REGION Network 40: ERROR - Descarga por S1
   RUNG wire#powerrail
      Contact( #EstadoZona.Rearme_CBx )
      S_RS(operand := #EstadoVI.Err_FTF_Sin_LibPHS_S1, s1 := wire#w2)
      S_Coil( #EstadoVI.Error_Mx )
   END_RUNG
   RUNG wire#powerrail
      I_Contact( #ConfigFB.SinErrorLiberarPHS_S1 )
      wire#w1
      Contact( #Mx_ET50 )
      Contact( #FTF_MSal )
      Contact( #Selec_M1_Salida )
   END_RUNG wire#w2
   RUNG wire#powerrail
      Contact( #ConfigFB.SinErrorLiberarPHS_S1 )
      I_Contact( #CNTSeg_ApHsMx.QU )
   END_RUNG wire#w1
   // the same network as SCL:
   IF #EstadoZona.Rearme_CBx THEN
       #EstadoVI.Err_FTF_Sin_LibPHS_S1 := FALSE;   // RS flip-flop
   END_IF;
   IF (NOT #ConfigFB.SinErrorLiberarPHS_S1 OR (#ConfigFB.SinErrorLiberarPHS_S1 AND NOT #CNTSeg_ApHsMx.QU)) AND #Mx_ET50 AND #FTF_MSal AND #Selec_M1_Salida THEN
       #EstadoVI.Err_FTF_Sin_LibPHS_S1 := TRUE;
   END_IF;
   IF #EstadoVI.Err_FTF_Sin_LibPHS_S1 THEN #EstadoVI.Error_Mx := TRUE; END_IF;
END_REGION

REGION Network 41: ERROR - Descarga por S3
   RUNG wire#powerrail
      Contact( #EstadoZona.Rearme_CBx )
      S_RS(operand := #EstadoVI.Err_FTF_Sin_LibPHS_S3, s1 := wire#w2)
      S_Coil( #EstadoVI.Error_Mx )
   END_RUNG
   RUNG wire#powerrail
      I_Contact( #ConfigFB.SinErrorLiberarPHS_S3 )
      wire#w1
      Contact( #Mx_ET50 )
      Contact( #FTF_MSal )
      Contact( #Selec_M3_Salida )
   END_RUNG wire#w2
   RUNG wire#powerrail
      Contact( #ConfigFB.SinErrorLiberarPHS_S3 )
      I_Contact( #CNTSeg_ApHsMx.QU )
   END_RUNG wire#w1
   // the same network as SCL:
   IF #EstadoZona.Rearme_CBx THEN
       #EstadoVI.Err_FTF_Sin_LibPHS_S3 := FALSE;   // RS flip-flop
   END_IF;
   IF (NOT #ConfigFB.SinErrorLiberarPHS_S3 OR (#ConfigFB.SinErrorLiberarPHS_S3 AND NOT #CNTSeg_ApHsMx.QU)) AND #Mx_ET50 AND #FTF_MSal AND #Selec_M3_Salida THEN
       #EstadoVI.Err_FTF_Sin_LibPHS_S3 := TRUE;
   END_IF;
   IF #EstadoVI.Err_FTF_Sin_LibPHS_S3 THEN #EstadoVI.Error_Mx := TRUE; END_IF;
END_REGION

REGION Network 42: TMP - ERROR - TimeOut Avance
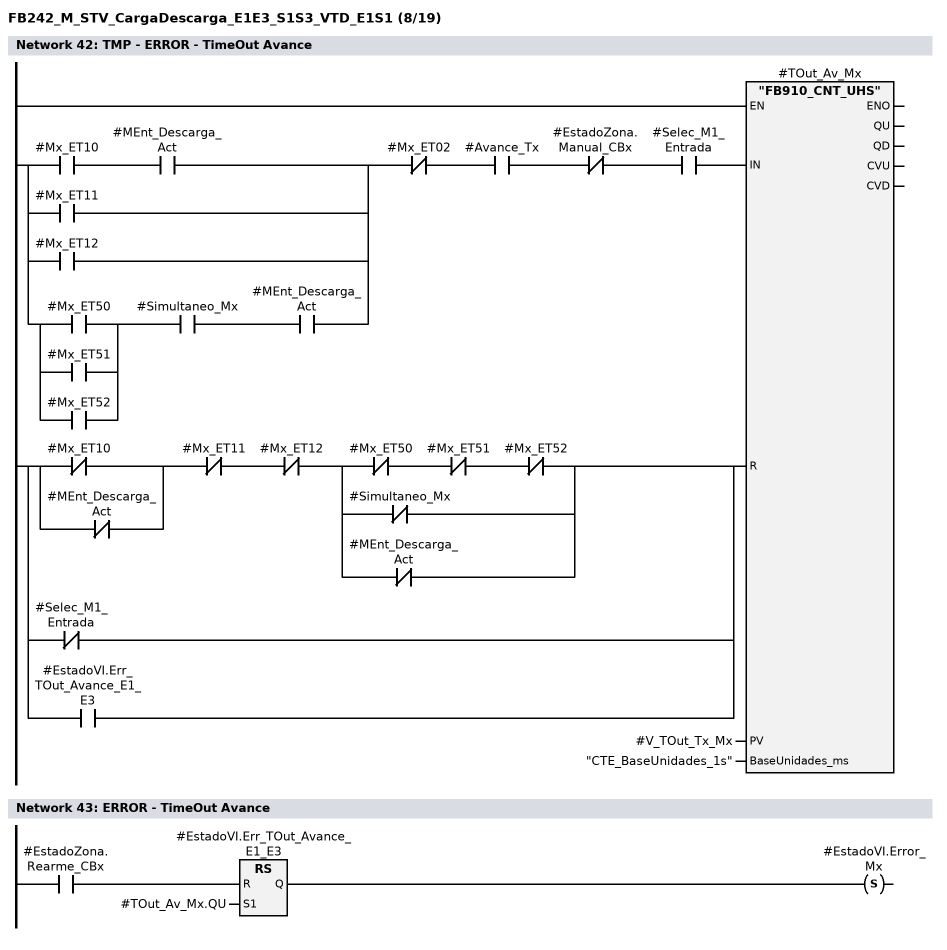
   RUNG wire#powerrail
      #TOut_Av_Mx(IN := wire#w3, R := wire#w6, PV := #V_TOut_Tx_Mx, BaseUnidades_ms := "CTE_BaseUnidades_1s", QU =>, QD =>, CVU =>, CVD =>)
   END_RUNG
   RUNG wire#powerrail
      Contact( #Mx_ET10 )
      Contact( #MEnt_Descarga_Act )
      wire#w1
      I_Contact( #Mx_ET02 )
      Contact( #Avance_Tx )
      I_Contact( #EstadoZona.Manual_CBx )
      Contact( #Selec_M1_Entrada )
   END_RUNG wire#w3
   RUNG wire#powerrail
      Contact( #Mx_ET11 )
   END_RUNG wire#w1
   RUNG wire#powerrail
      Contact( #Mx_ET12 )
   END_RUNG wire#w1
   RUNG wire#powerrail
      Contact( #Mx_ET50 )
      wire#w2
      Contact( #Simultaneo_Mx )
      Contact( #MEnt_Descarga_Act )
   END_RUNG wire#w1
   RUNG wire#powerrail
      Contact( #Mx_ET51 )
   END_RUNG wire#w2
   RUNG wire#powerrail
      Contact( #Mx_ET52 )
   END_RUNG wire#w2
   RUNG wire#powerrail
      I_Contact( #Mx_ET10 )
      wire#w4
      I_Contact( #Mx_ET11 )
      I_Contact( #Mx_ET12 )
      wire#w5
      I_Contact( #Mx_ET50 )
      I_Contact( #Mx_ET51 )
      I_Contact( #Mx_ET52 )
   END_RUNG wire#w6
   RUNG wire#powerrail
      I_Contact( #MEnt_Descarga_Act )
   END_RUNG wire#w4
   RUNG wire#w5
      I_Contact( #Simultaneo_Mx )
   END_RUNG wire#w6
   RUNG wire#w5
      I_Contact( #MEnt_Descarga_Act )
   END_RUNG wire#w6
   RUNG wire#powerrail
      I_Contact( #Selec_M1_Entrada )
   END_RUNG wire#w6
   RUNG wire#powerrail
      Contact( #EstadoVI.Err_TOut_Avance_E1_E3 )
   END_RUNG wire#w6
   // the same network as SCL:
   #TOut_Av_Mx(IN := ((#Mx_ET10 AND #MEnt_Descarga_Act) OR #Mx_ET11 OR #Mx_ET12 OR ((#Mx_ET50 OR #Mx_ET51 OR #Mx_ET52) AND #Simultaneo_Mx AND #MEnt_Descarga_Act)) AND NOT #Mx_ET02 AND #Avance_Tx AND NOT #EstadoZona.Manual_CBx AND #Selec_M1_Entrada,   // "FB910_CNT_UHS"
               R := ((NOT #Mx_ET10 OR NOT #MEnt_Descarga_Act) AND NOT #Mx_ET11 AND NOT #Mx_ET12 AND ((NOT #Mx_ET50 AND NOT #Mx_ET51 AND NOT #Mx_ET52) OR NOT #Simultaneo_Mx OR NOT #MEnt_Descarga_Act)) OR NOT #Selec_M1_Entrada OR #EstadoVI.Err_TOut_Avance_E1_E3,
               PV := #V_TOut_Tx_Mx,
               BaseUnidades_ms := "CTE_BaseUnidades_1s");
END_REGION

REGION Network 43: ERROR - TimeOut Avance
   RUNG wire#powerrail
      Contact( #EstadoZona.Rearme_CBx )
      S_RS(operand := #EstadoVI.Err_TOut_Avance_E1_E3, s1 := #TOut_Av_Mx.QU)
      S_Coil( #EstadoVI.Error_Mx )
   END_RUNG
   // the same network as SCL:
   IF #EstadoZona.Rearme_CBx THEN
       #EstadoVI.Err_TOut_Avance_E1_E3 := FALSE;   // RS flip-flop
   END_IF;
   IF #TOut_Av_Mx.QU THEN #EstadoVI.Err_TOut_Avance_E1_E3 := TRUE; END_IF;
   IF #EstadoVI.Err_TOut_Avance_E1_E3 THEN #EstadoVI.Error_Mx := TRUE; END_IF;
END_REGION

REGION Network 44: TMP - ERROR - TimeOut Retroceso
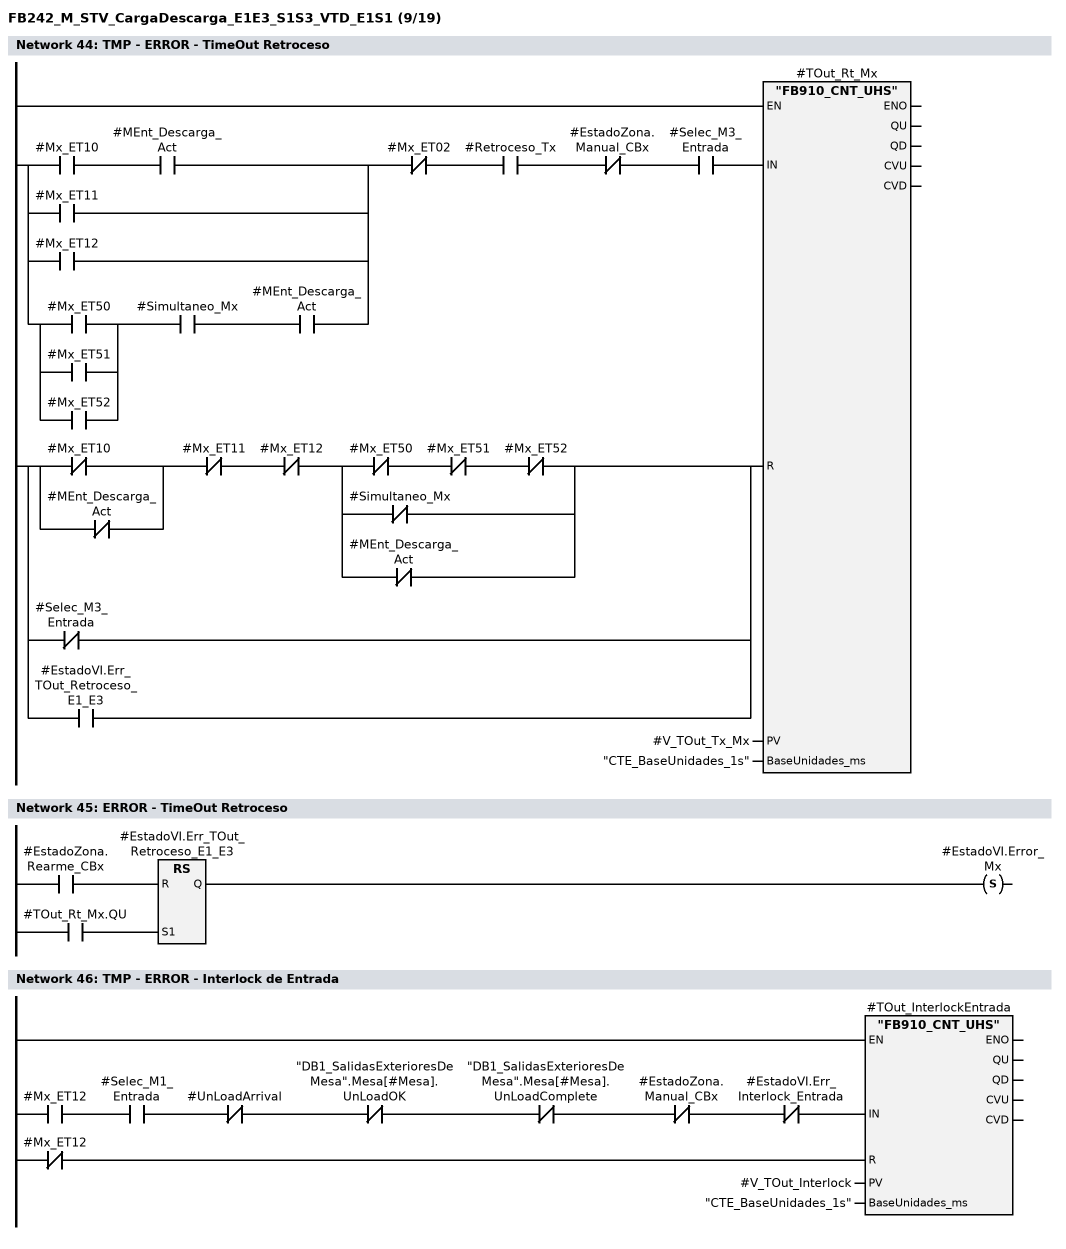
   RUNG wire#powerrail
      #TOut_Rt_Mx(IN := wire#w3, R := wire#w6, PV := #V_TOut_Tx_Mx, BaseUnidades_ms := "CTE_BaseUnidades_1s", QU =>, QD =>, CVU =>, CVD =>)
   END_RUNG
   RUNG wire#powerrail
      Contact( #Mx_ET10 )
      Contact( #MEnt_Descarga_Act )
      wire#w1
      I_Contact( #Mx_ET02 )
      Contact( #Retroceso_Tx )
      I_Contact( #EstadoZona.Manual_CBx )
      Contact( #Selec_M3_Entrada )
   END_RUNG wire#w3
   RUNG wire#powerrail
      Contact( #Mx_ET11 )
   END_RUNG wire#w1
   RUNG wire#powerrail
      Contact( #Mx_ET12 )
   END_RUNG wire#w1
   RUNG wire#powerrail
      Contact( #Mx_ET50 )
      wire#w2
      Contact( #Simultaneo_Mx )
      Contact( #MEnt_Descarga_Act )
   END_RUNG wire#w1
   RUNG wire#powerrail
      Contact( #Mx_ET51 )
   END_RUNG wire#w2
   RUNG wire#powerrail
      Contact( #Mx_ET52 )
   END_RUNG wire#w2
   RUNG wire#powerrail
      I_Contact( #Mx_ET10 )
      wire#w4
      I_Contact( #Mx_ET11 )
      I_Contact( #Mx_ET12 )
      wire#w5
      I_Contact( #Mx_ET50 )
      I_Contact( #Mx_ET51 )
      I_Contact( #Mx_ET52 )
   END_RUNG wire#w6
   RUNG wire#powerrail
      I_Contact( #MEnt_Descarga_Act )
   END_RUNG wire#w4
   RUNG wire#w5
      I_Contact( #Simultaneo_Mx )
   END_RUNG wire#w6
   RUNG wire#w5
      I_Contact( #MEnt_Descarga_Act )
   END_RUNG wire#w6
   RUNG wire#powerrail
      I_Contact( #Selec_M3_Entrada )
   END_RUNG wire#w6
   RUNG wire#powerrail
      Contact( #EstadoVI.Err_TOut_Retroceso_E1_E3 )
   END_RUNG wire#w6
   // the same network as SCL:
   #TOut_Rt_Mx(IN := ((#Mx_ET10 AND #MEnt_Descarga_Act) OR #Mx_ET11 OR #Mx_ET12 OR ((#Mx_ET50 OR #Mx_ET51 OR #Mx_ET52) AND #Simultaneo_Mx AND #MEnt_Descarga_Act)) AND NOT #Mx_ET02 AND #Retroceso_Tx AND NOT #EstadoZona.Manual_CBx AND #Selec_M3_Entrada,   // "FB910_CNT_UHS"
               R := ((NOT #Mx_ET10 OR NOT #MEnt_Descarga_Act) AND NOT #Mx_ET11 AND NOT #Mx_ET12 AND ((NOT #Mx_ET50 AND NOT #Mx_ET51 AND NOT #Mx_ET52) OR NOT #Simultaneo_Mx OR NOT #MEnt_Descarga_Act)) OR NOT #Selec_M3_Entrada OR #EstadoVI.Err_TOut_Retroceso_E1_E3,
               PV := #V_TOut_Tx_Mx,
               BaseUnidades_ms := "CTE_BaseUnidades_1s");
END_REGION

REGION Network 45: ERROR - TimeOut Retroceso
   RUNG wire#powerrail
      Contact( #EstadoZona.Rearme_CBx )
      S_RS(operand := #EstadoVI.Err_TOut_Retroceso_E1_E3, s1 := wire#w1)
      S_Coil( #EstadoVI.Error_Mx )
   END_RUNG
   RUNG wire#powerrail
      Contact( #TOut_Rt_Mx.QU )
   END_RUNG wire#w1
   // the same network as SCL:
   IF #EstadoZona.Rearme_CBx THEN
       #EstadoVI.Err_TOut_Retroceso_E1_E3 := FALSE;   // RS flip-flop
   END_IF;
   IF #TOut_Rt_Mx.QU THEN #EstadoVI.Err_TOut_Retroceso_E1_E3 := TRUE; END_IF;
   IF #EstadoVI.Err_TOut_Retroceso_E1_E3 THEN #EstadoVI.Error_Mx := TRUE; END_IF;
END_REGION

REGION Network 46: TMP - ERROR - Interlock de Entrada
   RUNG wire#powerrail
      #TOut_InterlockEntrada(IN := wire#w1, R := wire#w2, PV := #V_TOut_Interlock, BaseUnidades_ms := "CTE_BaseUnidades_1s", QU =>, QD =>, CVU =>, CVD =>)
   END_RUNG
   RUNG wire#powerrail
      Contact( #Mx_ET12 )
      Contact( #Selec_M1_Entrada )
      I_Contact( #UnLoadArrival )
      I_Contact( "DB1_SalidasExterioresDeMesa".Mesa[#Mesa].UnLoadOK )
      I_Contact( "DB1_SalidasExterioresDeMesa".Mesa[#Mesa].UnLoadComplete )
      I_Contact( #EstadoZona.Manual_CBx )
      I_Contact( #EstadoVI.Err_Interlock_Entrada )
   END_RUNG wire#w1
   RUNG wire#powerrail
      I_Contact( #Mx_ET12 )
   END_RUNG wire#w2
   // the same network as SCL:
   #TOut_InterlockEntrada(IN := #Mx_ET12 AND #Selec_M1_Entrada AND NOT #UnLoadArrival AND NOT "DB1_SalidasExterioresDeMesa".Mesa[#Mesa].UnLoadOK AND NOT "DB1_SalidasExterioresDeMesa".Mesa[#Mesa].UnLoadComplete AND NOT #EstadoZona.Manual_CBx AND NOT #EstadoVI.Err_Interlock_Entrada,   // "FB910_CNT_UHS"
                          R := NOT #Mx_ET12,
                          PV := #V_TOut_Interlock,
                          BaseUnidades_ms := "CTE_BaseUnidades_1s");
END_REGION

REGION Network 47: ERROR - Interlock de Entrada
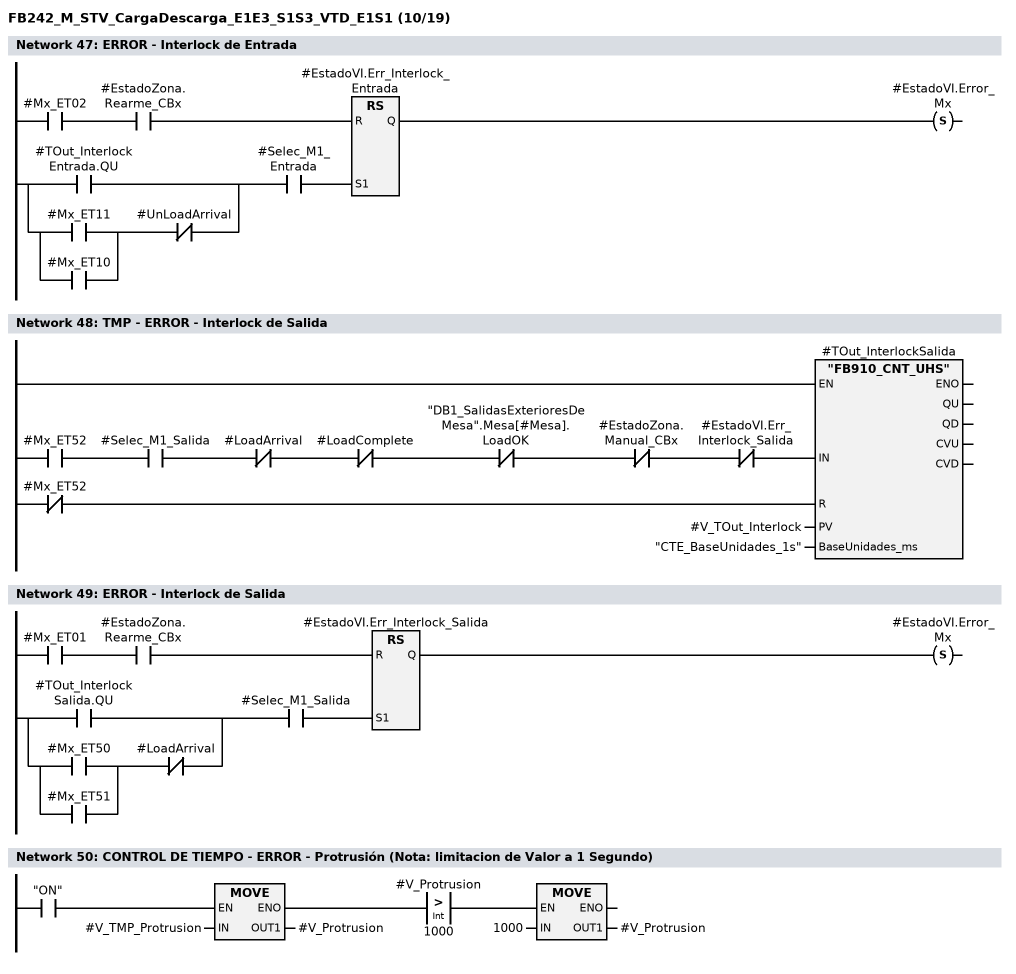
   RUNG wire#powerrail
      Contact( #Mx_ET02 )
      Contact( #EstadoZona.Rearme_CBx )
      S_RS(operand := #EstadoVI.Err_Interlock_Entrada, s1 := wire#w3)
      S_Coil( #EstadoVI.Error_Mx )
   END_RUNG
   RUNG wire#powerrail
      Contact( #TOut_InterlockEntrada.QU )
      wire#w1
      Contact( #Selec_M1_Entrada )
   END_RUNG wire#w3
   RUNG wire#powerrail
      Contact( #Mx_ET11 )
      wire#w2
      I_Contact( #UnLoadArrival )
   END_RUNG wire#w1
   RUNG wire#powerrail
      Contact( #Mx_ET10 )
   END_RUNG wire#w2
   // the same network as SCL:
   IF #Mx_ET02 AND #EstadoZona.Rearme_CBx THEN
       #EstadoVI.Err_Interlock_Entrada := FALSE;   // RS flip-flop
   END_IF;
   IF (#TOut_InterlockEntrada.QU OR ((#Mx_ET11 OR #Mx_ET10) AND NOT #UnLoadArrival)) AND #Selec_M1_Entrada THEN
       #EstadoVI.Err_Interlock_Entrada := TRUE;
   END_IF;
   IF #EstadoVI.Err_Interlock_Entrada THEN #EstadoVI.Error_Mx := TRUE; END_IF;
END_REGION

REGION Network 48: TMP - ERROR - Interlock de Salida
   RUNG wire#powerrail
      #TOut_InterlockSalida(IN := wire#w1, R := wire#w2, PV := #V_TOut_Interlock, BaseUnidades_ms := "CTE_BaseUnidades_1s", QU =>, QD =>, CVU =>, CVD =>)
   END_RUNG
   RUNG wire#powerrail
      Contact( #Mx_ET52 )
      Contact( #Selec_M1_Salida )
      I_Contact( #LoadArrival )
      I_Contact( #LoadComplete )
      I_Contact( "DB1_SalidasExterioresDeMesa".Mesa[#Mesa].LoadOK )
      I_Contact( #EstadoZona.Manual_CBx )
      I_Contact( #EstadoVI.Err_Interlock_Salida )
   END_RUNG wire#w1
   RUNG wire#powerrail
      I_Contact( #Mx_ET52 )
   END_RUNG wire#w2
   // the same network as SCL:
   #TOut_InterlockSalida(IN := #Mx_ET52 AND #Selec_M1_Salida AND NOT #LoadArrival AND NOT #LoadComplete AND NOT "DB1_SalidasExterioresDeMesa".Mesa[#Mesa].LoadOK AND NOT #EstadoZona.Manual_CBx AND NOT #EstadoVI.Err_Interlock_Salida,   // "FB910_CNT_UHS"
                         R := NOT #Mx_ET52,
                         PV := #V_TOut_Interlock,
                         BaseUnidades_ms := "CTE_BaseUnidades_1s");
END_REGION

REGION Network 49: ERROR - Interlock de Salida
   RUNG wire#powerrail
      Contact( #Mx_ET01 )
      Contact( #EstadoZona.Rearme_CBx )
      S_RS(operand := #EstadoVI.Err_Interlock_Salida, s1 := wire#w3)
      S_Coil( #EstadoVI.Error_Mx )
   END_RUNG
   RUNG wire#powerrail
      Contact( #TOut_InterlockSalida.QU )
      wire#w1
      Contact( #Selec_M1_Salida )
   END_RUNG wire#w3
   RUNG wire#powerrail
      Contact( #Mx_ET50 )
      wire#w2
      I_Contact( #LoadArrival )
   END_RUNG wire#w1
   RUNG wire#powerrail
      Contact( #Mx_ET51 )
   END_RUNG wire#w2
   // the same network as SCL:
   IF #Mx_ET01 AND #EstadoZona.Rearme_CBx THEN
       #EstadoVI.Err_Interlock_Salida := FALSE;   // RS flip-flop
   END_IF;
   IF (#TOut_InterlockSalida.QU OR ((#Mx_ET50 OR #Mx_ET51) AND NOT #LoadArrival)) AND #Selec_M1_Salida THEN
       #EstadoVI.Err_Interlock_Salida := TRUE;
   END_IF;
   IF #EstadoVI.Err_Interlock_Salida THEN #EstadoVI.Error_Mx := TRUE; END_IF;
END_REGION

REGION Network 50: CONTROL DE TIEMPO - ERROR - Protrusión (Nota: limitacion de Valor a 1 Segundo)
   RUNG wire#powerrail
      Contact( "ON" )
      Move(in := #V_TMP_Protrusion, out1 => #V_Protrusion)
      { S7_Templates := "SrcType := Int" } GT_Contact(in1 := #V_Protrusion, in2 := 1000)
      Move(in := 1000, out1 => #V_Protrusion)
   END_RUNG
   // the same network as SCL:
   IF "ON" THEN #V_Protrusion := #V_TMP_Protrusion; END_IF;
   IF "ON" AND (#V_Protrusion > 1000) THEN #V_Protrusion := 1000; END_IF;
END_REGION

REGION Network 51: TMP - ERROR - Protrusión
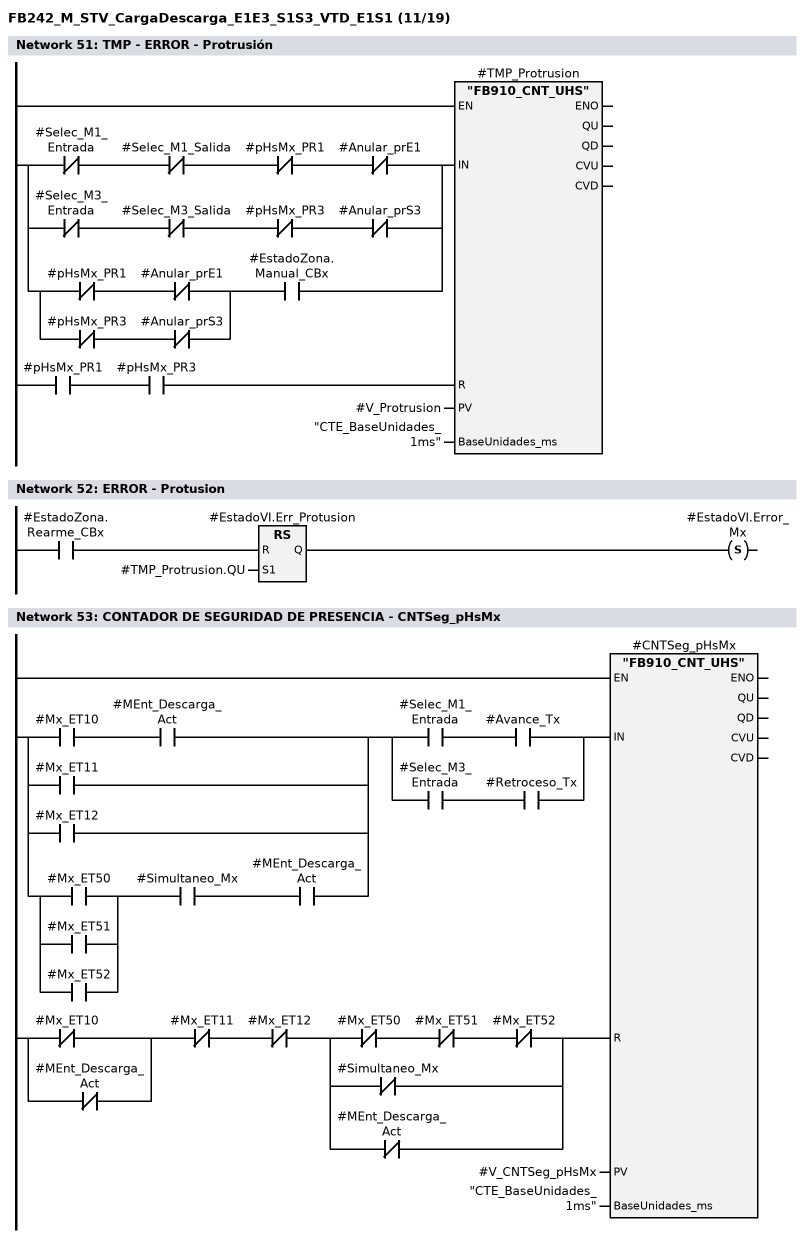
   RUNG wire#powerrail
      #TMP_Protrusion(IN := wire#w2, R := wire#w3, PV := #V_Protrusion, BaseUnidades_ms := "CTE_BaseUnidades_1ms", QU =>, QD =>, CVU =>, CVD =>)
   END_RUNG
   RUNG wire#powerrail
      I_Contact( #Selec_M1_Entrada )
      I_Contact( #Selec_M1_Salida )
      I_Contact( #pHsMx_PR1 )
      I_Contact( #Anular_prE1 )
   END_RUNG wire#w2
   RUNG wire#powerrail
      I_Contact( #Selec_M3_Entrada )
      I_Contact( #Selec_M3_Salida )
      I_Contact( #pHsMx_PR3 )
      I_Contact( #Anular_prS3 )
   END_RUNG wire#w2
   RUNG wire#powerrail
      I_Contact( #pHsMx_PR1 )
      I_Contact( #Anular_prE1 )
      wire#w1
      Contact( #EstadoZona.Manual_CBx )
   END_RUNG wire#w2
   RUNG wire#powerrail
      I_Contact( #pHsMx_PR3 )
      I_Contact( #Anular_prS3 )
   END_RUNG wire#w1
   RUNG wire#powerrail
      Contact( #pHsMx_PR1 )
      Contact( #pHsMx_PR3 )
   END_RUNG wire#w3
   // the same network as SCL:
   #TMP_Protrusion(IN := (NOT #Selec_M1_Entrada AND NOT #Selec_M1_Salida AND NOT #pHsMx_PR1 AND NOT #Anular_prE1) OR (NOT #Selec_M3_Entrada AND NOT #Selec_M3_Salida AND NOT #pHsMx_PR3 AND NOT #Anular_prS3) OR (((NOT #pHsMx_PR1 AND NOT #Anular_prE1) OR (NOT #pHsMx_PR3 AND NOT #Anular_prS3)) AND #EstadoZona.Manual_CBx),   // "FB910_CNT_UHS"
                   R := #pHsMx_PR1 AND #pHsMx_PR3,
                   PV := #V_Protrusion,
                   BaseUnidades_ms := "CTE_BaseUnidades_1ms");
END_REGION

REGION Network 52: ERROR - Protusion
   RUNG wire#powerrail
      Contact( #EstadoZona.Rearme_CBx )
      S_RS(operand := #EstadoVI.Err_Protusion, s1 := #TMP_Protrusion.QU)
      S_Coil( #EstadoVI.Error_Mx )
   END_RUNG
   // the same network as SCL:
   IF #EstadoZona.Rearme_CBx THEN
       #EstadoVI.Err_Protusion := FALSE;   // RS flip-flop
   END_IF;
   IF #TMP_Protrusion.QU THEN #EstadoVI.Err_Protusion := TRUE; END_IF;
   IF #EstadoVI.Err_Protusion THEN #EstadoVI.Error_Mx := TRUE; END_IF;
END_REGION

REGION Network 53: CONTADOR DE SEGURIDAD DE PRESENCIA - CNTSeg_pHsMx
   RUNG wire#powerrail
      #CNTSeg_pHsMx(IN := wire#w3, R := wire#w6, PV := #V_CNTSeg_pHsMx, BaseUnidades_ms := "CTE_BaseUnidades_1ms", QU =>, QD =>, CVU =>, CVD =>)
   END_RUNG
   RUNG wire#powerrail
      Contact( #Mx_ET10 )
      Contact( #MEnt_Descarga_Act )
      wire#w1
      Contact( #Selec_M1_Entrada )
      Contact( #Avance_Tx )
   END_RUNG wire#w3
   RUNG wire#powerrail
      Contact( #Mx_ET11 )
   END_RUNG wire#w1
   RUNG wire#powerrail
      Contact( #Mx_ET12 )
   END_RUNG wire#w1
   RUNG wire#powerrail
      Contact( #Mx_ET50 )
      wire#w2
      Contact( #Simultaneo_Mx )
      Contact( #MEnt_Descarga_Act )
   END_RUNG wire#w1
   RUNG wire#powerrail
      Contact( #Mx_ET51 )
   END_RUNG wire#w2
   RUNG wire#powerrail
      Contact( #Mx_ET52 )
   END_RUNG wire#w2
   RUNG wire#w1
      Contact( #Selec_M3_Entrada )
      Contact( #Retroceso_Tx )
   END_RUNG wire#w3
   RUNG wire#powerrail
      I_Contact( #Mx_ET10 )
      wire#w4
      I_Contact( #Mx_ET11 )
      I_Contact( #Mx_ET12 )
      wire#w5
      I_Contact( #Mx_ET50 )
      I_Contact( #Mx_ET51 )
      I_Contact( #Mx_ET52 )
   END_RUNG wire#w6
   RUNG wire#powerrail
      I_Contact( #MEnt_Descarga_Act )
   END_RUNG wire#w4
   RUNG wire#w5
      I_Contact( #Simultaneo_Mx )
   END_RUNG wire#w6
   RUNG wire#w5
      I_Contact( #MEnt_Descarga_Act )
   END_RUNG wire#w6
   // the same network as SCL:
   #CNTSeg_pHsMx(IN := ((#Mx_ET10 AND #MEnt_Descarga_Act) OR #Mx_ET11 OR #Mx_ET12 OR ((#Mx_ET50 OR #Mx_ET51 OR #Mx_ET52) AND #Simultaneo_Mx AND #MEnt_Descarga_Act)) AND ((#Selec_M1_Entrada AND #Avance_Tx) OR (#Selec_M3_Entrada AND #Retroceso_Tx)),   // "FB910_CNT_UHS"
                 R := (NOT #Mx_ET10 OR NOT #MEnt_Descarga_Act) AND NOT #Mx_ET11 AND NOT #Mx_ET12 AND ((NOT #Mx_ET50 AND NOT #Mx_ET51 AND NOT #Mx_ET52) OR NOT #Simultaneo_Mx OR NOT #MEnt_Descarga_Act),
                 PV := #V_CNTSeg_pHsMx,
                 BaseUnidades_ms := "CTE_BaseUnidades_1ms");
END_REGION

REGION Network 54: CONTADOR DE PRESENCIA - CNT_pHsMx
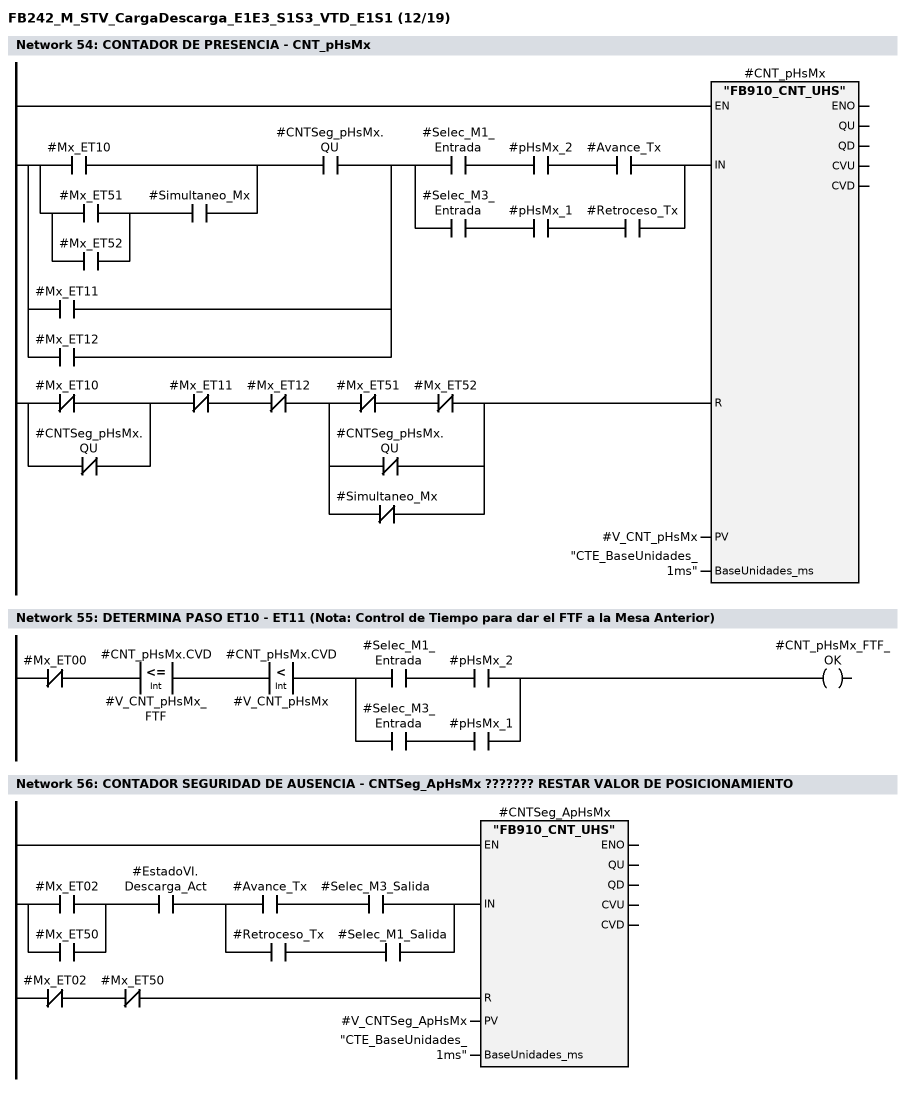
   RUNG wire#powerrail
      #CNT_pHsMx(IN := wire#w4, R := wire#w7, PV := #V_CNT_pHsMx, BaseUnidades_ms := "CTE_BaseUnidades_1ms", QU =>, QD =>, CVU =>, CVD =>)
   END_RUNG
   RUNG wire#powerrail
      Contact( #Mx_ET10 )
      wire#w1
      Contact( #CNTSeg_pHsMx.QU )
      wire#w3
      Contact( #Selec_M1_Entrada )
      Contact( #pHsMx_2 )
      Contact( #Avance_Tx )
   END_RUNG wire#w4
   RUNG wire#powerrail
      Contact( #Mx_ET51 )
      wire#w2
      Contact( #Simultaneo_Mx )
   END_RUNG wire#w1
   RUNG wire#powerrail
      Contact( #Mx_ET52 )
   END_RUNG wire#w2
   RUNG wire#powerrail
      Contact( #Mx_ET11 )
   END_RUNG wire#w3
   RUNG wire#powerrail
      Contact( #Mx_ET12 )
   END_RUNG wire#w3
   RUNG wire#w3
      Contact( #Selec_M3_Entrada )
      Contact( #pHsMx_1 )
      Contact( #Retroceso_Tx )
   END_RUNG wire#w4
   RUNG wire#powerrail
      I_Contact( #Mx_ET10 )
      wire#w5
      I_Contact( #Mx_ET11 )
      I_Contact( #Mx_ET12 )
      wire#w6
      I_Contact( #Mx_ET51 )
      I_Contact( #Mx_ET52 )
   END_RUNG wire#w7
   RUNG wire#powerrail
      I_Contact( #CNTSeg_pHsMx.QU )
   END_RUNG wire#w5
   RUNG wire#w6
      I_Contact( #CNTSeg_pHsMx.QU )
   END_RUNG wire#w7
   RUNG wire#w6
      I_Contact( #Simultaneo_Mx )
   END_RUNG wire#w7
   // the same network as SCL:
   #CNT_pHsMx(IN := (((#Mx_ET10 OR ((#Mx_ET51 OR #Mx_ET52) AND #Simultaneo_Mx)) AND #CNTSeg_pHsMx.QU) OR #Mx_ET11 OR #Mx_ET12) AND ((#Selec_M1_Entrada AND #pHsMx_2 AND #Avance_Tx) OR (#Selec_M3_Entrada AND #pHsMx_1 AND #Retroceso_Tx)),   // "FB910_CNT_UHS"
              R := (NOT #Mx_ET10 OR NOT #CNTSeg_pHsMx.QU) AND NOT #Mx_ET11 AND NOT #Mx_ET12 AND ((NOT #Mx_ET51 AND NOT #Mx_ET52) OR NOT #CNTSeg_pHsMx.QU OR NOT #Simultaneo_Mx),
              PV := #V_CNT_pHsMx,
              BaseUnidades_ms := "CTE_BaseUnidades_1ms");
END_REGION

REGION Network 55: DETERMINA PASO ET10 - ET11 (Nota: Control de Tiempo para dar el FTF a la Mesa Anterior)
   RUNG wire#powerrail
      I_Contact( #Mx_ET00 )
      { S7_Templates := "SrcType := Int" } LE_Contact(in1 := #CNT_pHsMx.CVD, in2 := #V_CNT_pHsMx_FTF)
      { S7_Templates := "SrcType := Int" } LT_Contact(in1 := #CNT_pHsMx.CVD, in2 := #V_CNT_pHsMx)
      wire#w1
      Contact( #Selec_M1_Entrada )
      Contact( #pHsMx_2 )
      wire#w2
      Coil( #CNT_pHsMx_FTF_OK )
   END_RUNG
   RUNG wire#w1
      Contact( #Selec_M3_Entrada )
      Contact( #pHsMx_1 )
   END_RUNG wire#w2
   // the same network as SCL:
   #CNT_pHsMx_FTF_OK := NOT #Mx_ET00 AND (#CNT_pHsMx.CVD <= #V_CNT_pHsMx_FTF) AND (#CNT_pHsMx.CVD < #V_CNT_pHsMx) AND ((#Selec_M1_Entrada AND #pHsMx_2) OR (#Selec_M3_Entrada AND #pHsMx_1));
END_REGION

REGION Network 56: CONTADOR SEGURIDAD DE AUSENCIA - CNTSeg_ApHsMx ??????? RESTAR VALOR DE POSICIONAMIENTO
   RUNG wire#powerrail
      #CNTSeg_ApHsMx(IN := wire#w3, R := wire#w4, PV := #V_CNTSeg_ApHsMx, BaseUnidades_ms := "CTE_BaseUnidades_1ms", QU =>, QD =>, CVU =>, CVD =>)
   END_RUNG
   RUNG wire#powerrail
      Contact( #Mx_ET02 )
      wire#w1
      Contact( #EstadoVI.Descarga_Act )
      wire#w2
      Contact( #Avance_Tx )
      Contact( #Selec_M3_Salida )
   END_RUNG wire#w3
   RUNG wire#powerrail
      Contact( #Mx_ET50 )
   END_RUNG wire#w1
   RUNG wire#w2
      Contact( #Retroceso_Tx )
      Contact( #Selec_M1_Salida )
   END_RUNG wire#w3
   RUNG wire#powerrail
      I_Contact( #Mx_ET02 )
      I_Contact( #Mx_ET50 )
   END_RUNG wire#w4
   // the same network as SCL:
   #CNTSeg_ApHsMx(IN := (#Mx_ET02 OR #Mx_ET50) AND #EstadoVI.Descarga_Act AND ((#Avance_Tx AND #Selec_M3_Salida) OR (#Retroceso_Tx AND #Selec_M1_Salida)),   // "FB910_CNT_UHS"
                  R := NOT #Mx_ET02 AND NOT #Mx_ET50,
                  PV := #V_CNTSeg_ApHsMx,
                  BaseUnidades_ms := "CTE_BaseUnidades_1ms");
END_REGION

REGION Network 57: CONTADOR DE LA AUSENCIA - CNT_ApHsMX
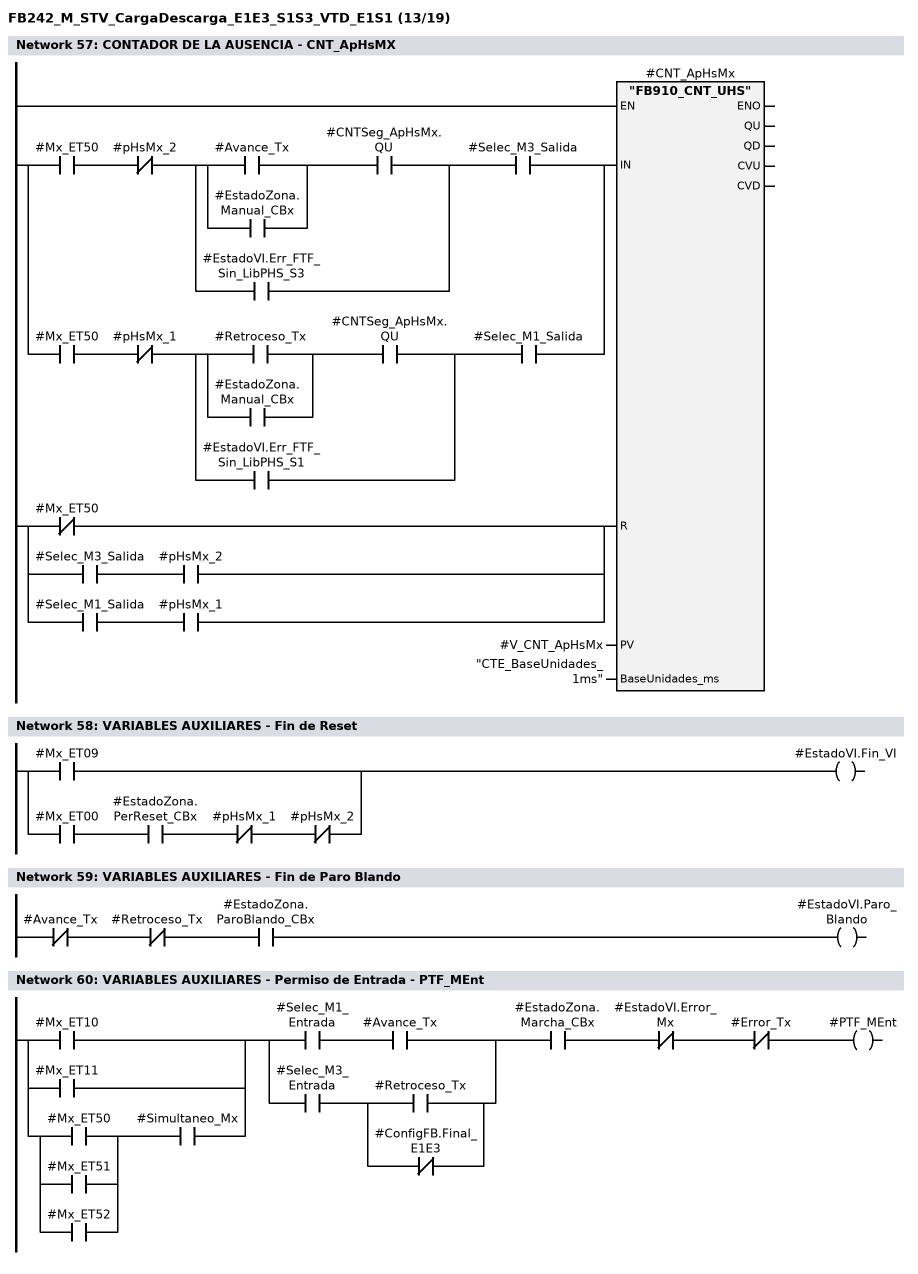
   RUNG wire#powerrail
      #CNT_ApHsMx(IN := wire#w7, R := wire#w8, PV := #V_CNT_ApHsMx, BaseUnidades_ms := "CTE_BaseUnidades_1ms", QU =>, QD =>, CVU =>, CVD =>)
   END_RUNG
   RUNG wire#powerrail
      Contact( #Mx_ET50 )
      I_Contact( #pHsMx_2 )
      wire#w1
      Contact( #Avance_Tx )
      wire#w2
      Contact( #CNTSeg_ApHsMx.QU )
      wire#w3
      Contact( #Selec_M3_Salida )
   END_RUNG wire#w7
   RUNG wire#w1
      Contact( #EstadoZona.Manual_CBx )
   END_RUNG wire#w2
   RUNG wire#w1
      Contact( #EstadoVI.Err_FTF_Sin_LibPHS_S3 )
   END_RUNG wire#w3
   RUNG wire#powerrail
      Contact( #Mx_ET50 )
      I_Contact( #pHsMx_1 )
      wire#w4
      Contact( #Retroceso_Tx )
      wire#w5
      Contact( #CNTSeg_ApHsMx.QU )
      wire#w6
      Contact( #Selec_M1_Salida )
   END_RUNG wire#w7
   RUNG wire#w4
      Contact( #EstadoZona.Manual_CBx )
   END_RUNG wire#w5
   RUNG wire#w4
      Contact( #EstadoVI.Err_FTF_Sin_LibPHS_S1 )
   END_RUNG wire#w6
   RUNG wire#powerrail
      I_Contact( #Mx_ET50 )
   END_RUNG wire#w8
   RUNG wire#powerrail
      Contact( #Selec_M3_Salida )
      Contact( #pHsMx_2 )
   END_RUNG wire#w8
   RUNG wire#powerrail
      Contact( #Selec_M1_Salida )
      Contact( #pHsMx_1 )
   END_RUNG wire#w8
   // the same network as SCL:
   #CNT_ApHsMx(IN := (#Mx_ET50 AND NOT #pHsMx_2 AND (((#Avance_Tx OR #EstadoZona.Manual_CBx) AND #CNTSeg_ApHsMx.QU) OR #EstadoVI.Err_FTF_Sin_LibPHS_S3) AND #Selec_M3_Salida) OR (#Mx_ET50 AND NOT #pHsMx_1 AND (((#Retroceso_Tx OR #EstadoZona.Manual_CBx) AND #CNTSeg_ApHsMx.QU) OR #EstadoVI.Err_FTF_Sin_LibPHS_S1) AND #Selec_M1_Salida),   // "FB910_CNT_UHS"
               R := NOT #Mx_ET50 OR (#Selec_M3_Salida AND #pHsMx_2) OR (#Selec_M1_Salida AND #pHsMx_1),
               PV := #V_CNT_ApHsMx,
               BaseUnidades_ms := "CTE_BaseUnidades_1ms");
END_REGION

REGION Network 58: VARIABLES AUXILIARES - Fin de Reset
   RUNG wire#powerrail
      Contact( #Mx_ET09 )
      wire#w1
      Coil( #EstadoVI.Fin_VI )
   END_RUNG
   RUNG wire#powerrail
      Contact( #Mx_ET00 )
      Contact( #EstadoZona.PerReset_CBx )
      I_Contact( #pHsMx_1 )
      I_Contact( #pHsMx_2 )
   END_RUNG wire#w1
   // the same network as SCL:
   #EstadoVI.Fin_VI := #Mx_ET09 OR (#Mx_ET00 AND #EstadoZona.PerReset_CBx AND NOT #pHsMx_1 AND NOT #pHsMx_2);
END_REGION

REGION Network 59: VARIABLES AUXILIARES - Fin de Paro Blando
   RUNG wire#powerrail
      I_Contact( #Avance_Tx )
      I_Contact( #Retroceso_Tx )
      Contact( #EstadoZona.ParoBlando_CBx )
      Coil( #EstadoVI.Paro_Blando )
   END_RUNG
   // the same network as SCL:
   #EstadoVI.Paro_Blando := NOT #Avance_Tx AND NOT #Retroceso_Tx AND #EstadoZona.ParoBlando_CBx;
END_REGION

REGION Network 60: VARIABLES AUXILIARES - Permiso de Entrada - PTF_MEnt
   RUNG wire#powerrail
      Contact( #Mx_ET10 )
      wire#w1
      Contact( #Selec_M1_Entrada )
      Contact( #Avance_Tx )
      wire#w3
      Contact( #EstadoZona.Marcha_CBx )
      I_Contact( #EstadoVI.Error_Mx )
      I_Contact( #Error_Tx )
      Coil( #PTF_MEnt )
   END_RUNG
   RUNG wire#powerrail
      Contact( #Mx_ET11 )
   END_RUNG wire#w1
   RUNG wire#powerrail
      Contact( #Mx_ET50 )
      wire#w2
      Contact( #Simultaneo_Mx )
   END_RUNG wire#w1
   RUNG wire#powerrail
      Contact( #Mx_ET51 )
   END_RUNG wire#w2
   RUNG wire#powerrail
      Contact( #Mx_ET52 )
   END_RUNG wire#w2
   RUNG wire#w1
      Contact( #Selec_M3_Entrada )
      wire#w4
      Contact( #Retroceso_Tx )
   END_RUNG wire#w3
   RUNG wire#w4
      I_Contact( #ConfigFB.Final_E1E3 )
   END_RUNG wire#w3
   // the same network as SCL:
   #PTF_MEnt := (#Mx_ET10 OR #Mx_ET11 OR ((#Mx_ET50 OR #Mx_ET51 OR #Mx_ET52) AND #Simultaneo_Mx)) AND ((#Selec_M1_Entrada AND #Avance_Tx) OR (#Selec_M3_Entrada AND (#Retroceso_Tx OR NOT #ConfigFB.Final_E1E3))) AND #EstadoZona.Marcha_CBx AND NOT #EstadoVI.Error_Mx AND NOT #Error_Tx;
END_REGION

REGION Network 61: VARIABLES AUXILIARES - Aviso de Salida - AVTF_MEnt
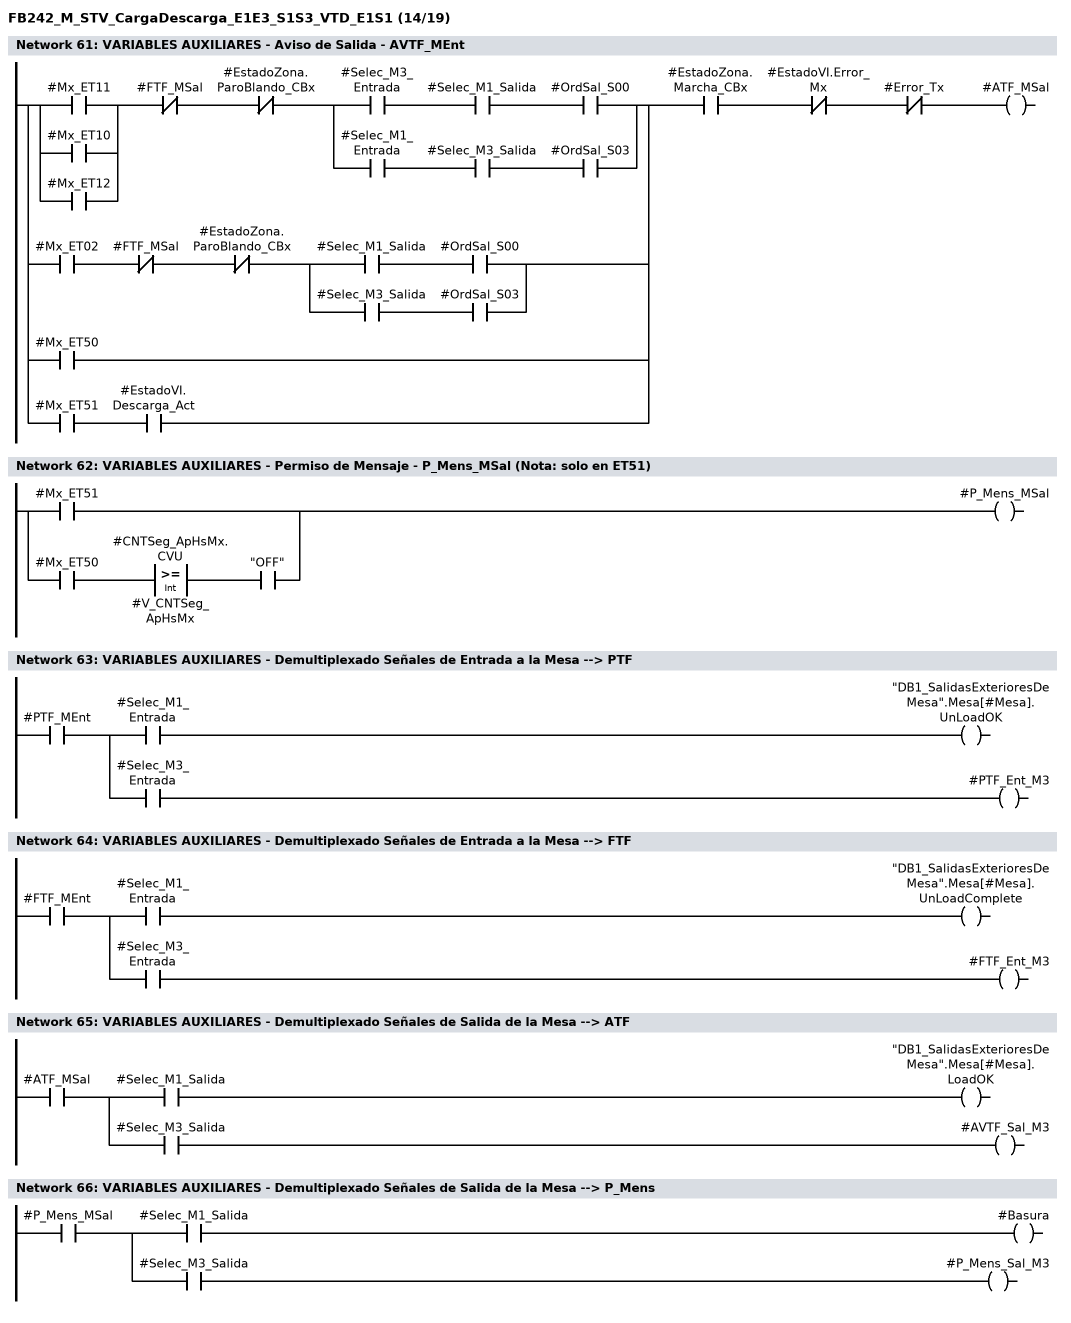
   RUNG wire#powerrail
      Contact( #Mx_ET11 )
      wire#w1
      I_Contact( #FTF_MSal )
      I_Contact( #EstadoZona.ParoBlando_CBx )
      wire#w2
      Contact( #Selec_M3_Entrada )
      Contact( #Selec_M1_Salida )
      Contact( #OrdSal_S00 )
      wire#w3
      Contact( #EstadoZona.Marcha_CBx )
      I_Contact( #EstadoVI.Error_Mx )
      I_Contact( #Error_Tx )
      Coil( #ATF_MSal )
   END_RUNG
   RUNG wire#powerrail
      Contact( #Mx_ET10 )
   END_RUNG wire#w1
   RUNG wire#powerrail
      Contact( #Mx_ET12 )
   END_RUNG wire#w1
   RUNG wire#w2
      Contact( #Selec_M1_Entrada )
      Contact( #Selec_M3_Salida )
      Contact( #OrdSal_S03 )
   END_RUNG wire#w3
   RUNG wire#powerrail
      Contact( #Mx_ET02 )
      I_Contact( #FTF_MSal )
      I_Contact( #EstadoZona.ParoBlando_CBx )
      wire#w4
      Contact( #Selec_M1_Salida )
      Contact( #OrdSal_S00 )
   END_RUNG wire#w3
   RUNG wire#w4
      Contact( #Selec_M3_Salida )
      Contact( #OrdSal_S03 )
   END_RUNG wire#w3
   RUNG wire#powerrail
      Contact( #Mx_ET50 )
   END_RUNG wire#w3
   RUNG wire#powerrail
      Contact( #Mx_ET51 )
      Contact( #EstadoVI.Descarga_Act )
   END_RUNG wire#w3
   // the same network as SCL:
   #ATF_MSal := (((#Mx_ET11 OR #Mx_ET10 OR #Mx_ET12) AND NOT #FTF_MSal AND NOT #EstadoZona.ParoBlando_CBx AND ((#Selec_M3_Entrada AND #Selec_M1_Salida AND #OrdSal_S00) OR (#Selec_M1_Entrada AND #Selec_M3_Salida AND #OrdSal_S03))) OR (#Mx_ET02 AND NOT #FTF_MSal AND NOT #EstadoZona.ParoBlando_CBx AND ((#Selec_M1_Salida AND #OrdSal_S00) OR (#Selec_M3_Salida AND #OrdSal_S03))) OR #Mx_ET50 OR (#Mx_ET51 AND #EstadoVI.Descarga_Act)) AND #EstadoZona.Marcha_CBx AND NOT #EstadoVI.Error_Mx AND NOT #Error_Tx;
END_REGION

REGION Network 62: VARIABLES AUXILIARES - Permiso de Mensaje - P_Mens_MSal (Nota: solo en ET51)
   RUNG wire#powerrail
      Contact( #Mx_ET51 )
      wire#w1
      Coil( #P_Mens_MSal )
   END_RUNG
   RUNG wire#powerrail
      Contact( #Mx_ET50 )
      { S7_Templates := "SrcType := Int" } GE_Contact(in1 := #CNTSeg_ApHsMx.CVU, in2 := #V_CNTSeg_ApHsMx)
      Contact( "OFF" )
   END_RUNG wire#w1
   // the same network as SCL:
   #P_Mens_MSal := #Mx_ET51 OR (#Mx_ET50 AND (#CNTSeg_ApHsMx.CVU >= #V_CNTSeg_ApHsMx) AND "OFF");
END_REGION

REGION Network 63: VARIABLES AUXILIARES - Demultiplexado Señales de Entrada a la Mesa --> PTF
   RUNG wire#powerrail
      Contact( #PTF_MEnt )
      wire#w1
      Contact( #Selec_M1_Entrada )
      Coil( "DB1_SalidasExterioresDeMesa".Mesa[#Mesa].UnLoadOK )
   END_RUNG
   RUNG wire#w1
      Contact( #Selec_M3_Entrada )
      Coil( #PTF_Ent_M3 )
   END_RUNG
   // the same network as SCL:
   "DB1_SalidasExterioresDeMesa".Mesa[#Mesa].UnLoadOK := #PTF_MEnt AND #Selec_M1_Entrada;
   #PTF_Ent_M3 := #PTF_MEnt AND #Selec_M3_Entrada;
END_REGION

REGION Network 64: VARIABLES AUXILIARES - Demultiplexado Señales de Entrada a la Mesa --> FTF
   RUNG wire#powerrail
      Contact( #FTF_MEnt )
      wire#w1
      Contact( #Selec_M1_Entrada )
      Coil( "DB1_SalidasExterioresDeMesa".Mesa[#Mesa].UnLoadComplete )
   END_RUNG
   RUNG wire#w1
      Contact( #Selec_M3_Entrada )
      Coil( #FTF_Ent_M3 )
   END_RUNG
   // the same network as SCL:
   "DB1_SalidasExterioresDeMesa".Mesa[#Mesa].UnLoadComplete := #FTF_MEnt AND #Selec_M1_Entrada;
   #FTF_Ent_M3 := #FTF_MEnt AND #Selec_M3_Entrada;
END_REGION

REGION Network 65: VARIABLES AUXILIARES - Demultiplexado Señales de Salida de la Mesa --> ATF
   RUNG wire#powerrail
      Contact( #ATF_MSal )
      wire#w1
      Contact( #Selec_M1_Salida )
      Coil( "DB1_SalidasExterioresDeMesa".Mesa[#Mesa].LoadOK )
   END_RUNG
   RUNG wire#w1
      Contact( #Selec_M3_Salida )
      Coil( #AVTF_Sal_M3 )
   END_RUNG
   // the same network as SCL:
   "DB1_SalidasExterioresDeMesa".Mesa[#Mesa].LoadOK := #ATF_MSal AND #Selec_M1_Salida;
   #AVTF_Sal_M3 := #ATF_MSal AND #Selec_M3_Salida;
END_REGION

REGION Network 66: VARIABLES AUXILIARES - Demultiplexado Señales de Salida de la Mesa --> P_Mens
   RUNG wire#powerrail
      Contact( #P_Mens_MSal )
      wire#w1
      Contact( #Selec_M1_Salida )
      Coil( #Basura )
   END_RUNG
   RUNG wire#w1
      Contact( #Selec_M3_Salida )
      Coil( #P_Mens_Sal_M3 )
   END_RUNG
   // the same network as SCL:
   #Basura := #P_Mens_MSal AND #Selec_M1_Salida;
   #P_Mens_Sal_M3 := #P_Mens_MSal AND #Selec_M3_Salida;
END_REGION

REGION Network 67: CONTADOR DE SIMULTANEO
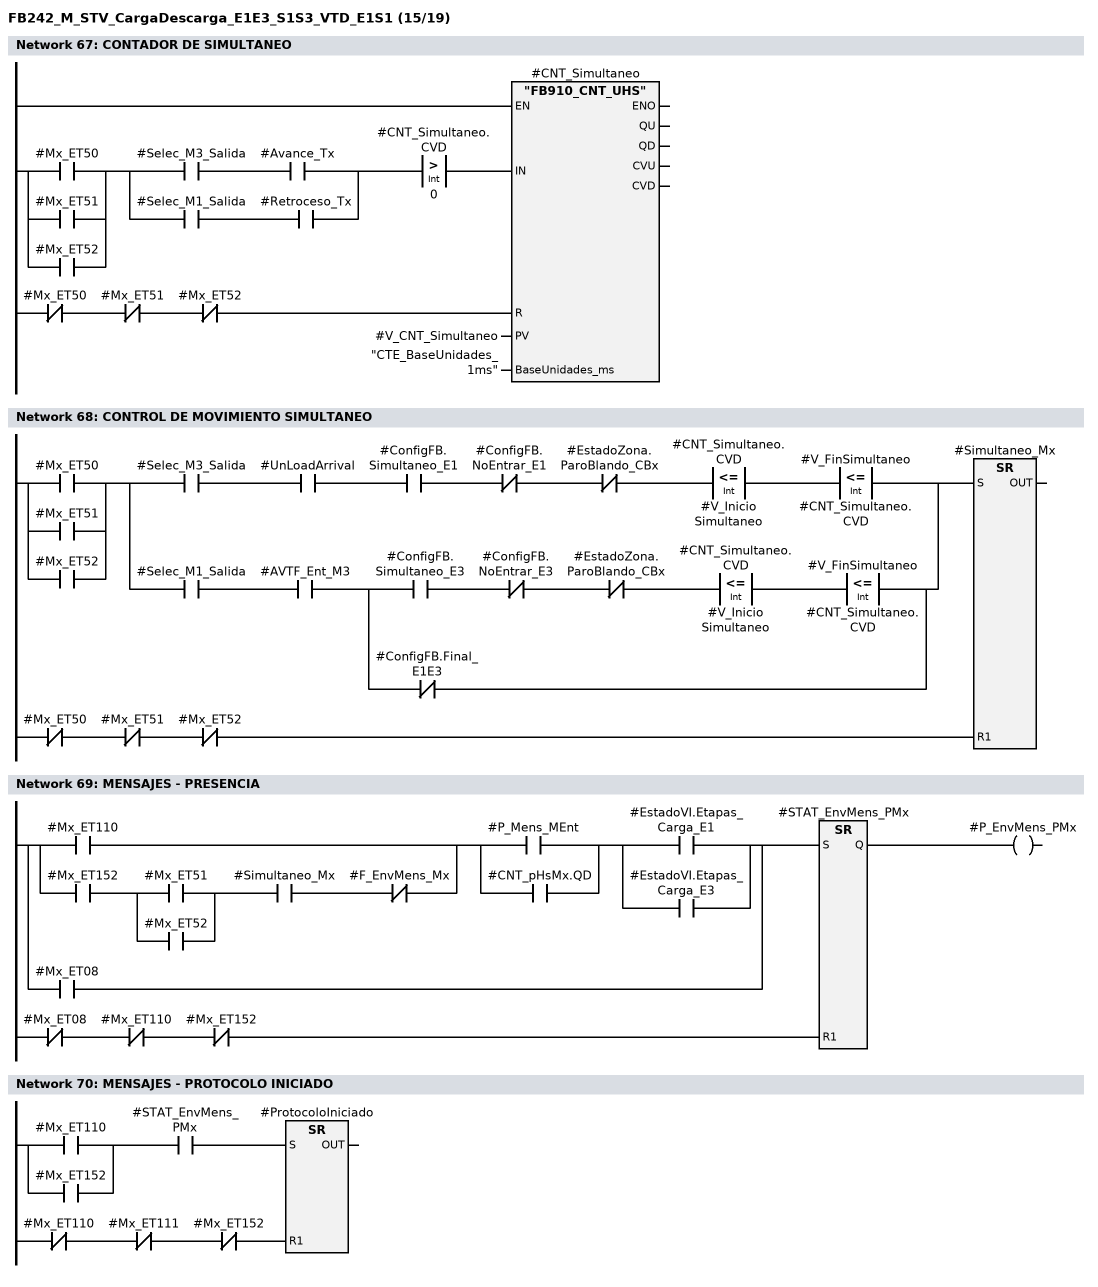
   RUNG wire#powerrail
      #CNT_Simultaneo(IN := wire#w3, R := wire#w4, PV := #V_CNT_Simultaneo, BaseUnidades_ms := "CTE_BaseUnidades_1ms", QU =>, QD =>, CVU =>, CVD =>)
   END_RUNG
   RUNG wire#powerrail
      Contact( #Mx_ET50 )
      wire#w1
      Contact( #Selec_M3_Salida )
      Contact( #Avance_Tx )
      wire#w2
      { S7_Templates := "SrcType := Int" } GT_Contact(in1 := #CNT_Simultaneo.CVD, in2 := 0)
   END_RUNG wire#w3
   RUNG wire#powerrail
      Contact( #Mx_ET51 )
   END_RUNG wire#w1
   RUNG wire#powerrail
      Contact( #Mx_ET52 )
   END_RUNG wire#w1
   RUNG wire#w1
      Contact( #Selec_M1_Salida )
      Contact( #Retroceso_Tx )
   END_RUNG wire#w2
   RUNG wire#powerrail
      I_Contact( #Mx_ET50 )
      I_Contact( #Mx_ET51 )
      I_Contact( #Mx_ET52 )
   END_RUNG wire#w4
   // the same network as SCL:
   #CNT_Simultaneo(IN := (#Mx_ET50 OR #Mx_ET51 OR #Mx_ET52) AND ((#Selec_M3_Salida AND #Avance_Tx) OR (#Selec_M1_Salida AND #Retroceso_Tx)) AND (#CNT_Simultaneo.CVD > 0),   // "FB910_CNT_UHS"
                   R := NOT #Mx_ET50 AND NOT #Mx_ET51 AND NOT #Mx_ET52,
                   PV := #V_CNT_Simultaneo,
                   BaseUnidades_ms := "CTE_BaseUnidades_1ms");
END_REGION

REGION Network 68: CONTROL DE MOVIMIENTO SIMULTANEO
   RUNG wire#powerrail
      Contact( #Mx_ET50 )
      wire#w1
      Contact( #Selec_M3_Salida )
      Contact( #UnLoadArrival )
      Contact( #ConfigFB.Simultaneo_E1 )
      I_Contact( #ConfigFB.NoEntrar_E1 )
      I_Contact( #EstadoZona.ParoBlando_CBx )
      { S7_Templates := "SrcType := Int" } LE_Contact(in1 := #CNT_Simultaneo.CVD, in2 := #V_InicioSimultaneo)
      { S7_Templates := "SrcType := Int" } LE_Contact(in1 := #V_FinSimultaneo, in2 := #CNT_Simultaneo.CVD)
      wire#w2
      S_SR(operand := #Simultaneo_Mx, r1 := wire#w4)
   END_RUNG
   RUNG wire#powerrail
      Contact( #Mx_ET51 )
   END_RUNG wire#w1
   RUNG wire#powerrail
      Contact( #Mx_ET52 )
   END_RUNG wire#w1
   RUNG wire#w1
      Contact( #Selec_M1_Salida )
      Contact( #AVTF_Ent_M3 )
      wire#w3
      Contact( #ConfigFB.Simultaneo_E3 )
      I_Contact( #ConfigFB.NoEntrar_E3 )
      I_Contact( #EstadoZona.ParoBlando_CBx )
      { S7_Templates := "SrcType := Int" } LE_Contact(in1 := #CNT_Simultaneo.CVD, in2 := #V_InicioSimultaneo)
      { S7_Templates := "SrcType := Int" } LE_Contact(in1 := #V_FinSimultaneo, in2 := #CNT_Simultaneo.CVD)
   END_RUNG wire#w2
   RUNG wire#w3
      I_Contact( #ConfigFB.Final_E1E3 )
   END_RUNG wire#w2
   RUNG wire#powerrail
      I_Contact( #Mx_ET50 )
      I_Contact( #Mx_ET51 )
      I_Contact( #Mx_ET52 )
   END_RUNG wire#w4
   // the same network as SCL:
   IF (#Mx_ET50 OR #Mx_ET51 OR #Mx_ET52) AND ((#Selec_M3_Salida AND #UnLoadArrival AND #ConfigFB.Simultaneo_E1 AND NOT #ConfigFB.NoEntrar_E1 AND NOT #EstadoZona.ParoBlando_CBx AND (#CNT_Simultaneo.CVD <= #V_InicioSimultaneo) AND (#V_FinSimultaneo <= #CNT_Simultaneo.CVD)) OR (#Selec_M1_Salida AND #AVTF_Ent_M3 AND ((#ConfigFB.Simultaneo_E3 AND NOT #ConfigFB.NoEntrar_E3 AND NOT #EstadoZona.ParoBlando_CBx AND (#CNT_Simultaneo.CVD <= #V_InicioSimultaneo) AND (#V_FinSimultaneo <= #CNT_Simultaneo.CVD)) OR NOT #ConfigFB.Final_E1E3))) THEN
       #Simultaneo_Mx := TRUE;   // SR flip-flop
   END_IF;
   IF NOT #Mx_ET50 AND NOT #Mx_ET51 AND NOT #Mx_ET52 THEN #Simultaneo_Mx := FALSE; END_IF;
END_REGION

REGION Network 69: MENSAJES - PRESENCIA
   RUNG wire#powerrail
      Contact( #Mx_ET110 )
      wire#w1
      Contact( #P_Mens_MEnt )
      wire#w4
      Contact( #EstadoVI.Etapas_Carga_E1 )
      wire#w5
      S_SR(operand := #STAT_EnvMens_PMx, r1 := wire#w6)
      Coil( #P_EnvMens_PMx )
   END_RUNG
   RUNG wire#powerrail
      Contact( #Mx_ET152 )
      wire#w2
      Contact( #Mx_ET51 )
      wire#w3
      Contact( #Simultaneo_Mx )
      I_Contact( #F_EnvMens_Mx )
   END_RUNG wire#w1
   RUNG wire#w2
      Contact( #Mx_ET52 )
   END_RUNG wire#w3
   RUNG wire#w1
      Contact( #CNT_pHsMx.QD )
   END_RUNG wire#w4
   RUNG wire#w4
      Contact( #EstadoVI.Etapas_Carga_E3 )
   END_RUNG wire#w5
   RUNG wire#powerrail
      Contact( #Mx_ET08 )
   END_RUNG wire#w5
   RUNG wire#powerrail
      I_Contact( #Mx_ET08 )
      I_Contact( #Mx_ET110 )
      I_Contact( #Mx_ET152 )
   END_RUNG wire#w6
   // the same network as SCL:
   IF ((#Mx_ET110 OR (#Mx_ET152 AND (#Mx_ET51 OR #Mx_ET52) AND #Simultaneo_Mx AND NOT #F_EnvMens_Mx)) AND (#P_Mens_MEnt OR #CNT_pHsMx.QD) AND (#EstadoVI.Etapas_Carga_E1 OR #EstadoVI.Etapas_Carga_E3)) OR #Mx_ET08 THEN
       #STAT_EnvMens_PMx := TRUE;   // SR flip-flop
   END_IF;
   IF NOT #Mx_ET08 AND NOT #Mx_ET110 AND NOT #Mx_ET152 THEN #STAT_EnvMens_PMx := FALSE; END_IF;
   #P_EnvMens_PMx := #STAT_EnvMens_PMx;
END_REGION

REGION Network 70: MENSAJES - PROTOCOLO INICIADO
   RUNG wire#powerrail
      Contact( #Mx_ET110 )
      wire#w1
      Contact( #STAT_EnvMens_PMx )
      S_SR(operand := #ProtocoloIniciado, r1 := wire#w2)
   END_RUNG
   RUNG wire#powerrail
      Contact( #Mx_ET152 )
   END_RUNG wire#w1
   RUNG wire#powerrail
      I_Contact( #Mx_ET110 )
      I_Contact( #Mx_ET111 )
      I_Contact( #Mx_ET152 )
   END_RUNG wire#w2
   // the same network as SCL:
   IF (#Mx_ET110 OR #Mx_ET152) AND #STAT_EnvMens_PMx THEN
       #ProtocoloIniciado := TRUE;   // SR flip-flop
   END_IF;
   IF NOT #Mx_ET110 AND NOT #Mx_ET111 AND NOT #Mx_ET152 THEN #ProtocoloIniciado := FALSE; END_IF;
END_REGION

REGION Network 71: MENSAJES - AUSENCIA
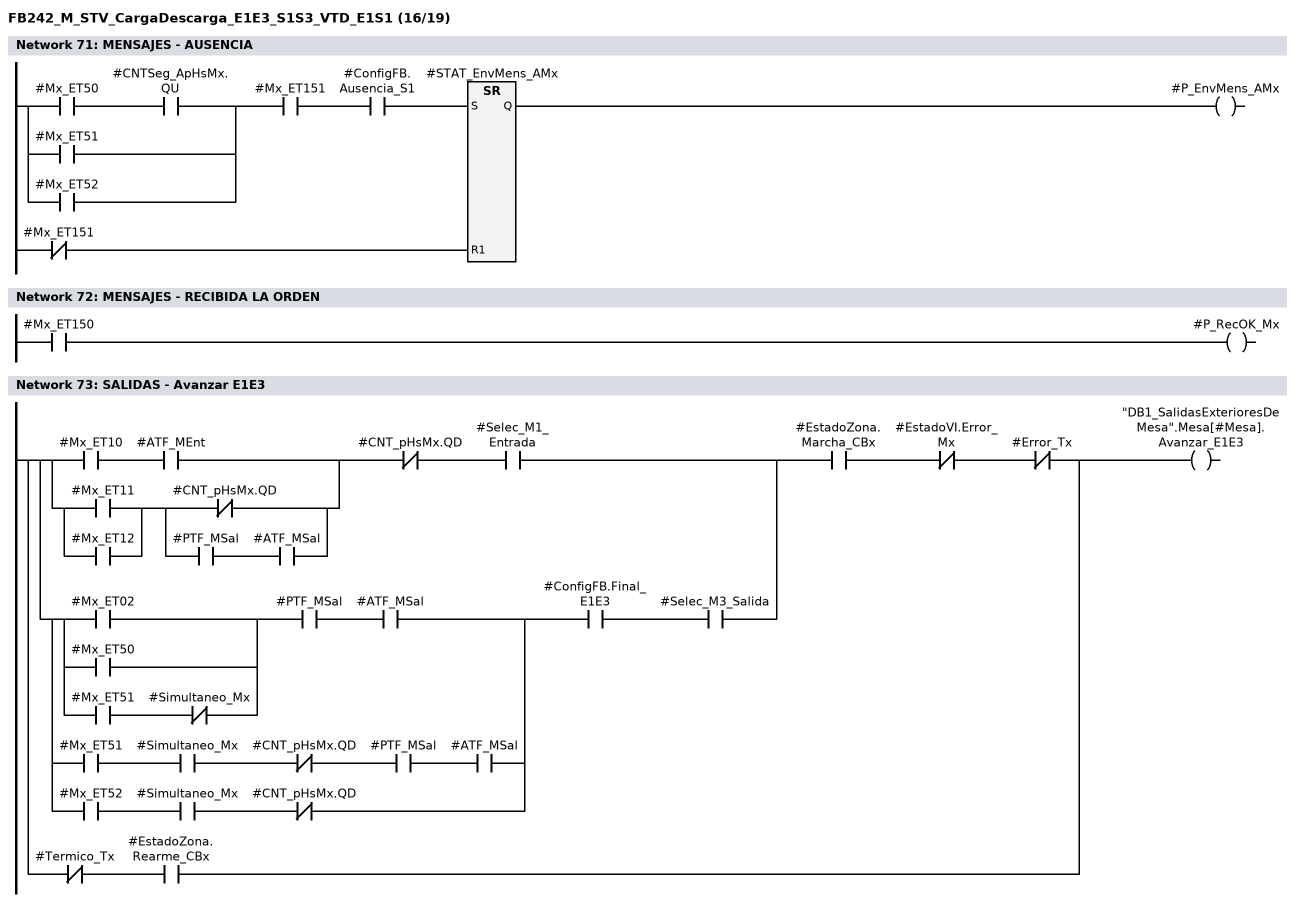
   RUNG wire#powerrail
      Contact( #Mx_ET50 )
      Contact( #CNTSeg_ApHsMx.QU )
      wire#w1
      Contact( #Mx_ET151 )
      Contact( #ConfigFB.Ausencia_S1 )
      S_SR(operand := #STAT_EnvMens_AMx, r1 := wire#w2)
      Coil( #P_EnvMens_AMx )
   END_RUNG
   RUNG wire#powerrail
      Contact( #Mx_ET51 )
   END_RUNG wire#w1
   RUNG wire#powerrail
      Contact( #Mx_ET52 )
   END_RUNG wire#w1
   RUNG wire#powerrail
      I_Contact( #Mx_ET151 )
   END_RUNG wire#w2
   // the same network as SCL:
   IF ((#Mx_ET50 AND #CNTSeg_ApHsMx.QU) OR #Mx_ET51 OR #Mx_ET52) AND #Mx_ET151 AND #ConfigFB.Ausencia_S1 THEN
       #STAT_EnvMens_AMx := TRUE;   // SR flip-flop
   END_IF;
   IF NOT #Mx_ET151 THEN #STAT_EnvMens_AMx := FALSE; END_IF;
   #P_EnvMens_AMx := #STAT_EnvMens_AMx;
END_REGION

REGION Network 72: MENSAJES - RECIBIDA LA ORDEN
   RUNG wire#powerrail
      Contact( #Mx_ET150 )
      Coil( #P_RecOK_Mx )
   END_RUNG
   // the same network as SCL:
   #P_RecOK_Mx := #Mx_ET150;
END_REGION

REGION Network 73: SALIDAS - Avanzar E1E3
   RUNG wire#powerrail
      Contact( #Mx_ET10 )
      Contact( #ATF_MEnt )
      wire#w1
      I_Contact( #CNT_pHsMx.QD )
      Contact( #Selec_M1_Entrada )
      wire#w3
      Contact( #EstadoZona.Marcha_CBx )
      I_Contact( #EstadoVI.Error_Mx )
      I_Contact( #Error_Tx )
      wire#w6
      Coil( "DB1_SalidasExterioresDeMesa".Mesa[#Mesa].Avanzar_E1E3 )
   END_RUNG
   RUNG wire#powerrail
      Contact( #Mx_ET11 )
      wire#w2
      I_Contact( #CNT_pHsMx.QD )
   END_RUNG wire#w1
   RUNG wire#powerrail
      Contact( #Mx_ET12 )
   END_RUNG wire#w2
   RUNG wire#w2
      Contact( #PTF_MSal )
      Contact( #ATF_MSal )
   END_RUNG wire#w1
   RUNG wire#powerrail
      Contact( #Mx_ET02 )
      wire#w4
      Contact( #PTF_MSal )
      Contact( #ATF_MSal )
      wire#w5
      Contact( #ConfigFB.Final_E1E3 )
      Contact( #Selec_M3_Salida )
   END_RUNG wire#w3
   RUNG wire#powerrail
      Contact( #Mx_ET50 )
   END_RUNG wire#w4
   RUNG wire#powerrail
      Contact( #Mx_ET51 )
      I_Contact( #Simultaneo_Mx )
   END_RUNG wire#w4
   RUNG wire#powerrail
      Contact( #Mx_ET51 )
      Contact( #Simultaneo_Mx )
      I_Contact( #CNT_pHsMx.QD )
      Contact( #PTF_MSal )
      Contact( #ATF_MSal )
   END_RUNG wire#w5
   RUNG wire#powerrail
      Contact( #Mx_ET52 )
      Contact( #Simultaneo_Mx )
      I_Contact( #CNT_pHsMx.QD )
   END_RUNG wire#w5
   RUNG wire#powerrail
      I_Contact( #Termico_Tx )
      Contact( #EstadoZona.Rearme_CBx )
   END_RUNG wire#w6
   // the same network as SCL:
   "DB1_SalidasExterioresDeMesa".Mesa[#Mesa].Avanzar_E1E3 := (((((#Mx_ET10 AND #ATF_MEnt) OR ((#Mx_ET11 OR #Mx_ET12) AND (NOT #CNT_pHsMx.QD OR (#PTF_MSal AND #ATF_MSal)))) AND NOT #CNT_pHsMx.QD AND #Selec_M1_Entrada) OR ((((#Mx_ET02 OR #Mx_ET50 OR (#Mx_ET51 AND NOT #Simultaneo_Mx)) AND #PTF_MSal AND #ATF_MSal) OR (#Mx_ET51 AND #Simultaneo_Mx AND NOT #CNT_pHsMx.QD AND #PTF_MSal AND #ATF_MSal) OR (#Mx_ET52 AND #Simultaneo_Mx AND NOT #CNT_pHsMx.QD)) AND #ConfigFB.Final_E1E3 AND #Selec_M3_Salida)) AND #EstadoZona.Marcha_CBx AND NOT #EstadoVI.Error_Mx AND NOT #Error_Tx) OR (NOT #Termico_Tx AND #EstadoZona.Rearme_CBx);
END_REGION

REGION Network 74: SALIDAS - Retroceder E1E3
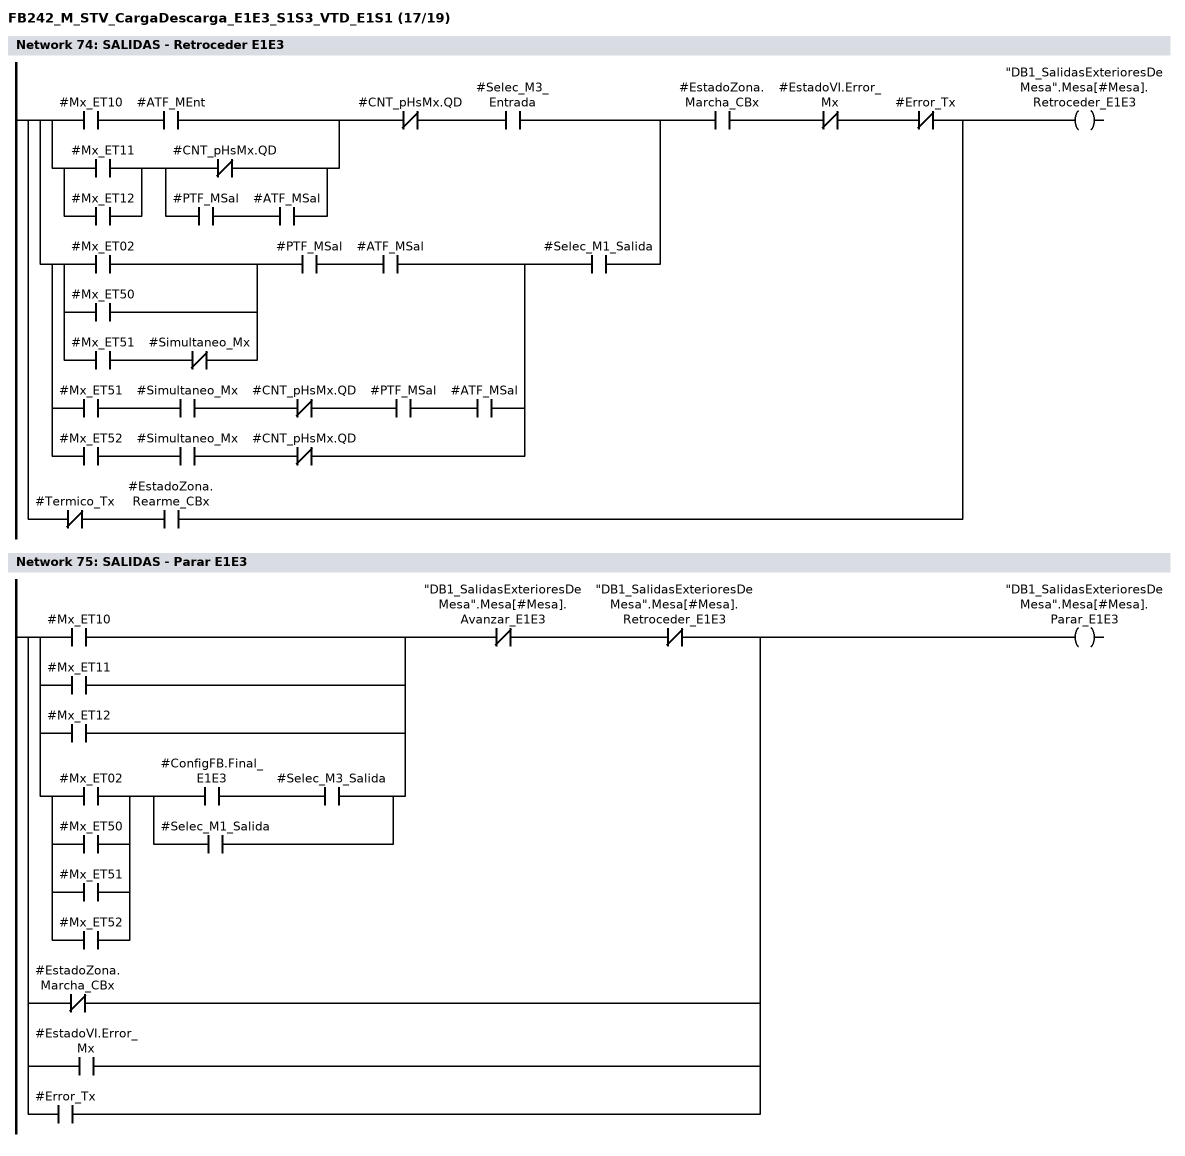
   RUNG wire#powerrail
      Contact( #Mx_ET10 )
      Contact( #ATF_MEnt )
      wire#w1
      I_Contact( #CNT_pHsMx.QD )
      Contact( #Selec_M3_Entrada )
      wire#w3
      Contact( #EstadoZona.Marcha_CBx )
      I_Contact( #EstadoVI.Error_Mx )
      I_Contact( #Error_Tx )
      wire#w6
      Coil( "DB1_SalidasExterioresDeMesa".Mesa[#Mesa].Retroceder_E1E3 )
   END_RUNG
   RUNG wire#powerrail
      Contact( #Mx_ET11 )
      wire#w2
      I_Contact( #CNT_pHsMx.QD )
   END_RUNG wire#w1
   RUNG wire#powerrail
      Contact( #Mx_ET12 )
   END_RUNG wire#w2
   RUNG wire#w2
      Contact( #PTF_MSal )
      Contact( #ATF_MSal )
   END_RUNG wire#w1
   RUNG wire#powerrail
      Contact( #Mx_ET02 )
      wire#w4
      Contact( #PTF_MSal )
      Contact( #ATF_MSal )
      wire#w5
      Contact( #Selec_M1_Salida )
   END_RUNG wire#w3
   RUNG wire#powerrail
      Contact( #Mx_ET50 )
   END_RUNG wire#w4
   RUNG wire#powerrail
      Contact( #Mx_ET51 )
      I_Contact( #Simultaneo_Mx )
   END_RUNG wire#w4
   RUNG wire#powerrail
      Contact( #Mx_ET51 )
      Contact( #Simultaneo_Mx )
      I_Contact( #CNT_pHsMx.QD )
      Contact( #PTF_MSal )
      Contact( #ATF_MSal )
   END_RUNG wire#w5
   RUNG wire#powerrail
      Contact( #Mx_ET52 )
      Contact( #Simultaneo_Mx )
      I_Contact( #CNT_pHsMx.QD )
   END_RUNG wire#w5
   RUNG wire#powerrail
      I_Contact( #Termico_Tx )
      Contact( #EstadoZona.Rearme_CBx )
   END_RUNG wire#w6
   // the same network as SCL:
   "DB1_SalidasExterioresDeMesa".Mesa[#Mesa].Retroceder_E1E3 := (((((#Mx_ET10 AND #ATF_MEnt) OR ((#Mx_ET11 OR #Mx_ET12) AND (NOT #CNT_pHsMx.QD OR (#PTF_MSal AND #ATF_MSal)))) AND NOT #CNT_pHsMx.QD AND #Selec_M3_Entrada) OR ((((#Mx_ET02 OR #Mx_ET50 OR (#Mx_ET51 AND NOT #Simultaneo_Mx)) AND #PTF_MSal AND #ATF_MSal) OR (#Mx_ET51 AND #Simultaneo_Mx AND NOT #CNT_pHsMx.QD AND #PTF_MSal AND #ATF_MSal) OR (#Mx_ET52 AND #Simultaneo_Mx AND NOT #CNT_pHsMx.QD)) AND #Selec_M1_Salida)) AND #EstadoZona.Marcha_CBx AND NOT #EstadoVI.Error_Mx AND NOT #Error_Tx) OR (NOT #Termico_Tx AND #EstadoZona.Rearme_CBx);
END_REGION

REGION Network 75: SALIDAS - Parar E1E3
   RUNG wire#powerrail
      Contact( #Mx_ET10 )
      wire#w1
      I_Contact( "DB1_SalidasExterioresDeMesa".Mesa[#Mesa].Avanzar_E1E3 )
      I_Contact( "DB1_SalidasExterioresDeMesa".Mesa[#Mesa].Retroceder_E1E3 )
      wire#w3
      Coil( "DB1_SalidasExterioresDeMesa".Mesa[#Mesa].Parar_E1E3 )
   END_RUNG
   RUNG wire#powerrail
      Contact( #Mx_ET11 )
   END_RUNG wire#w1
   RUNG wire#powerrail
      Contact( #Mx_ET12 )
   END_RUNG wire#w1
   RUNG wire#powerrail
      Contact( #Mx_ET02 )
      wire#w2
      Contact( #ConfigFB.Final_E1E3 )
      Contact( #Selec_M3_Salida )
   END_RUNG wire#w1
   RUNG wire#powerrail
      Contact( #Mx_ET50 )
   END_RUNG wire#w2
   RUNG wire#powerrail
      Contact( #Mx_ET51 )
   END_RUNG wire#w2
   RUNG wire#powerrail
      Contact( #Mx_ET52 )
   END_RUNG wire#w2
   RUNG wire#w2
      Contact( #Selec_M1_Salida )
   END_RUNG wire#w1
   RUNG wire#powerrail
      I_Contact( #EstadoZona.Marcha_CBx )
   END_RUNG wire#w3
   RUNG wire#powerrail
      Contact( #EstadoVI.Error_Mx )
   END_RUNG wire#w3
   RUNG wire#powerrail
      Contact( #Error_Tx )
   END_RUNG wire#w3
   // the same network as SCL:
   "DB1_SalidasExterioresDeMesa".Mesa[#Mesa].Parar_E1E3 := ((#Mx_ET10 OR #Mx_ET11 OR #Mx_ET12 OR ((#Mx_ET02 OR #Mx_ET50 OR #Mx_ET51 OR #Mx_ET52) AND ((#ConfigFB.Final_E1E3 AND #Selec_M3_Salida) OR #Selec_M1_Salida))) AND NOT "DB1_SalidasExterioresDeMesa".Mesa[#Mesa].Avanzar_E1E3 AND NOT "DB1_SalidasExterioresDeMesa".Mesa[#Mesa].Retroceder_E1E3) OR NOT #EstadoZona.Marcha_CBx OR #EstadoVI.Error_Mx OR #Error_Tx;
END_REGION

REGION Network 76: SALIDAS - Valor Frecuencia Lenta E1E3
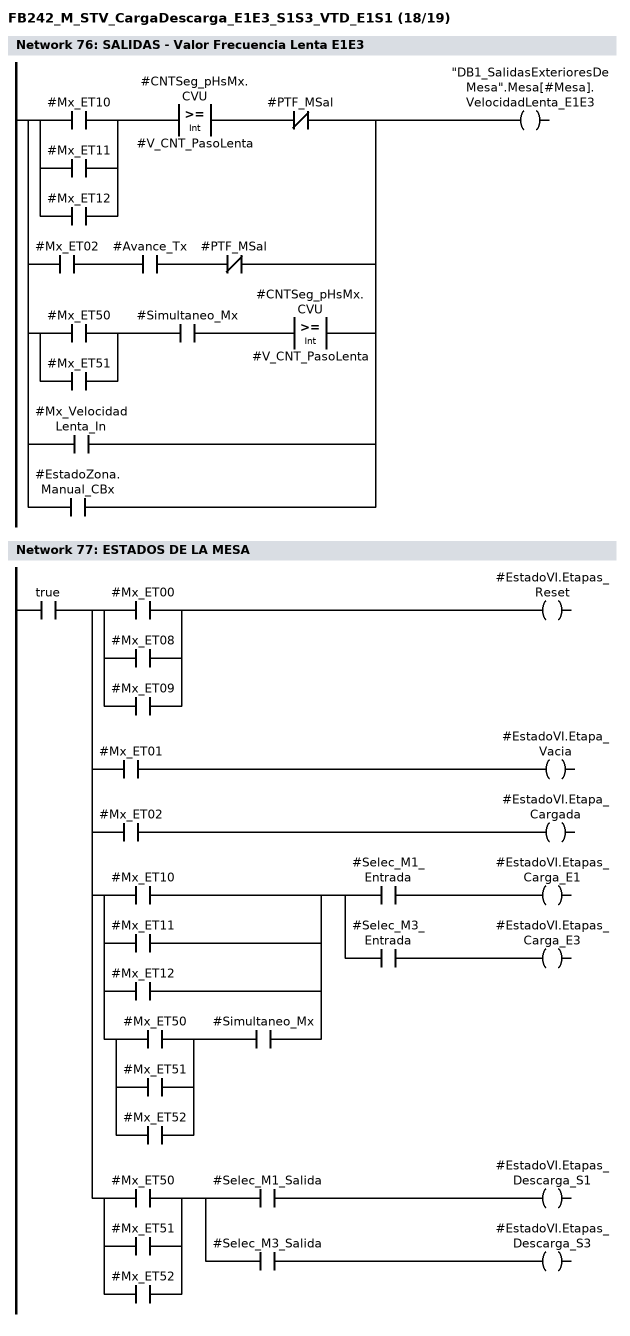
   RUNG wire#powerrail
      Contact( #Mx_ET10 )
      wire#w1
      { S7_Templates := "SrcType := Int" } GE_Contact(in1 := #CNTSeg_pHsMx.CVU, in2 := #V_CNT_PasoLenta)
      I_Contact( #PTF_MSal )
      wire#w2
      Coil( "DB1_SalidasExterioresDeMesa".Mesa[#Mesa].VelocidadLenta_E1E3 )
   END_RUNG
   RUNG wire#powerrail
      Contact( #Mx_ET11 )
   END_RUNG wire#w1
   RUNG wire#powerrail
      Contact( #Mx_ET12 )
   END_RUNG wire#w1
   RUNG wire#powerrail
      Contact( #Mx_ET02 )
      Contact( #Avance_Tx )
      I_Contact( #PTF_MSal )
   END_RUNG wire#w2
   RUNG wire#powerrail
      Contact( #Mx_ET50 )
      wire#w3
      Contact( #Simultaneo_Mx )
      { S7_Templates := "SrcType := Int" } GE_Contact(in1 := #CNTSeg_pHsMx.CVU, in2 := #V_CNT_PasoLenta)
   END_RUNG wire#w2
   RUNG wire#powerrail
      Contact( #Mx_ET51 )
   END_RUNG wire#w3
   RUNG wire#powerrail
      Contact( #Mx_VelocidadLenta_In )
   END_RUNG wire#w2
   RUNG wire#powerrail
      Contact( #EstadoZona.Manual_CBx )
   END_RUNG wire#w2
   // the same network as SCL:
   "DB1_SalidasExterioresDeMesa".Mesa[#Mesa].VelocidadLenta_E1E3 := ((#Mx_ET10 OR #Mx_ET11 OR #Mx_ET12) AND (#CNTSeg_pHsMx.CVU >= #V_CNT_PasoLenta) AND NOT #PTF_MSal) OR (#Mx_ET02 AND #Avance_Tx AND NOT #PTF_MSal) OR ((#Mx_ET50 OR #Mx_ET51) AND #Simultaneo_Mx AND (#CNTSeg_pHsMx.CVU >= #V_CNT_PasoLenta)) OR #Mx_VelocidadLenta_In OR #EstadoZona.Manual_CBx;
END_REGION

REGION Network 77: ESTADOS DE LA MESA
   RUNG wire#powerrail
      Contact( true )
      wire#w1
      Contact( #Mx_ET00 )
      wire#w2
      Coil( #EstadoVI.Etapas_Reset )
   END_RUNG
   RUNG wire#w1
      Contact( #Mx_ET08 )
   END_RUNG wire#w2
   RUNG wire#w1
      Contact( #Mx_ET09 )
   END_RUNG wire#w2
   RUNG wire#w1
      Contact( #Mx_ET01 )
      Coil( #EstadoVI.Etapa_Vacia )
   END_RUNG
   RUNG wire#w1
      Contact( #Mx_ET02 )
      Coil( #EstadoVI.Etapa_Cargada )
   END_RUNG
   RUNG wire#w1
      Contact( #Mx_ET10 )
      wire#w3
      Contact( #Selec_M1_Entrada )
      Coil( #EstadoVI.Etapas_Carga_E1 )
   END_RUNG
   RUNG wire#w1
      Contact( #Mx_ET11 )
   END_RUNG wire#w3
   RUNG wire#w1
      Contact( #Mx_ET12 )
   END_RUNG wire#w3
   RUNG wire#w1
      Contact( #Mx_ET50 )
      wire#w4
      Contact( #Simultaneo_Mx )
   END_RUNG wire#w3
   RUNG wire#w1
      Contact( #Mx_ET51 )
   END_RUNG wire#w4
   RUNG wire#w1
      Contact( #Mx_ET52 )
   END_RUNG wire#w4
   RUNG wire#w3
      Contact( #Selec_M3_Entrada )
      Coil( #EstadoVI.Etapas_Carga_E3 )
   END_RUNG
   RUNG wire#w1
      Contact( #Mx_ET50 )
      wire#w5
      Contact( #Selec_M1_Salida )
      Coil( #EstadoVI.Etapas_Descarga_S1 )
   END_RUNG
   RUNG wire#w1
      Contact( #Mx_ET51 )
   END_RUNG wire#w5
   RUNG wire#w1
      Contact( #Mx_ET52 )
   END_RUNG wire#w5
   RUNG wire#w5
      Contact( #Selec_M3_Salida )
      Coil( #EstadoVI.Etapas_Descarga_S3 )
   END_RUNG
   // the same network as SCL:
   #EstadoVI.Etapas_Reset := true AND (#Mx_ET00 OR #Mx_ET08 OR #Mx_ET09);
   #EstadoVI.Etapa_Vacia := true AND #Mx_ET01;
   #EstadoVI.Etapa_Cargada := true AND #Mx_ET02;
   #_w1 := true AND (#Mx_ET10 OR #Mx_ET11 OR #Mx_ET12 OR ((#Mx_ET50 OR #Mx_ET51 OR #Mx_ET52) AND #Simultaneo_Mx));
   #EstadoVI.Etapas_Carga_E1 := #_w1 AND #Selec_M1_Entrada;
   #EstadoVI.Etapas_Carga_E3 := #_w1 AND #Selec_M3_Entrada;
   #_w2 := true AND (#Mx_ET50 OR #Mx_ET51 OR #Mx_ET52);
   #EstadoVI.Etapas_Descarga_S1 := #_w2 AND #Selec_M1_Salida;
   #EstadoVI.Etapas_Descarga_S3 := #_w2 AND #Selec_M3_Salida;
END_REGION

REGION Network 78: ENTRADAS DE LA MESA
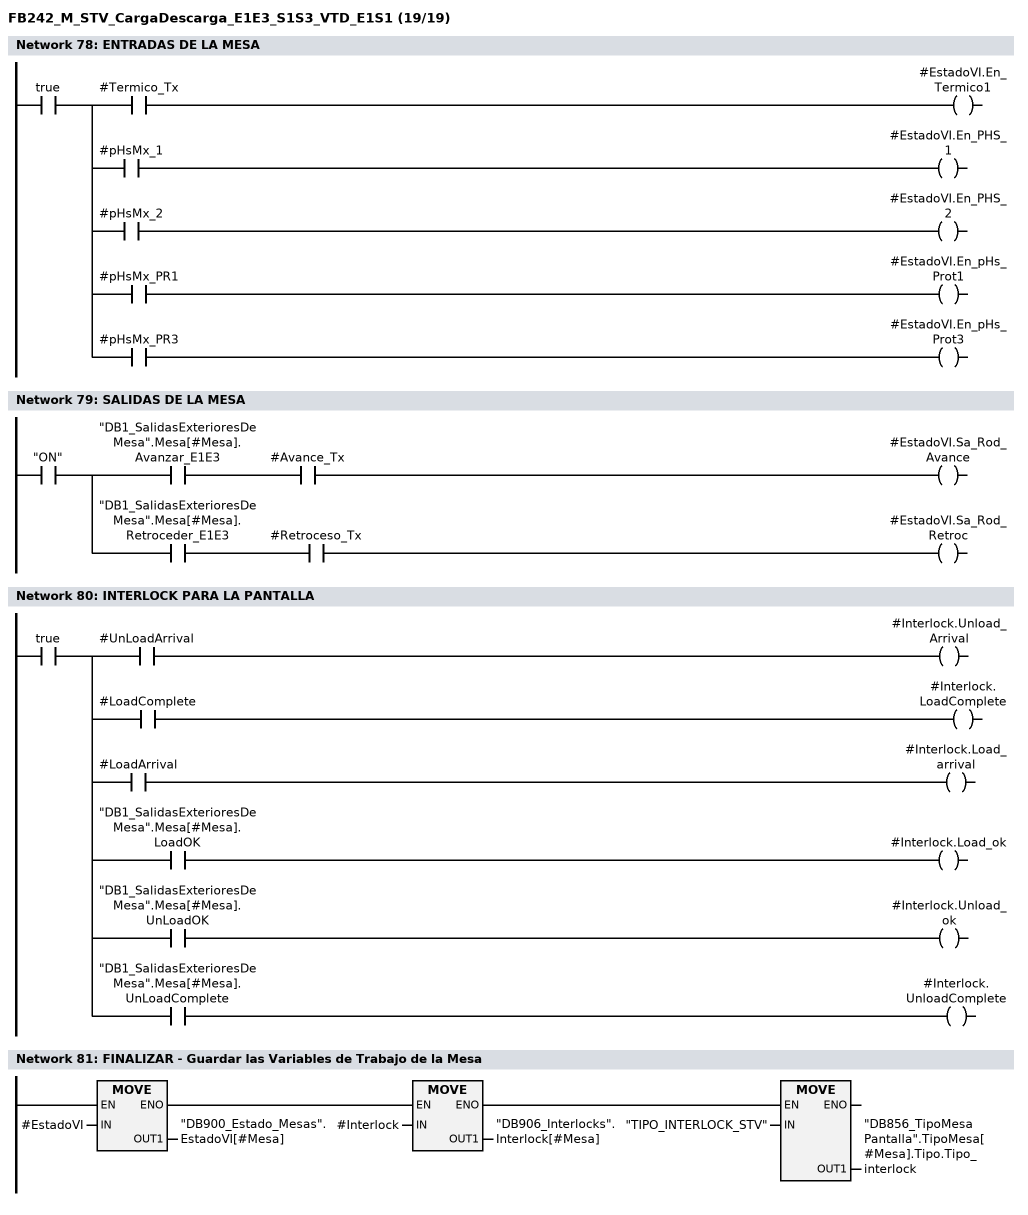
   RUNG wire#powerrail
      Contact( true )
      wire#w1
      Contact( #Termico_Tx )
      Coil( #EstadoVI.En_Termico1 )
   END_RUNG
   RUNG wire#w1
      Contact( #pHsMx_1 )
      Coil( #EstadoVI.En_PHS_1 )
   END_RUNG
   RUNG wire#w1
      Contact( #pHsMx_2 )
      Coil( #EstadoVI.En_PHS_2 )
   END_RUNG
   RUNG wire#w1
      Contact( #pHsMx_PR1 )
      Coil( #EstadoVI.En_pHs_Prot1 )
   END_RUNG
   RUNG wire#w1
      Contact( #pHsMx_PR3 )
      Coil( #EstadoVI.En_pHs_Prot3 )
   END_RUNG
   // the same network as SCL:
   #EstadoVI.En_Termico1 := true AND #Termico_Tx;
   #EstadoVI.En_PHS_1 := true AND #pHsMx_1;
   #EstadoVI.En_PHS_2 := true AND #pHsMx_2;
   #EstadoVI.En_pHs_Prot1 := true AND #pHsMx_PR1;
   #EstadoVI.En_pHs_Prot3 := true AND #pHsMx_PR3;
END_REGION

REGION Network 79: SALIDAS DE LA MESA
   RUNG wire#powerrail
      Contact( "ON" )
      wire#w1
      Contact( "DB1_SalidasExterioresDeMesa".Mesa[#Mesa].Avanzar_E1E3 )
      Contact( #Avance_Tx )
      Coil( #EstadoVI.Sa_Rod_Avance )
   END_RUNG
   RUNG wire#w1
      Contact( "DB1_SalidasExterioresDeMesa".Mesa[#Mesa].Retroceder_E1E3 )
      Contact( #Retroceso_Tx )
      Coil( #EstadoVI.Sa_Rod_Retroc )
   END_RUNG
   // the same network as SCL:
   #EstadoVI.Sa_Rod_Avance := "ON" AND "DB1_SalidasExterioresDeMesa".Mesa[#Mesa].Avanzar_E1E3 AND #Avance_Tx;
   #EstadoVI.Sa_Rod_Retroc := "ON" AND "DB1_SalidasExterioresDeMesa".Mesa[#Mesa].Retroceder_E1E3 AND #Retroceso_Tx;
END_REGION

REGION Network 80: INTERLOCK PARA LA PANTALLA
   RUNG wire#powerrail
      Contact( true )
      wire#w1
      Contact( #UnLoadArrival )
      Coil( #Interlock.Unload_Arrival )
   END_RUNG
   RUNG wire#w1
      Contact( #LoadComplete )
      Coil( #Interlock.LoadComplete )
   END_RUNG
   RUNG wire#w1
      Contact( #LoadArrival )
      Coil( #Interlock.Load_arrival )
   END_RUNG
   RUNG wire#w1
      Contact( "DB1_SalidasExterioresDeMesa".Mesa[#Mesa].LoadOK )
      Coil( #Interlock.Load_ok )
   END_RUNG
   RUNG wire#w1
      Contact( "DB1_SalidasExterioresDeMesa".Mesa[#Mesa].UnLoadOK )
      Coil( #Interlock.Unload_ok )
   END_RUNG
   RUNG wire#w1
      Contact( "DB1_SalidasExterioresDeMesa".Mesa[#Mesa].UnLoadComplete )
      Coil( #Interlock.UnloadComplete )
   END_RUNG
   // the same network as SCL:
   #Interlock.Unload_Arrival := true AND #UnLoadArrival;
   #Interlock.LoadComplete := true AND #LoadComplete;
   #Interlock.Load_arrival := true AND #LoadArrival;
   #Interlock.Load_ok := true AND "DB1_SalidasExterioresDeMesa".Mesa[#Mesa].LoadOK;
   #Interlock.Unload_ok := true AND "DB1_SalidasExterioresDeMesa".Mesa[#Mesa].UnLoadOK;
   #Interlock.UnloadComplete := true AND "DB1_SalidasExterioresDeMesa".Mesa[#Mesa].UnLoadComplete;
END_REGION

REGION Network 81: FINALIZAR - Guardar las Variables de Trabajo de la Mesa
   RUNG wire#powerrail
      Move(in := #EstadoVI, out1 => "DB900_Estado_Mesas".EstadoVI[#Mesa])
      Move(in := #Interlock, out1 => "DB906_Interlocks".Interlock[#Mesa])
      Move(in := "TIPO_INTERLOCK_STV", out1 => "DB856_TipoMesaPantalla".TipoMesa[#Mesa].Tipo.Tipo_interlock)
   END_RUNG
   // the same network as SCL:
   "DB900_Estado_Mesas".EstadoVI[#Mesa] := #EstadoVI;
   "DB906_Interlocks".Interlock[#Mesa] := #Interlock;
   "DB856_TipoMesaPantalla".TipoMesa[#Mesa].Tipo.Tipo_interlock := "TIPO_INTERLOCK_STV";
END_REGION
END_FUNCTION_BLOCK

FUNCTION_BLOCK "FB244_M_STV_Descarga_E1_S3_Doble"   // FB244, LAD
TITLE = Control del Ramal de Salidas
{ S7_Optimized_Access := 'FALSE' }
AUTHOR : VTD
NAME : 20160509
VERSION : 3.5
// stored: AutoNumber false, SetENOAutomatically false
   VAR_INPUT
      Mesa : UInt;   // Mesa de la FB
      Error_Tx : Bool;   // Error en el Tx
      EnTension : Bool;   // Existe Tension en la Mesa
      Termico_Tx : Bool;   // Proteccion del Tx
      pHsMx_1 : Bool;   // pHs de la Mesa
      pHsMx_2 : Bool;   // pHs de la Mesa
      pHsMx_PR1 : Bool;   // pHs de Protrusion de la Mesa. Nota: No existe >> ON
      pHsMx_PR3 : Bool;   // pHs de Protrusion de la Mesa. Nota: No existe >> ON
      Avance_Tx : Bool;   // Avance del Tx
      UnLoadArrival : Bool;   // UnLoad Arrival >>> VTD
      PTF_Mx_MSig : Bool;   // S3 >> Mesa Siguiente PTF
      FTF_Mx_MSig : Bool;   // S3 >> Mesa Siguiente FTF
      MSig_CargaAct : Bool;
      F_EnvMens_Mx : Bool;   // Forzar a Velociada Lenta
      Mx_VelocidadLenta_In : Bool;   // Fin de Envio de Mensaje
      OrdSal_S03 : Bool;   // Orden de Salida por S3
      S03_CargaLarga : Bool;   // Orden de Sslida de Carga Larga
      V_CNT_pHsMx : Int := 1000;   // Valor de Presencia
      V_CNT_pHsMx_FTF : Int := 200;   // Valor para activar FTF. Nota: < = V_CNT_pHsMx.
      V_CNTSeg_pHsMx : Int := 2000;   // Valor de Seguriadad para Presencia
      V_CNT_PasoLenta : Int := 2000;   // Valor de Paso a Lenta
      V_CNT_ApHsMx : Int := 200;   // Valor de Ausencia
      V_CNTSeg_ApHsMx : Int := 2000;   // Valor de Seguriadad para Ausencia
      V_TOut_Tx_Mx : Int := 15000;   // TimeOut de Entrada por E1
      V_TOut_Interlock : Int := 5000;   // TimeOut de Fin del Interlock con el VTD
      V_TMP_Protrusion : Int := 200;   // TMP de Protrusion
      V_CNT_PerdidapHs : Int := 1000;   // CNT de Perdida de pHs
   END_VAR
   VAR_OUTPUT
      P_EnvMens_PMx : Bool;   // Permiso de Enviar Mensaje de Presencia
      P_RecepOK_Mx : Bool;   // Recepcion OK
      AVTF_Mx_MSig : Bool;   // S3 >> Mesa Siguiente AVTF
      P_Mens_Mx_MSig : Bool;   // S3 >> Mesa Siguiente P_Mens
   END_VAR
   VAR
      Anular_prE1 : Bool;   // ???
      Anular_prS3 : Bool;   // ???
      Mx_ET00 : Bool;
      Mx_ET01 : Bool;
      Mx_ET02 : Bool;
      Mx_ET06 : Bool;
      Mx_ET07 : Bool;
      Mx_ET08 : Bool;
      Mx_ET09 : Bool;
      Mx_ET10 : Bool;
      Mx_ET11 : Bool;
      Mx_ET12 : Bool;
      Mx_ET110 : Bool;
      Mx_ET111 : Bool;
      Mx_ET50 : Bool;
      Mx_ET51 : Bool;
      Mx_ET52 : Bool;
      Mx_ET150 : Bool;
      Mx_ET151 : Bool;
      MemoriaCargaDoble : Bool;   // Interna >>> Memoria Carga Doble
      ProtocoloIniciado : Bool;   // Iniciado el Envio del Mensaje de Presencia
      CNT_pHsMx_FTF_OK : Bool;   // Enviar ya FTF
      STAT_EnvMens_PMx : Bool;   // Interna >> Envio del Mensaje de Presencia
      STAT_AVTF_Mx_MSig : Bool;   // Interna >> AVTF de Mx >> MSig
      CNT_pHsMx { S7_SetPoint := 'True'} : "FB910_CNT_UHS";   // CNT de la Presencia
      CNTSeg_pHsMx { S7_SetPoint := 'True'} : "FB910_CNT_UHS";   // CNT de Seguridad de la Presencia
      CNT_ApHsMx { S7_SetPoint := 'True'} : "FB910_CNT_UHS";   // CNT de la Ausencia
      CNTSeg_ApHsMx { S7_SetPoint := 'True'} : "FB910_CNT_UHS";   // CNT de Seguridad de la Ausencia
      TMP_EnTension { S7_SetPoint := 'True'} : "FB910_CNT_UHS";
      TOut_Av_Mx { S7_SetPoint := 'True'} : "FB910_CNT_UHS";   // Time Out de Entrada de E1
      TOut_Interlock { S7_SetPoint := 'True'} : "FB910_CNT_UHS";   // Time Out de Fin de Interlock con el VTD
      TMP_Protrusion { S7_SetPoint := 'True'} : "FB910_CNT_UHS";   // TMP de la Protrusion
      CNT_PerdidapHs { S7_SetPoint := 'True'} : "FB910_CNT_UHS";   // CNT de Perdida de pHs
      Interlock_manual { S7_SetPoint := 'True'} : "UDT_Interlock_manual_STV";
   END_VAR
   VAR_TEMP
      EstadoZona : "EstadoZona";   // Estado de Zona de la Mesa
      EstadoVI : "EstadosMesa";   // Estado del Vehiculo Inteliguente de la Mesa
      ConfigFB : "UDT_ConfigFB";   // Configuracion de la FB de la Mesa
      Interlock : "UDT_Interlock_STV";
      V_Protrusion : Int;
      retval : Int;
      cero : USInt;
      Aux_ET00 : Bool;
   END_VAR
BEGIN

REGION Network 1: INICIALIZAR - Recoger las Variables de Estado de la Mesa
   // Se recoge - Estado_CBx
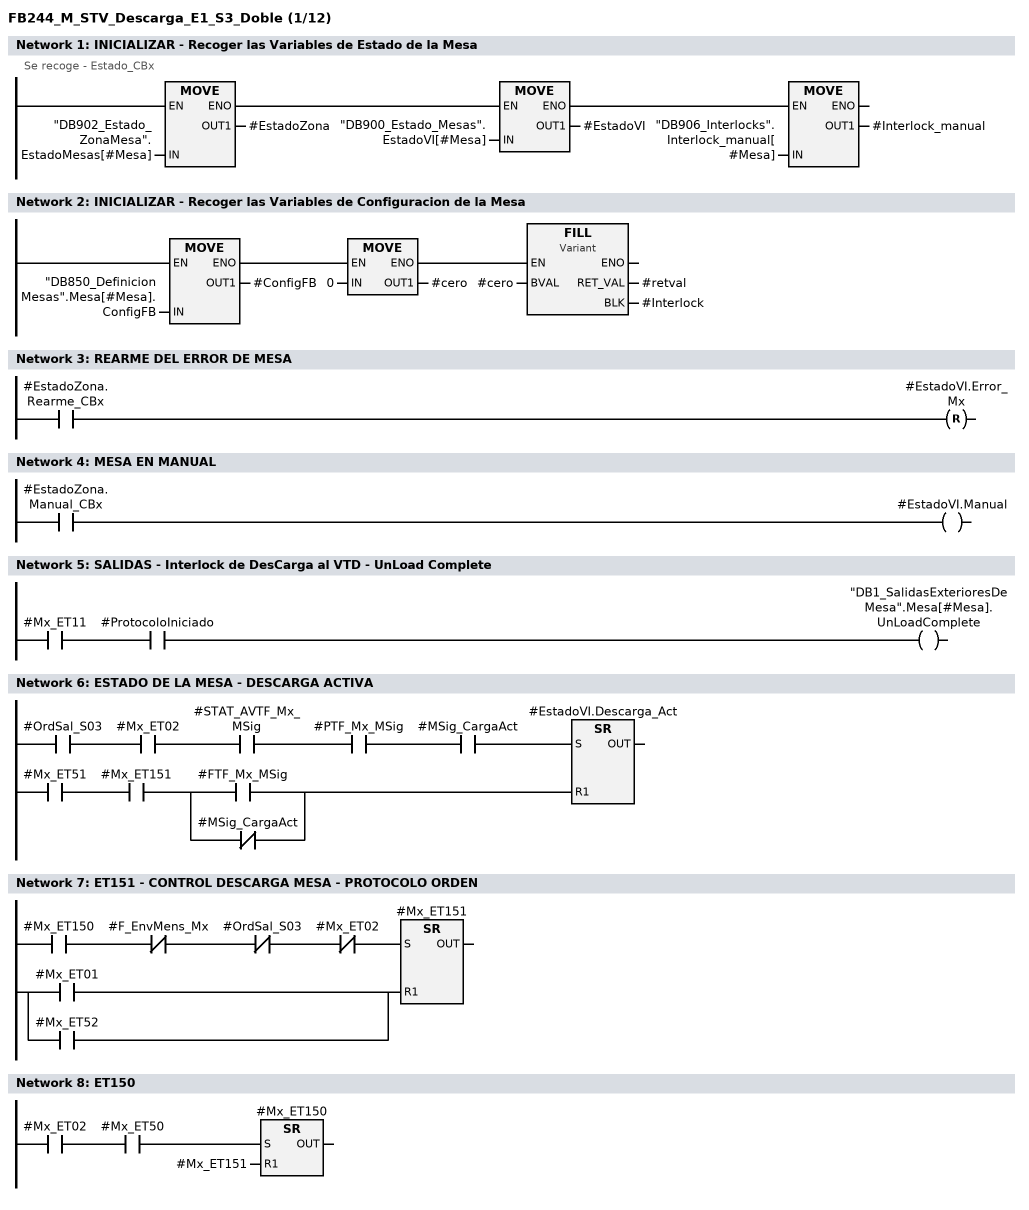
   RUNG wire#powerrail
      Move(in := "DB902_Estado_ZonaMesa".EstadoMesas[#Mesa], out1 => #EstadoZona)
      Move(in := "DB900_Estado_Mesas".EstadoVI[#Mesa], out1 => #EstadoVI)
      Move(in := "DB906_Interlocks".Interlock_manual[#Mesa], out1 => #Interlock_manual)
   END_RUNG
   // the same network as SCL:
   #EstadoZona := "DB902_Estado_ZonaMesa".EstadoMesas[#Mesa];
   #EstadoVI := "DB900_Estado_Mesas".EstadoVI[#Mesa];
   #Interlock_manual := "DB906_Interlocks".Interlock_manual[#Mesa];
END_REGION

REGION Network 2: INICIALIZAR - Recoger las Variables de Configuracion de la Mesa
   RUNG wire#powerrail
      Move(in := "DB850_DefinicionMesas".Mesa[#Mesa].ConfigFB, out1 => #ConfigFB)
      Move(in := 0, out1 => #cero)
      { S7_Templates := "ptr_type := Variant" } FILL(BVAL := #cero, RET_VAL => #retval, BLK => #Interlock)
   END_RUNG
   // the same network as SCL:
   #ConfigFB := "DB850_DefinicionMesas".Mesa[#Mesa].ConfigFB;
   #cero := 0;
   #retval := FILL(BVAL := #cero, BLK => #Interlock);
END_REGION

REGION Network 3: REARME DEL ERROR DE MESA
   RUNG wire#powerrail
      Contact( #EstadoZona.Rearme_CBx )
      R_Coil( #EstadoVI.Error_Mx )
   END_RUNG
   // the same network as SCL:
   IF #EstadoZona.Rearme_CBx THEN #EstadoVI.Error_Mx := FALSE; END_IF;
END_REGION

REGION Network 4: MESA EN MANUAL
   RUNG wire#powerrail
      Contact( #EstadoZona.Manual_CBx )
      Coil( #EstadoVI.Manual )
   END_RUNG
   // the same network as SCL:
   #EstadoVI.Manual := #EstadoZona.Manual_CBx;
END_REGION

REGION Network 5: SALIDAS - Interlock de DesCarga al VTD - UnLoad Complete
   RUNG wire#powerrail
      Contact( #Mx_ET11 )
      Contact( #ProtocoloIniciado )
      Coil( "DB1_SalidasExterioresDeMesa".Mesa[#Mesa].UnLoadComplete )
   END_RUNG
   // the same network as SCL:
   "DB1_SalidasExterioresDeMesa".Mesa[#Mesa].UnLoadComplete := #Mx_ET11 AND #ProtocoloIniciado;
END_REGION

REGION Network 6: ESTADO DE LA MESA - DESCARGA ACTIVA
   RUNG wire#powerrail
      Contact( #OrdSal_S03 )
      Contact( #Mx_ET02 )
      Contact( #STAT_AVTF_Mx_MSig )
      Contact( #PTF_Mx_MSig )
      Contact( #MSig_CargaAct )
      S_SR(operand := #EstadoVI.Descarga_Act, r1 := wire#w2)
   END_RUNG
   RUNG wire#powerrail
      Contact( #Mx_ET51 )
      Contact( #Mx_ET151 )
      wire#w1
      Contact( #FTF_Mx_MSig )
   END_RUNG wire#w2
   RUNG wire#w1
      I_Contact( #MSig_CargaAct )
   END_RUNG wire#w2
   // the same network as SCL:
   IF #OrdSal_S03 AND #Mx_ET02 AND #STAT_AVTF_Mx_MSig AND #PTF_Mx_MSig AND #MSig_CargaAct THEN
       #EstadoVI.Descarga_Act := TRUE;   // SR flip-flop
   END_IF;
   IF #Mx_ET51 AND #Mx_ET151 AND (#FTF_Mx_MSig OR NOT #MSig_CargaAct) THEN
       #EstadoVI.Descarga_Act := FALSE;
   END_IF;
END_REGION

REGION Network 7: ET151 - CONTROL DESCARGA MESA - PROTOCOLO ORDEN
   RUNG wire#powerrail
      Contact( #Mx_ET150 )
      I_Contact( #F_EnvMens_Mx )
      I_Contact( #OrdSal_S03 )
      I_Contact( #Mx_ET02 )
      S_SR(operand := #Mx_ET151, r1 := wire#w1)
   END_RUNG
   RUNG wire#powerrail
      Contact( #Mx_ET01 )
   END_RUNG wire#w1
   RUNG wire#powerrail
      Contact( #Mx_ET52 )
   END_RUNG wire#w1
   // the same network as SCL:
   IF #Mx_ET150 AND NOT #F_EnvMens_Mx AND NOT #OrdSal_S03 AND NOT #Mx_ET02 THEN
       #Mx_ET151 := TRUE;   // SR flip-flop
   END_IF;
   IF #Mx_ET01 OR #Mx_ET52 THEN #Mx_ET151 := FALSE; END_IF;
END_REGION

REGION Network 8: ET150
   RUNG wire#powerrail
      Contact( #Mx_ET02 )
      Contact( #Mx_ET50 )
      S_SR(operand := #Mx_ET150, r1 := #Mx_ET151)
   END_RUNG
   // the same network as SCL:
   IF #Mx_ET02 AND #Mx_ET50 THEN
       #Mx_ET150 := TRUE;   // SR flip-flop
   END_IF;
   IF #Mx_ET151 THEN #Mx_ET150 := FALSE; END_IF;
END_REGION

REGION Network 9: ET52 - CONTROL DESCARGA MESA
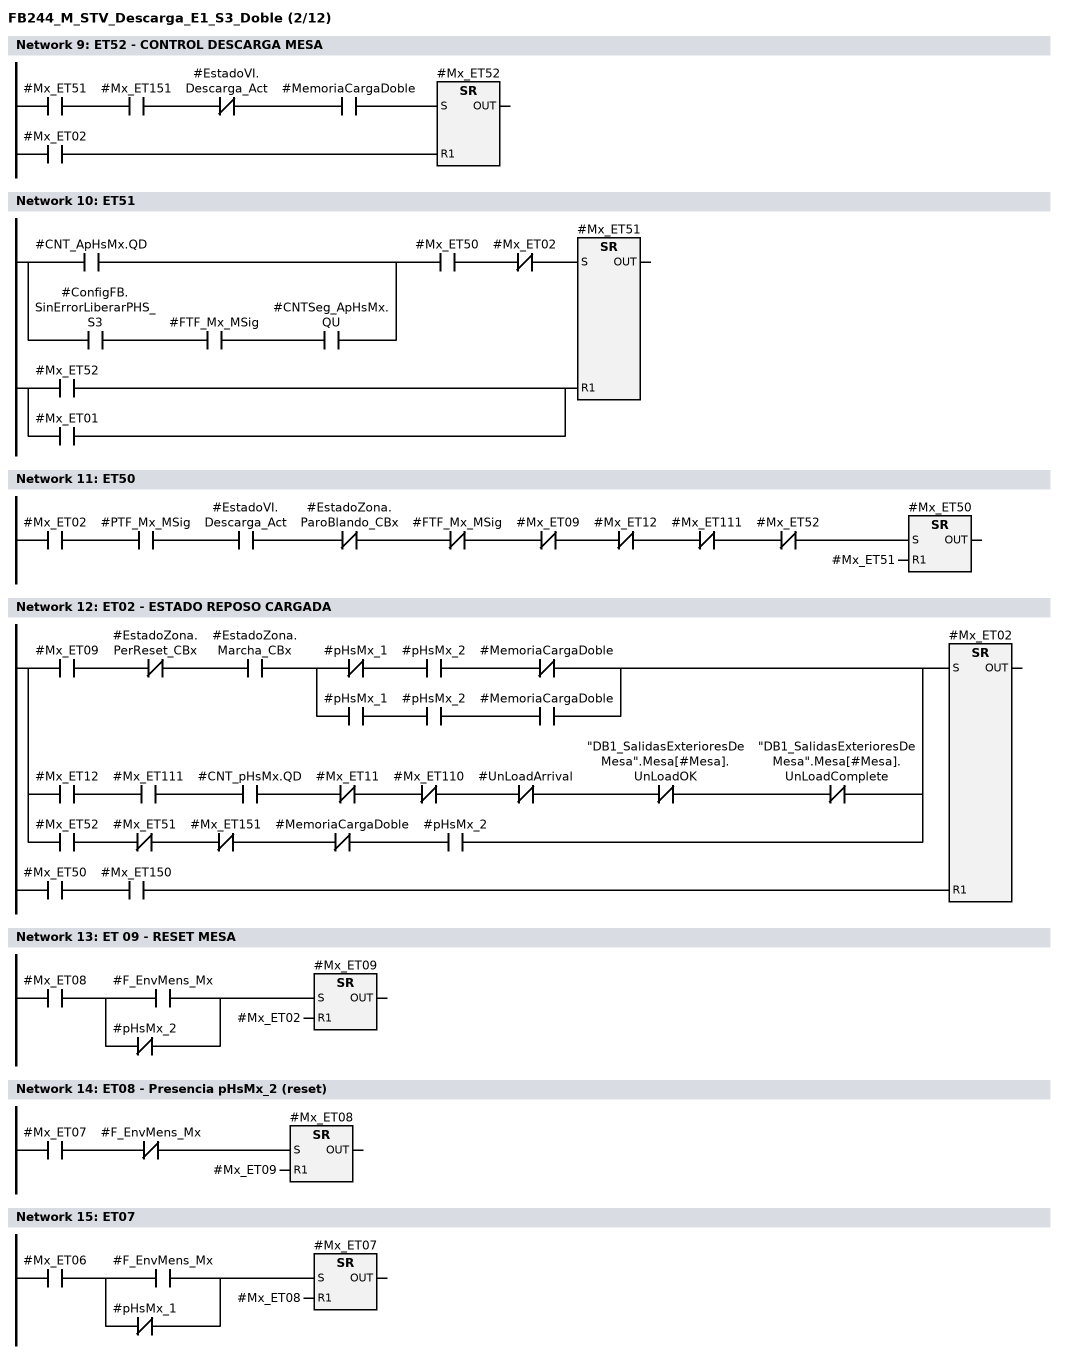
   RUNG wire#powerrail
      Contact( #Mx_ET51 )
      Contact( #Mx_ET151 )
      I_Contact( #EstadoVI.Descarga_Act )
      Contact( #MemoriaCargaDoble )
      S_SR(operand := #Mx_ET52, r1 := wire#w1)
   END_RUNG
   RUNG wire#powerrail
      Contact( #Mx_ET02 )
   END_RUNG wire#w1
   // the same network as SCL:
   IF #Mx_ET51 AND #Mx_ET151 AND NOT #EstadoVI.Descarga_Act AND #MemoriaCargaDoble THEN
       #Mx_ET52 := TRUE;   // SR flip-flop
   END_IF;
   IF #Mx_ET02 THEN #Mx_ET52 := FALSE; END_IF;
END_REGION

REGION Network 10: ET51
   RUNG wire#powerrail
      Contact( #CNT_ApHsMx.QD )
      wire#w1
      Contact( #Mx_ET50 )
      I_Contact( #Mx_ET02 )
      S_SR(operand := #Mx_ET51, r1 := wire#w2)
   END_RUNG
   RUNG wire#powerrail
      Contact( #ConfigFB.SinErrorLiberarPHS_S3 )
      Contact( #FTF_Mx_MSig )
      Contact( #CNTSeg_ApHsMx.QU )
   END_RUNG wire#w1
   RUNG wire#powerrail
      Contact( #Mx_ET52 )
   END_RUNG wire#w2
   RUNG wire#powerrail
      Contact( #Mx_ET01 )
   END_RUNG wire#w2
   // the same network as SCL:
   IF (#CNT_ApHsMx.QD OR (#ConfigFB.SinErrorLiberarPHS_S3 AND #FTF_Mx_MSig AND #CNTSeg_ApHsMx.QU)) AND #Mx_ET50 AND NOT #Mx_ET02 THEN
       #Mx_ET51 := TRUE;   // SR flip-flop
   END_IF;
   IF #Mx_ET52 OR #Mx_ET01 THEN #Mx_ET51 := FALSE; END_IF;
END_REGION

REGION Network 11: ET50
   RUNG wire#powerrail
      Contact( #Mx_ET02 )
      Contact( #PTF_Mx_MSig )
      Contact( #EstadoVI.Descarga_Act )
      I_Contact( #EstadoZona.ParoBlando_CBx )
      I_Contact( #FTF_Mx_MSig )
      I_Contact( #Mx_ET09 )
      I_Contact( #Mx_ET12 )
      I_Contact( #Mx_ET111 )
      I_Contact( #Mx_ET52 )
      S_SR(operand := #Mx_ET50, r1 := #Mx_ET51)
   END_RUNG
   // the same network as SCL:
   IF #Mx_ET02 AND #PTF_Mx_MSig AND #EstadoVI.Descarga_Act AND NOT #EstadoZona.ParoBlando_CBx AND NOT #FTF_Mx_MSig AND NOT #Mx_ET09 AND NOT #Mx_ET12 AND NOT #Mx_ET111 AND NOT #Mx_ET52 THEN
       #Mx_ET50 := TRUE;   // SR flip-flop
   END_IF;
   IF #Mx_ET51 THEN #Mx_ET50 := FALSE; END_IF;
END_REGION

REGION Network 12: ET02 - ESTADO REPOSO CARGADA
   RUNG wire#powerrail
      Contact( #Mx_ET09 )
      I_Contact( #EstadoZona.PerReset_CBx )
      Contact( #EstadoZona.Marcha_CBx )
      wire#w1
      I_Contact( #pHsMx_1 )
      Contact( #pHsMx_2 )
      I_Contact( #MemoriaCargaDoble )
      wire#w2
      S_SR(operand := #Mx_ET02, r1 := wire#w3)
   END_RUNG
   RUNG wire#w1
      Contact( #pHsMx_1 )
      Contact( #pHsMx_2 )
      Contact( #MemoriaCargaDoble )
   END_RUNG wire#w2
   RUNG wire#powerrail
      Contact( #Mx_ET12 )
      Contact( #Mx_ET111 )
      Contact( #CNT_pHsMx.QD )
      I_Contact( #Mx_ET11 )
      I_Contact( #Mx_ET110 )
      I_Contact( #UnLoadArrival )
      I_Contact( "DB1_SalidasExterioresDeMesa".Mesa[#Mesa].UnLoadOK )
      I_Contact( "DB1_SalidasExterioresDeMesa".Mesa[#Mesa].UnLoadComplete )
   END_RUNG wire#w2
   RUNG wire#powerrail
      Contact( #Mx_ET52 )
      I_Contact( #Mx_ET51 )
      I_Contact( #Mx_ET151 )
      I_Contact( #MemoriaCargaDoble )
      Contact( #pHsMx_2 )
   END_RUNG wire#w2
   RUNG wire#powerrail
      Contact( #Mx_ET50 )
      Contact( #Mx_ET150 )
   END_RUNG wire#w3
   // the same network as SCL:
   IF (#Mx_ET09 AND NOT #EstadoZona.PerReset_CBx AND #EstadoZona.Marcha_CBx AND ((NOT #pHsMx_1 AND #pHsMx_2 AND NOT #MemoriaCargaDoble) OR (#pHsMx_1 AND #pHsMx_2 AND #MemoriaCargaDoble))) OR (#Mx_ET12 AND #Mx_ET111 AND #CNT_pHsMx.QD AND NOT #Mx_ET11 AND NOT #Mx_ET110 AND NOT #UnLoadArrival AND NOT "DB1_SalidasExterioresDeMesa".Mesa[#Mesa].UnLoadOK AND NOT "DB1_SalidasExterioresDeMesa".Mesa[#Mesa].UnLoadComplete) OR (#Mx_ET52 AND NOT #Mx_ET51 AND NOT #Mx_ET151 AND NOT #MemoriaCargaDoble AND #pHsMx_2) THEN
       #Mx_ET02 := TRUE;   // SR flip-flop
   END_IF;
   IF #Mx_ET50 AND #Mx_ET150 THEN #Mx_ET02 := FALSE; END_IF;
END_REGION

REGION Network 13: ET 09 - RESET MESA
   RUNG wire#powerrail
      Contact( #Mx_ET08 )
      wire#w1
      Contact( #F_EnvMens_Mx )
      wire#w2
      S_SR(operand := #Mx_ET09, r1 := #Mx_ET02)
   END_RUNG
   RUNG wire#w1
      I_Contact( #pHsMx_2 )
   END_RUNG wire#w2
   // the same network as SCL:
   IF #Mx_ET08 AND (#F_EnvMens_Mx OR NOT #pHsMx_2) THEN
       #Mx_ET09 := TRUE;   // SR flip-flop
   END_IF;
   IF #Mx_ET02 THEN #Mx_ET09 := FALSE; END_IF;
END_REGION

REGION Network 14: ET08 - Presencia pHsMx_2 (reset)
   RUNG wire#powerrail
      Contact( #Mx_ET07 )
      I_Contact( #F_EnvMens_Mx )
      S_SR(operand := #Mx_ET08, r1 := #Mx_ET09)
   END_RUNG
   // the same network as SCL:
   IF #Mx_ET07 AND NOT #F_EnvMens_Mx THEN
       #Mx_ET08 := TRUE;   // SR flip-flop
   END_IF;
   IF #Mx_ET09 THEN #Mx_ET08 := FALSE; END_IF;
END_REGION

REGION Network 15: ET07
   RUNG wire#powerrail
      Contact( #Mx_ET06 )
      wire#w1
      Contact( #F_EnvMens_Mx )
      wire#w2
      S_SR(operand := #Mx_ET07, r1 := #Mx_ET08)
   END_RUNG
   RUNG wire#w1
      I_Contact( #pHsMx_1 )
   END_RUNG wire#w2
   // the same network as SCL:
   IF #Mx_ET06 AND (#F_EnvMens_Mx OR NOT #pHsMx_1) THEN
       #Mx_ET07 := TRUE;   // SR flip-flop
   END_IF;
   IF #Mx_ET08 THEN #Mx_ET07 := FALSE; END_IF;
END_REGION

REGION Network 16: ET06 - Presencia pHsMx_1 (reset)
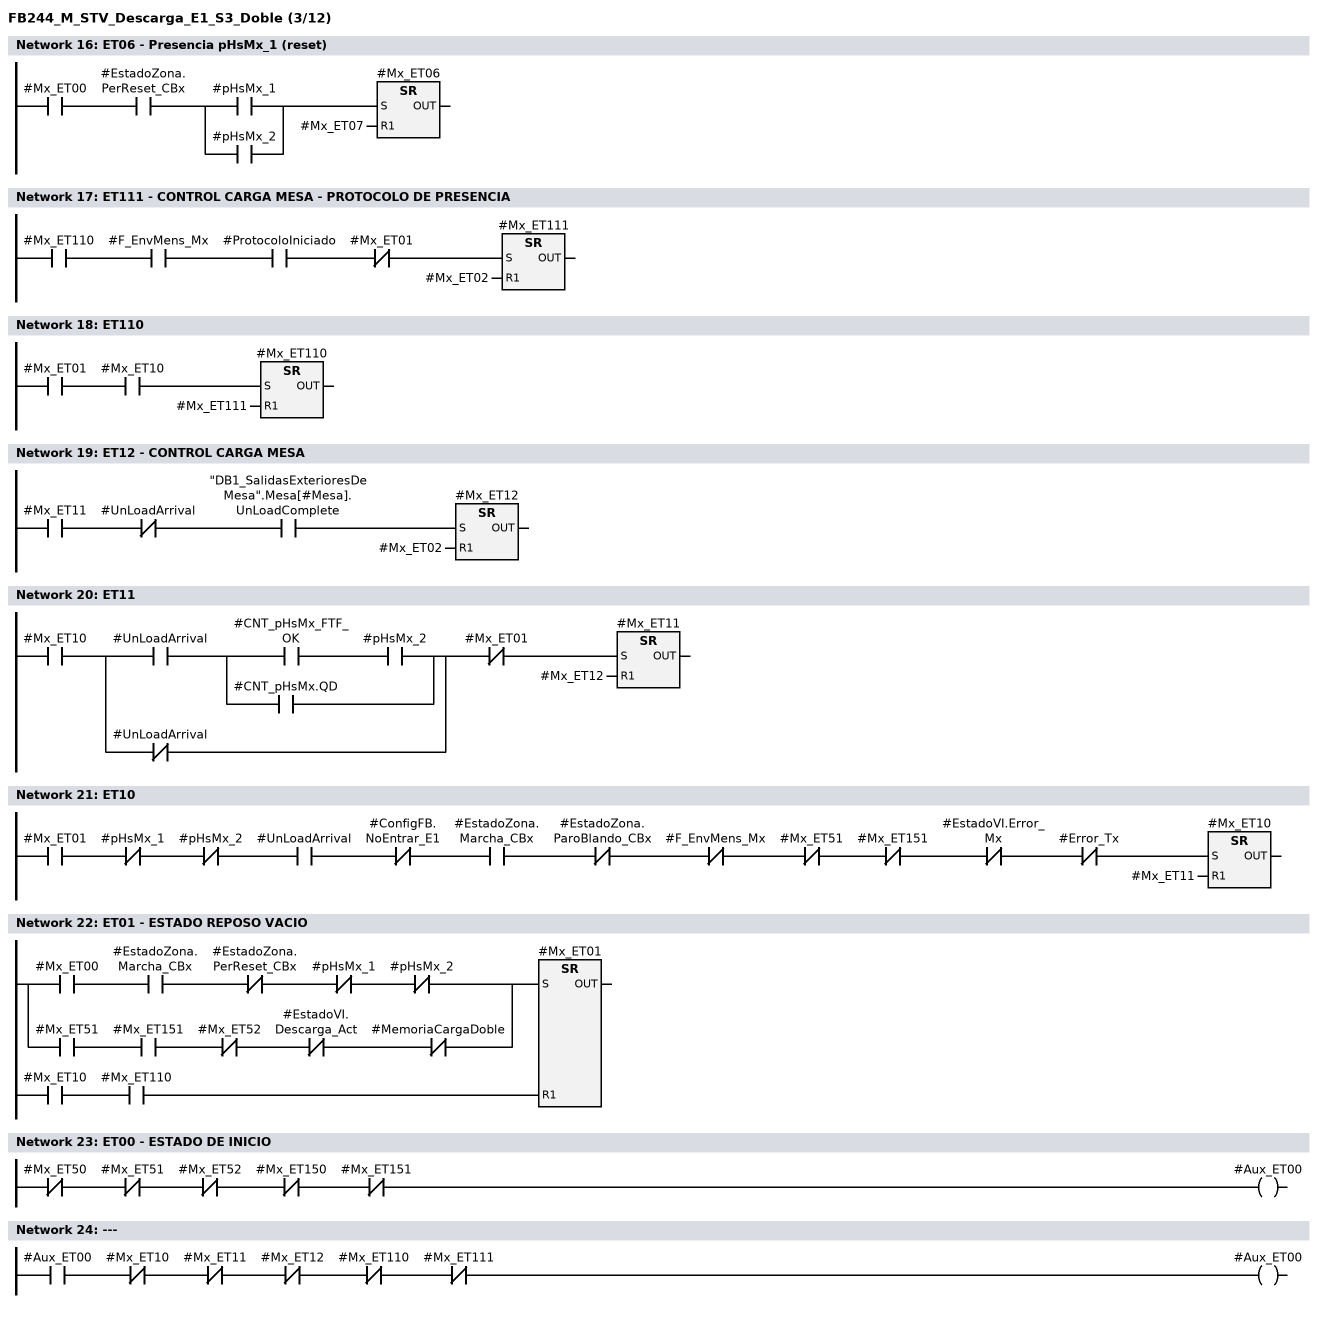
   RUNG wire#powerrail
      Contact( #Mx_ET00 )
      Contact( #EstadoZona.PerReset_CBx )
      wire#w1
      Contact( #pHsMx_1 )
      wire#w2
      S_SR(operand := #Mx_ET06, r1 := #Mx_ET07)
   END_RUNG
   RUNG wire#w1
      Contact( #pHsMx_2 )
   END_RUNG wire#w2
   // the same network as SCL:
   IF #Mx_ET00 AND #EstadoZona.PerReset_CBx AND (#pHsMx_1 OR #pHsMx_2) THEN
       #Mx_ET06 := TRUE;   // SR flip-flop
   END_IF;
   IF #Mx_ET07 THEN #Mx_ET06 := FALSE; END_IF;
END_REGION

REGION Network 17: ET111 - CONTROL CARGA MESA - PROTOCOLO DE PRESENCIA
   RUNG wire#powerrail
      Contact( #Mx_ET110 )
      Contact( #F_EnvMens_Mx )
      Contact( #ProtocoloIniciado )
      I_Contact( #Mx_ET01 )
      S_SR(operand := #Mx_ET111, r1 := #Mx_ET02)
   END_RUNG
   // the same network as SCL:
   IF #Mx_ET110 AND #F_EnvMens_Mx AND #ProtocoloIniciado AND NOT #Mx_ET01 THEN
       #Mx_ET111 := TRUE;   // SR flip-flop
   END_IF;
   IF #Mx_ET02 THEN #Mx_ET111 := FALSE; END_IF;
END_REGION

REGION Network 18: ET110
   RUNG wire#powerrail
      Contact( #Mx_ET01 )
      Contact( #Mx_ET10 )
      S_SR(operand := #Mx_ET110, r1 := #Mx_ET111)
   END_RUNG
   // the same network as SCL:
   IF #Mx_ET01 AND #Mx_ET10 THEN
       #Mx_ET110 := TRUE;   // SR flip-flop
   END_IF;
   IF #Mx_ET111 THEN #Mx_ET110 := FALSE; END_IF;
END_REGION

REGION Network 19: ET12 - CONTROL CARGA MESA
   RUNG wire#powerrail
      Contact( #Mx_ET11 )
      I_Contact( #UnLoadArrival )
      Contact( "DB1_SalidasExterioresDeMesa".Mesa[#Mesa].UnLoadComplete )
      S_SR(operand := #Mx_ET12, r1 := #Mx_ET02)
   END_RUNG
   // the same network as SCL:
   IF #Mx_ET11 AND NOT #UnLoadArrival AND "DB1_SalidasExterioresDeMesa".Mesa[#Mesa].UnLoadComplete THEN
       #Mx_ET12 := TRUE;   // SR flip-flop
   END_IF;
   IF #Mx_ET02 THEN #Mx_ET12 := FALSE; END_IF;
END_REGION

REGION Network 20: ET11
   RUNG wire#powerrail
      Contact( #Mx_ET10 )
      wire#w1
      Contact( #UnLoadArrival )
      wire#w2
      Contact( #CNT_pHsMx_FTF_OK )
      Contact( #pHsMx_2 )
      wire#w3
      I_Contact( #Mx_ET01 )
      S_SR(operand := #Mx_ET11, r1 := #Mx_ET12)
   END_RUNG
   RUNG wire#w2
      Contact( #CNT_pHsMx.QD )
   END_RUNG wire#w3
   RUNG wire#w1
      I_Contact( #UnLoadArrival )
   END_RUNG wire#w3
   // the same network as SCL:
   IF #Mx_ET10 AND ((#UnLoadArrival AND ((#CNT_pHsMx_FTF_OK AND #pHsMx_2) OR #CNT_pHsMx.QD)) OR NOT #UnLoadArrival) AND NOT #Mx_ET01 THEN
       #Mx_ET11 := TRUE;   // SR flip-flop
   END_IF;
   IF #Mx_ET12 THEN #Mx_ET11 := FALSE; END_IF;
END_REGION

REGION Network 21: ET10
   RUNG wire#powerrail
      Contact( #Mx_ET01 )
      I_Contact( #pHsMx_1 )
      I_Contact( #pHsMx_2 )
      Contact( #UnLoadArrival )
      I_Contact( #ConfigFB.NoEntrar_E1 )
      Contact( #EstadoZona.Marcha_CBx )
      I_Contact( #EstadoZona.ParoBlando_CBx )
      I_Contact( #F_EnvMens_Mx )
      I_Contact( #Mx_ET51 )
      I_Contact( #Mx_ET151 )
      I_Contact( #EstadoVI.Error_Mx )
      I_Contact( #Error_Tx )
      S_SR(operand := #Mx_ET10, r1 := #Mx_ET11)
   END_RUNG
   // the same network as SCL:
   IF #Mx_ET01 AND NOT #pHsMx_1 AND NOT #pHsMx_2 AND #UnLoadArrival AND NOT #ConfigFB.NoEntrar_E1 AND #EstadoZona.Marcha_CBx AND NOT #EstadoZona.ParoBlando_CBx AND NOT #F_EnvMens_Mx AND NOT #Mx_ET51 AND NOT #Mx_ET151 AND NOT #EstadoVI.Error_Mx AND NOT #Error_Tx THEN
       #Mx_ET10 := TRUE;   // SR flip-flop
   END_IF;
   IF #Mx_ET11 THEN #Mx_ET10 := FALSE; END_IF;
END_REGION

REGION Network 22: ET01 - ESTADO REPOSO VACIO
   RUNG wire#powerrail
      Contact( #Mx_ET00 )
      Contact( #EstadoZona.Marcha_CBx )
      I_Contact( #EstadoZona.PerReset_CBx )
      I_Contact( #pHsMx_1 )
      I_Contact( #pHsMx_2 )
      wire#w1
      S_SR(operand := #Mx_ET01, r1 := wire#w2)
   END_RUNG
   RUNG wire#powerrail
      Contact( #Mx_ET51 )
      Contact( #Mx_ET151 )
      I_Contact( #Mx_ET52 )
      I_Contact( #EstadoVI.Descarga_Act )
      I_Contact( #MemoriaCargaDoble )
   END_RUNG wire#w1
   RUNG wire#powerrail
      Contact( #Mx_ET10 )
      Contact( #Mx_ET110 )
   END_RUNG wire#w2
   // the same network as SCL:
   IF (#Mx_ET00 AND #EstadoZona.Marcha_CBx AND NOT #EstadoZona.PerReset_CBx AND NOT #pHsMx_1 AND NOT #pHsMx_2) OR (#Mx_ET51 AND #Mx_ET151 AND NOT #Mx_ET52 AND NOT #EstadoVI.Descarga_Act AND NOT #MemoriaCargaDoble) THEN
       #Mx_ET01 := TRUE;   // SR flip-flop
   END_IF;
   IF #Mx_ET10 AND #Mx_ET110 THEN #Mx_ET01 := FALSE; END_IF;
END_REGION

REGION Network 23: ET00 - ESTADO DE INICIO
   RUNG wire#powerrail
      I_Contact( #Mx_ET50 )
      I_Contact( #Mx_ET51 )
      I_Contact( #Mx_ET52 )
      I_Contact( #Mx_ET150 )
      I_Contact( #Mx_ET151 )
      Coil( #Aux_ET00 )
   END_RUNG
   // the same network as SCL:
   #Aux_ET00 := NOT #Mx_ET50 AND NOT #Mx_ET51 AND NOT #Mx_ET52 AND NOT #Mx_ET150 AND NOT #Mx_ET151;
END_REGION

REGION Network 24: ---
   RUNG wire#powerrail
      Contact( #Aux_ET00 )
      I_Contact( #Mx_ET10 )
      I_Contact( #Mx_ET11 )
      I_Contact( #Mx_ET12 )
      I_Contact( #Mx_ET110 )
      I_Contact( #Mx_ET111 )
      Coil( #Aux_ET00 )
   END_RUNG
   // the same network as SCL:
   #Aux_ET00 := #Aux_ET00 AND NOT #Mx_ET10 AND NOT #Mx_ET11 AND NOT #Mx_ET12 AND NOT #Mx_ET110 AND NOT #Mx_ET111;
END_REGION

REGION Network 25: ---
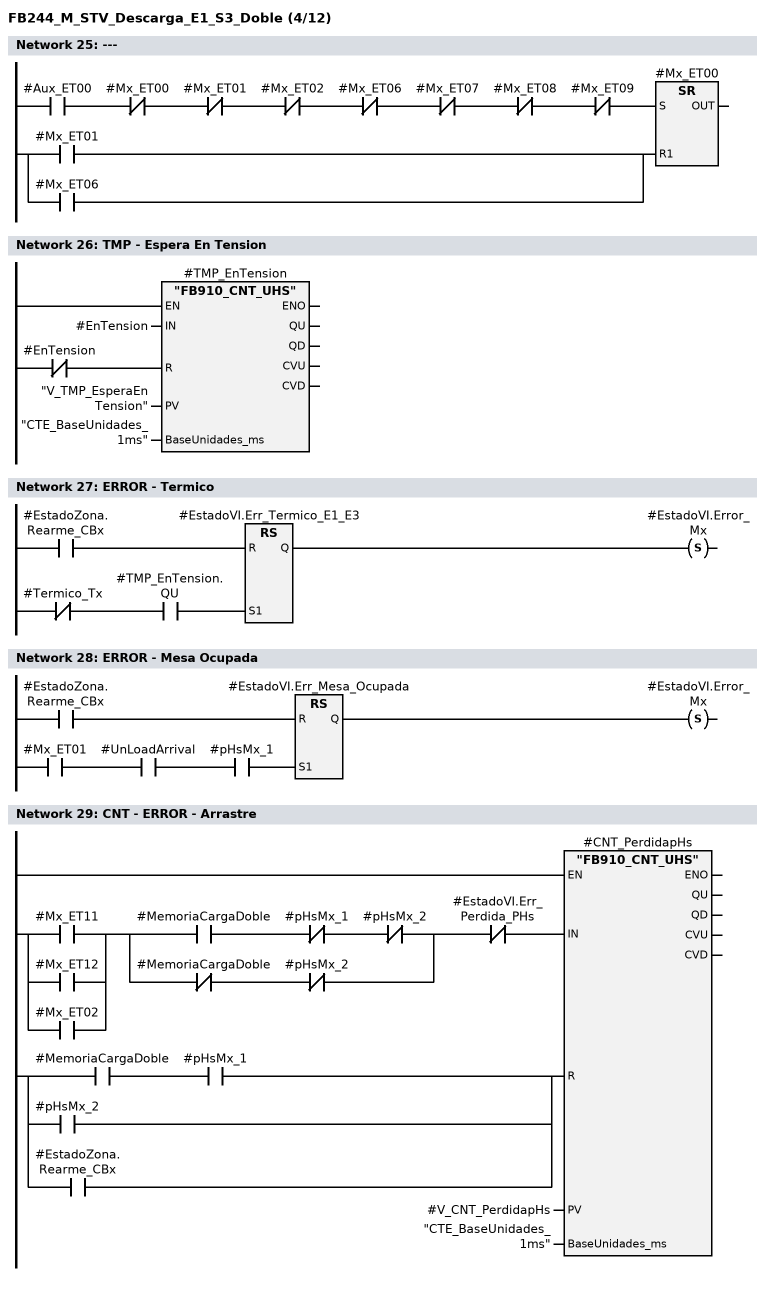
   RUNG wire#powerrail
      Contact( #Aux_ET00 )
      I_Contact( #Mx_ET00 )
      I_Contact( #Mx_ET01 )
      I_Contact( #Mx_ET02 )
      I_Contact( #Mx_ET06 )
      I_Contact( #Mx_ET07 )
      I_Contact( #Mx_ET08 )
      I_Contact( #Mx_ET09 )
      S_SR(operand := #Mx_ET00, r1 := wire#w1)
   END_RUNG
   RUNG wire#powerrail
      Contact( #Mx_ET01 )
   END_RUNG wire#w1
   RUNG wire#powerrail
      Contact( #Mx_ET06 )
   END_RUNG wire#w1
   // the same network as SCL:
   IF #Aux_ET00 AND NOT #Mx_ET00 AND NOT #Mx_ET01 AND NOT #Mx_ET02 AND NOT #Mx_ET06 AND NOT #Mx_ET07 AND NOT #Mx_ET08 AND NOT #Mx_ET09 THEN
       #Mx_ET00 := TRUE;   // SR flip-flop
   END_IF;
   IF #Mx_ET01 OR #Mx_ET06 THEN #Mx_ET00 := FALSE; END_IF;
END_REGION

REGION Network 26: TMP - Espera En Tension
   RUNG wire#powerrail
      #TMP_EnTension(R := wire#w1, IN := #EnTension, PV := "V_TMP_EsperaEnTension", BaseUnidades_ms := "CTE_BaseUnidades_1ms", QU =>, QD =>, CVU =>, CVD =>)
   END_RUNG
   RUNG wire#powerrail
      I_Contact( #EnTension )
   END_RUNG wire#w1
   // the same network as SCL:
   #TMP_EnTension(IN := #EnTension,   // "FB910_CNT_UHS"
                  R := NOT #EnTension,
                  PV := "V_TMP_EsperaEnTension",
                  BaseUnidades_ms := "CTE_BaseUnidades_1ms");
END_REGION

REGION Network 27: ERROR - Termico
   RUNG wire#powerrail
      Contact( #EstadoZona.Rearme_CBx )
      S_RS(operand := #EstadoVI.Err_Termico_E1_E3, s1 := wire#w1)
      S_Coil( #EstadoVI.Error_Mx )
   END_RUNG
   RUNG wire#powerrail
      I_Contact( #Termico_Tx )
      Contact( #TMP_EnTension.QU )
   END_RUNG wire#w1
   // the same network as SCL:
   IF #EstadoZona.Rearme_CBx THEN
       #EstadoVI.Err_Termico_E1_E3 := FALSE;   // RS flip-flop
   END_IF;
   IF NOT #Termico_Tx AND #TMP_EnTension.QU THEN #EstadoVI.Err_Termico_E1_E3 := TRUE; END_IF;
   IF #EstadoVI.Err_Termico_E1_E3 THEN #EstadoVI.Error_Mx := TRUE; END_IF;
END_REGION

REGION Network 28: ERROR - Mesa Ocupada
   RUNG wire#powerrail
      Contact( #EstadoZona.Rearme_CBx )
      S_RS(operand := #EstadoVI.Err_Mesa_Ocupada, s1 := wire#w1)
      S_Coil( #EstadoVI.Error_Mx )
   END_RUNG
   RUNG wire#powerrail
      Contact( #Mx_ET01 )
      Contact( #UnLoadArrival )
      Contact( #pHsMx_1 )
   END_RUNG wire#w1
   // the same network as SCL:
   IF #EstadoZona.Rearme_CBx THEN
       #EstadoVI.Err_Mesa_Ocupada := FALSE;   // RS flip-flop
   END_IF;
   IF #Mx_ET01 AND #UnLoadArrival AND #pHsMx_1 THEN #EstadoVI.Err_Mesa_Ocupada := TRUE; END_IF;
   IF #EstadoVI.Err_Mesa_Ocupada THEN #EstadoVI.Error_Mx := TRUE; END_IF;
END_REGION

REGION Network 29: CNT - ERROR - Arrastre
   RUNG wire#powerrail
      #CNT_PerdidapHs(IN := wire#w3, R := wire#w4, PV := #V_CNT_PerdidapHs, BaseUnidades_ms := "CTE_BaseUnidades_1ms", QU =>, QD =>, CVU =>, CVD =>)
   END_RUNG
   RUNG wire#powerrail
      Contact( #Mx_ET11 )
      wire#w1
      Contact( #MemoriaCargaDoble )
      I_Contact( #pHsMx_1 )
      I_Contact( #pHsMx_2 )
      wire#w2
      I_Contact( #EstadoVI.Err_Perdida_PHs )
   END_RUNG wire#w3
   RUNG wire#powerrail
      Contact( #Mx_ET12 )
   END_RUNG wire#w1
   RUNG wire#powerrail
      Contact( #Mx_ET02 )
   END_RUNG wire#w1
   RUNG wire#w1
      I_Contact( #MemoriaCargaDoble )
      I_Contact( #pHsMx_2 )
   END_RUNG wire#w2
   RUNG wire#powerrail
      Contact( #MemoriaCargaDoble )
      Contact( #pHsMx_1 )
   END_RUNG wire#w4
   RUNG wire#powerrail
      Contact( #pHsMx_2 )
   END_RUNG wire#w4
   RUNG wire#powerrail
      Contact( #EstadoZona.Rearme_CBx )
   END_RUNG wire#w4
   // the same network as SCL:
   #CNT_PerdidapHs(IN := (#Mx_ET11 OR #Mx_ET12 OR #Mx_ET02) AND ((#MemoriaCargaDoble AND NOT #pHsMx_1 AND NOT #pHsMx_2) OR (NOT #MemoriaCargaDoble AND NOT #pHsMx_2)) AND NOT #EstadoVI.Err_Perdida_PHs,   // "FB910_CNT_UHS"
                   R := (#MemoriaCargaDoble AND #pHsMx_1) OR #pHsMx_2 OR #EstadoZona.Rearme_CBx,
                   PV := #V_CNT_PerdidapHs,
                   BaseUnidades_ms := "CTE_BaseUnidades_1ms");
END_REGION

REGION Network 30: ERROR - Arrastre
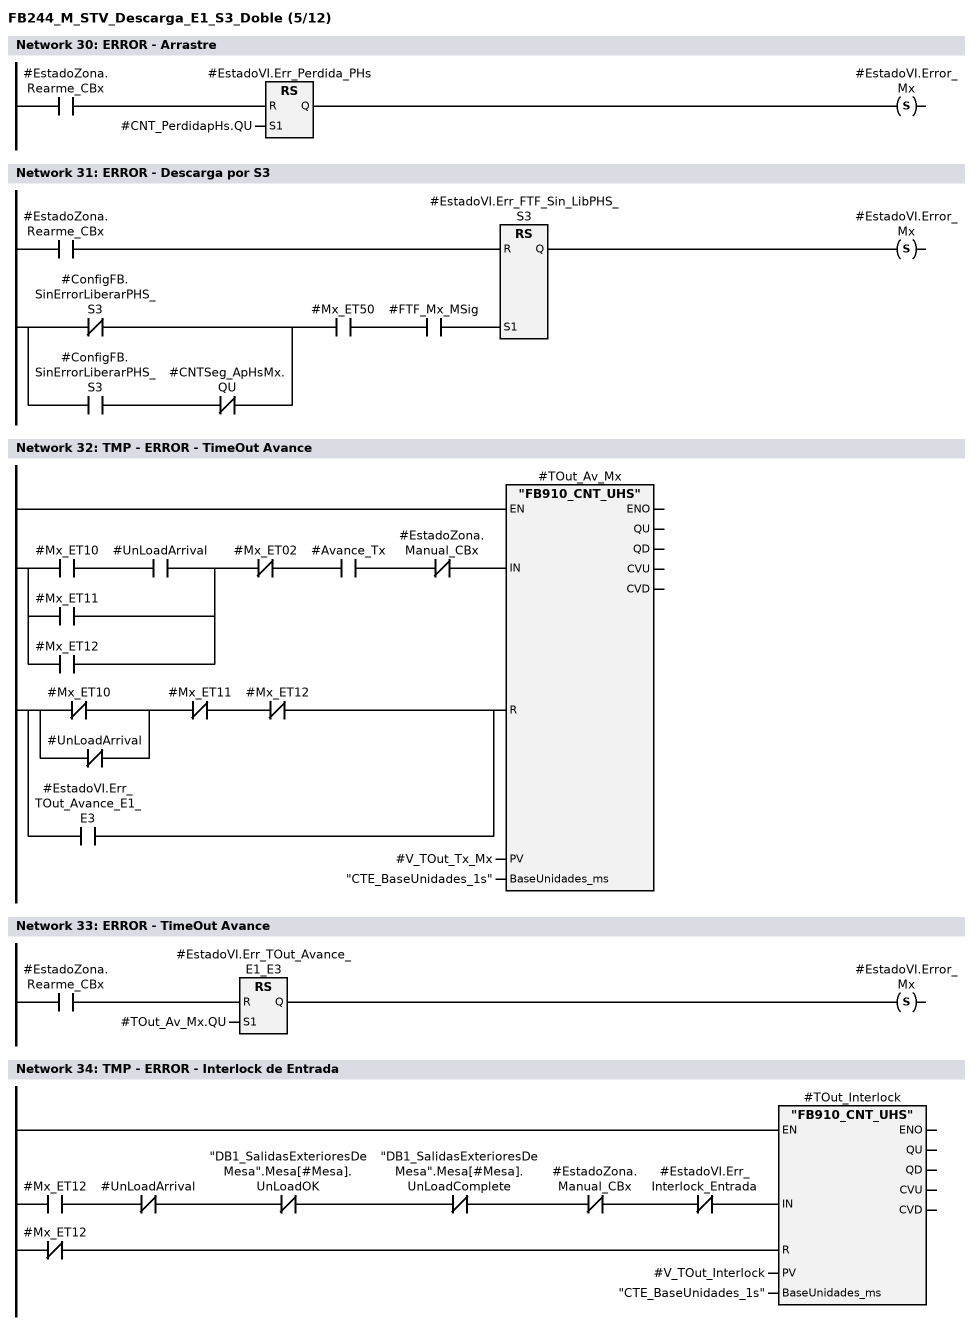
   RUNG wire#powerrail
      Contact( #EstadoZona.Rearme_CBx )
      S_RS(operand := #EstadoVI.Err_Perdida_PHs, s1 := #CNT_PerdidapHs.QU)
      S_Coil( #EstadoVI.Error_Mx )
   END_RUNG
   // the same network as SCL:
   IF #EstadoZona.Rearme_CBx THEN
       #EstadoVI.Err_Perdida_PHs := FALSE;   // RS flip-flop
   END_IF;
   IF #CNT_PerdidapHs.QU THEN #EstadoVI.Err_Perdida_PHs := TRUE; END_IF;
   IF #EstadoVI.Err_Perdida_PHs THEN #EstadoVI.Error_Mx := TRUE; END_IF;
END_REGION

REGION Network 31: ERROR - Descarga por S3
   RUNG wire#powerrail
      Contact( #EstadoZona.Rearme_CBx )
      S_RS(operand := #EstadoVI.Err_FTF_Sin_LibPHS_S3, s1 := wire#w2)
      S_Coil( #EstadoVI.Error_Mx )
   END_RUNG
   RUNG wire#powerrail
      I_Contact( #ConfigFB.SinErrorLiberarPHS_S3 )
      wire#w1
      Contact( #Mx_ET50 )
      Contact( #FTF_Mx_MSig )
   END_RUNG wire#w2
   RUNG wire#powerrail
      Contact( #ConfigFB.SinErrorLiberarPHS_S3 )
      I_Contact( #CNTSeg_ApHsMx.QU )
   END_RUNG wire#w1
   // the same network as SCL:
   IF #EstadoZona.Rearme_CBx THEN
       #EstadoVI.Err_FTF_Sin_LibPHS_S3 := FALSE;   // RS flip-flop
   END_IF;
   IF (NOT #ConfigFB.SinErrorLiberarPHS_S3 OR (#ConfigFB.SinErrorLiberarPHS_S3 AND NOT #CNTSeg_ApHsMx.QU)) AND #Mx_ET50 AND #FTF_Mx_MSig THEN
       #EstadoVI.Err_FTF_Sin_LibPHS_S3 := TRUE;
   END_IF;
   IF #EstadoVI.Err_FTF_Sin_LibPHS_S3 THEN #EstadoVI.Error_Mx := TRUE; END_IF;
END_REGION

REGION Network 32: TMP - ERROR - TimeOut Avance
   RUNG wire#powerrail
      #TOut_Av_Mx(IN := wire#w2, R := wire#w4, PV := #V_TOut_Tx_Mx, BaseUnidades_ms := "CTE_BaseUnidades_1s", QU =>, QD =>, CVU =>, CVD =>)
   END_RUNG
   RUNG wire#powerrail
      Contact( #Mx_ET10 )
      Contact( #UnLoadArrival )
      wire#w1
      I_Contact( #Mx_ET02 )
      Contact( #Avance_Tx )
      I_Contact( #EstadoZona.Manual_CBx )
   END_RUNG wire#w2
   RUNG wire#powerrail
      Contact( #Mx_ET11 )
   END_RUNG wire#w1
   RUNG wire#powerrail
      Contact( #Mx_ET12 )
   END_RUNG wire#w1
   RUNG wire#powerrail
      I_Contact( #Mx_ET10 )
      wire#w3
      I_Contact( #Mx_ET11 )
      I_Contact( #Mx_ET12 )
   END_RUNG wire#w4
   RUNG wire#powerrail
      I_Contact( #UnLoadArrival )
   END_RUNG wire#w3
   RUNG wire#powerrail
      Contact( #EstadoVI.Err_TOut_Avance_E1_E3 )
   END_RUNG wire#w4
   // the same network as SCL:
   #TOut_Av_Mx(IN := ((#Mx_ET10 AND #UnLoadArrival) OR #Mx_ET11 OR #Mx_ET12) AND NOT #Mx_ET02 AND #Avance_Tx AND NOT #EstadoZona.Manual_CBx,   // "FB910_CNT_UHS"
               R := ((NOT #Mx_ET10 OR NOT #UnLoadArrival) AND NOT #Mx_ET11 AND NOT #Mx_ET12) OR #EstadoVI.Err_TOut_Avance_E1_E3,
               PV := #V_TOut_Tx_Mx,
               BaseUnidades_ms := "CTE_BaseUnidades_1s");
END_REGION

REGION Network 33: ERROR - TimeOut Avance
   RUNG wire#powerrail
      Contact( #EstadoZona.Rearme_CBx )
      S_RS(operand := #EstadoVI.Err_TOut_Avance_E1_E3, s1 := #TOut_Av_Mx.QU)
      S_Coil( #EstadoVI.Error_Mx )
   END_RUNG
   // the same network as SCL:
   IF #EstadoZona.Rearme_CBx THEN
       #EstadoVI.Err_TOut_Avance_E1_E3 := FALSE;   // RS flip-flop
   END_IF;
   IF #TOut_Av_Mx.QU THEN #EstadoVI.Err_TOut_Avance_E1_E3 := TRUE; END_IF;
   IF #EstadoVI.Err_TOut_Avance_E1_E3 THEN #EstadoVI.Error_Mx := TRUE; END_IF;
END_REGION

REGION Network 34: TMP - ERROR - Interlock de Entrada
   RUNG wire#powerrail
      #TOut_Interlock(IN := wire#w1, R := wire#w2, PV := #V_TOut_Interlock, BaseUnidades_ms := "CTE_BaseUnidades_1s", QU =>, QD =>, CVU =>, CVD =>)
   END_RUNG
   RUNG wire#powerrail
      Contact( #Mx_ET12 )
      I_Contact( #UnLoadArrival )
      I_Contact( "DB1_SalidasExterioresDeMesa".Mesa[#Mesa].UnLoadOK )
      I_Contact( "DB1_SalidasExterioresDeMesa".Mesa[#Mesa].UnLoadComplete )
      I_Contact( #EstadoZona.Manual_CBx )
      I_Contact( #EstadoVI.Err_Interlock_Entrada )
   END_RUNG wire#w1
   RUNG wire#powerrail
      I_Contact( #Mx_ET12 )
   END_RUNG wire#w2
   // the same network as SCL:
   #TOut_Interlock(IN := #Mx_ET12 AND NOT #UnLoadArrival AND NOT "DB1_SalidasExterioresDeMesa".Mesa[#Mesa].UnLoadOK AND NOT "DB1_SalidasExterioresDeMesa".Mesa[#Mesa].UnLoadComplete AND NOT #EstadoZona.Manual_CBx AND NOT #EstadoVI.Err_Interlock_Entrada,   // "FB910_CNT_UHS"
                   R := NOT #Mx_ET12,
                   PV := #V_TOut_Interlock,
                   BaseUnidades_ms := "CTE_BaseUnidades_1s");
END_REGION

REGION Network 35: ERROR - Interlock de Entrada
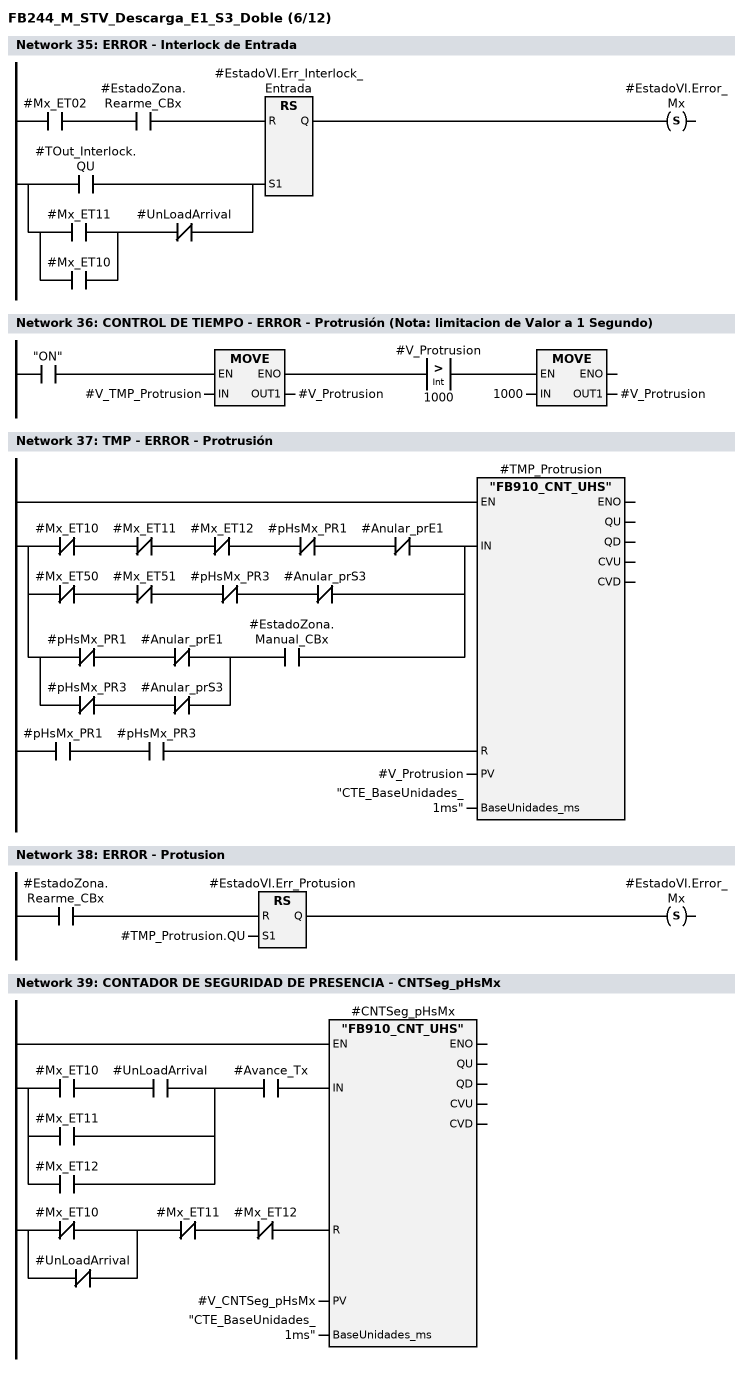
   RUNG wire#powerrail
      Contact( #Mx_ET02 )
      Contact( #EstadoZona.Rearme_CBx )
      S_RS(operand := #EstadoVI.Err_Interlock_Entrada, s1 := wire#w2)
      S_Coil( #EstadoVI.Error_Mx )
   END_RUNG
   RUNG wire#powerrail
      Contact( #TOut_Interlock.QU )
   END_RUNG wire#w2
   RUNG wire#powerrail
      Contact( #Mx_ET11 )
      wire#w1
      I_Contact( #UnLoadArrival )
   END_RUNG wire#w2
   RUNG wire#powerrail
      Contact( #Mx_ET10 )
   END_RUNG wire#w1
   // the same network as SCL:
   IF #Mx_ET02 AND #EstadoZona.Rearme_CBx THEN
       #EstadoVI.Err_Interlock_Entrada := FALSE;   // RS flip-flop
   END_IF;
   IF #TOut_Interlock.QU OR ((#Mx_ET11 OR #Mx_ET10) AND NOT #UnLoadArrival) THEN
       #EstadoVI.Err_Interlock_Entrada := TRUE;
   END_IF;
   IF #EstadoVI.Err_Interlock_Entrada THEN #EstadoVI.Error_Mx := TRUE; END_IF;
END_REGION

REGION Network 36: CONTROL DE TIEMPO - ERROR - Protrusión (Nota: limitacion de Valor a 1 Segundo)
   RUNG wire#powerrail
      Contact( "ON" )
      Move(in := #V_TMP_Protrusion, out1 => #V_Protrusion)
      { S7_Templates := "SrcType := Int" } GT_Contact(in1 := #V_Protrusion, in2 := 1000)
      Move(in := 1000, out1 => #V_Protrusion)
   END_RUNG
   // the same network as SCL:
   IF "ON" THEN #V_Protrusion := #V_TMP_Protrusion; END_IF;
   IF "ON" AND (#V_Protrusion > 1000) THEN #V_Protrusion := 1000; END_IF;
END_REGION

REGION Network 37: TMP - ERROR - Protrusión
   RUNG wire#powerrail
      #TMP_Protrusion(IN := wire#w2, R := wire#w3, PV := #V_Protrusion, BaseUnidades_ms := "CTE_BaseUnidades_1ms", QU =>, QD =>, CVU =>, CVD =>)
   END_RUNG
   RUNG wire#powerrail
      I_Contact( #Mx_ET10 )
      I_Contact( #Mx_ET11 )
      I_Contact( #Mx_ET12 )
      I_Contact( #pHsMx_PR1 )
      I_Contact( #Anular_prE1 )
   END_RUNG wire#w2
   RUNG wire#powerrail
      I_Contact( #Mx_ET50 )
      I_Contact( #Mx_ET51 )
      I_Contact( #pHsMx_PR3 )
      I_Contact( #Anular_prS3 )
   END_RUNG wire#w2
   RUNG wire#powerrail
      I_Contact( #pHsMx_PR1 )
      I_Contact( #Anular_prE1 )
      wire#w1
      Contact( #EstadoZona.Manual_CBx )
   END_RUNG wire#w2
   RUNG wire#powerrail
      I_Contact( #pHsMx_PR3 )
      I_Contact( #Anular_prS3 )
   END_RUNG wire#w1
   RUNG wire#powerrail
      Contact( #pHsMx_PR1 )
      Contact( #pHsMx_PR3 )
   END_RUNG wire#w3
   // the same network as SCL:
   #TMP_Protrusion(IN := (NOT #Mx_ET10 AND NOT #Mx_ET11 AND NOT #Mx_ET12 AND NOT #pHsMx_PR1 AND NOT #Anular_prE1) OR (NOT #Mx_ET50 AND NOT #Mx_ET51 AND NOT #pHsMx_PR3 AND NOT #Anular_prS3) OR (((NOT #pHsMx_PR1 AND NOT #Anular_prE1) OR (NOT #pHsMx_PR3 AND NOT #Anular_prS3)) AND #EstadoZona.Manual_CBx),   // "FB910_CNT_UHS"
                   R := #pHsMx_PR1 AND #pHsMx_PR3,
                   PV := #V_Protrusion,
                   BaseUnidades_ms := "CTE_BaseUnidades_1ms");
END_REGION

REGION Network 38: ERROR - Protusion
   RUNG wire#powerrail
      Contact( #EstadoZona.Rearme_CBx )
      S_RS(operand := #EstadoVI.Err_Protusion, s1 := #TMP_Protrusion.QU)
      S_Coil( #EstadoVI.Error_Mx )
   END_RUNG
   // the same network as SCL:
   IF #EstadoZona.Rearme_CBx THEN
       #EstadoVI.Err_Protusion := FALSE;   // RS flip-flop
   END_IF;
   IF #TMP_Protrusion.QU THEN #EstadoVI.Err_Protusion := TRUE; END_IF;
   IF #EstadoVI.Err_Protusion THEN #EstadoVI.Error_Mx := TRUE; END_IF;
END_REGION

REGION Network 39: CONTADOR DE SEGURIDAD DE PRESENCIA - CNTSeg_pHsMx
   RUNG wire#powerrail
      #CNTSeg_pHsMx(IN := wire#w2, R := wire#w4, PV := #V_CNTSeg_pHsMx, BaseUnidades_ms := "CTE_BaseUnidades_1ms", QU =>, QD =>, CVU =>, CVD =>)
   END_RUNG
   RUNG wire#powerrail
      Contact( #Mx_ET10 )
      Contact( #UnLoadArrival )
      wire#w1
      Contact( #Avance_Tx )
   END_RUNG wire#w2
   RUNG wire#powerrail
      Contact( #Mx_ET11 )
   END_RUNG wire#w1
   RUNG wire#powerrail
      Contact( #Mx_ET12 )
   END_RUNG wire#w1
   RUNG wire#powerrail
      I_Contact( #Mx_ET10 )
      wire#w3
      I_Contact( #Mx_ET11 )
      I_Contact( #Mx_ET12 )
   END_RUNG wire#w4
   RUNG wire#powerrail
      I_Contact( #UnLoadArrival )
   END_RUNG wire#w3
   // the same network as SCL:
   #CNTSeg_pHsMx(IN := ((#Mx_ET10 AND #UnLoadArrival) OR #Mx_ET11 OR #Mx_ET12) AND #Avance_Tx,   // "FB910_CNT_UHS"
                 R := (NOT #Mx_ET10 OR NOT #UnLoadArrival) AND NOT #Mx_ET11 AND NOT #Mx_ET12,
                 PV := #V_CNTSeg_pHsMx,
                 BaseUnidades_ms := "CTE_BaseUnidades_1ms");
END_REGION

REGION Network 40: CONTADOR DE PRESENCIA - CNT_pHsMx
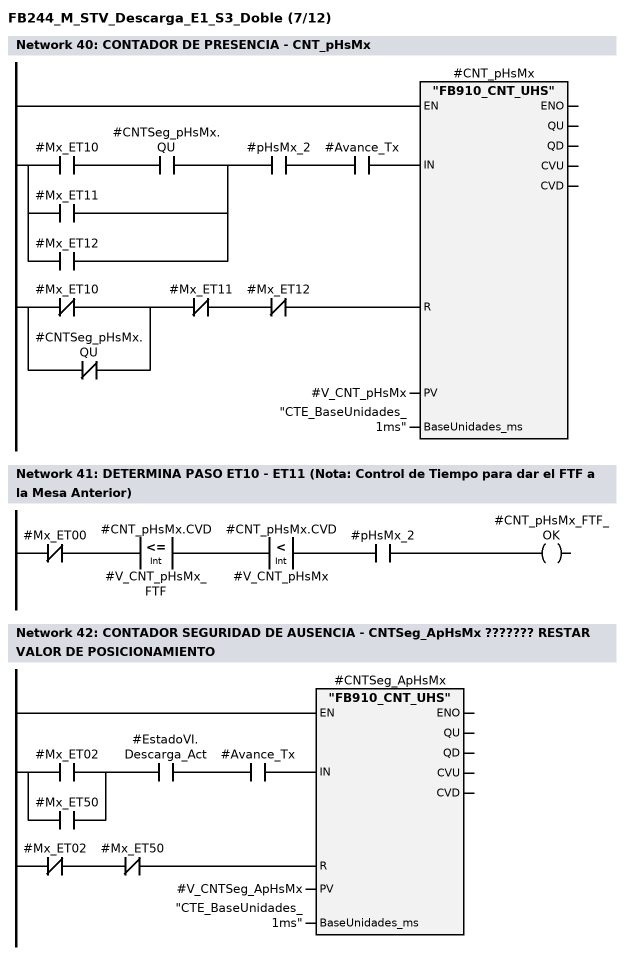
   RUNG wire#powerrail
      #CNT_pHsMx(IN := wire#w2, R := wire#w4, PV := #V_CNT_pHsMx, BaseUnidades_ms := "CTE_BaseUnidades_1ms", QU =>, QD =>, CVU =>, CVD =>)
   END_RUNG
   RUNG wire#powerrail
      Contact( #Mx_ET10 )
      Contact( #CNTSeg_pHsMx.QU )
      wire#w1
      Contact( #pHsMx_2 )
      Contact( #Avance_Tx )
   END_RUNG wire#w2
   RUNG wire#powerrail
      Contact( #Mx_ET11 )
   END_RUNG wire#w1
   RUNG wire#powerrail
      Contact( #Mx_ET12 )
   END_RUNG wire#w1
   RUNG wire#powerrail
      I_Contact( #Mx_ET10 )
      wire#w3
      I_Contact( #Mx_ET11 )
      I_Contact( #Mx_ET12 )
   END_RUNG wire#w4
   RUNG wire#powerrail
      I_Contact( #CNTSeg_pHsMx.QU )
   END_RUNG wire#w3
   // the same network as SCL:
   #CNT_pHsMx(IN := ((#Mx_ET10 AND #CNTSeg_pHsMx.QU) OR #Mx_ET11 OR #Mx_ET12) AND #pHsMx_2 AND #Avance_Tx,   // "FB910_CNT_UHS"
              R := (NOT #Mx_ET10 OR NOT #CNTSeg_pHsMx.QU) AND NOT #Mx_ET11 AND NOT #Mx_ET12,
              PV := #V_CNT_pHsMx,
              BaseUnidades_ms := "CTE_BaseUnidades_1ms");
END_REGION

REGION Network 41: DETERMINA PASO ET10 - ET11 (Nota: Control de Tiempo para dar el FTF a la Mesa Anterior)
   RUNG wire#powerrail
      I_Contact( #Mx_ET00 )
      { S7_Templates := "SrcType := Int" } LE_Contact(in1 := #CNT_pHsMx.CVD, in2 := #V_CNT_pHsMx_FTF)
      { S7_Templates := "SrcType := Int" } LT_Contact(in1 := #CNT_pHsMx.CVD, in2 := #V_CNT_pHsMx)
      Contact( #pHsMx_2 )
      Coil( #CNT_pHsMx_FTF_OK )
   END_RUNG
   // the same network as SCL:
   #CNT_pHsMx_FTF_OK := NOT #Mx_ET00 AND (#CNT_pHsMx.CVD <= #V_CNT_pHsMx_FTF) AND (#CNT_pHsMx.CVD < #V_CNT_pHsMx) AND #pHsMx_2;
END_REGION

REGION Network 42: CONTADOR SEGURIDAD DE AUSENCIA - CNTSeg_ApHsMx ??????? RESTAR VALOR DE POSICIONAMIENTO
   RUNG wire#powerrail
      #CNTSeg_ApHsMx(IN := wire#w2, R := wire#w3, PV := #V_CNTSeg_ApHsMx, BaseUnidades_ms := "CTE_BaseUnidades_1ms", QU =>, QD =>, CVU =>, CVD =>)
   END_RUNG
   RUNG wire#powerrail
      Contact( #Mx_ET02 )
      wire#w1
      Contact( #EstadoVI.Descarga_Act )
      Contact( #Avance_Tx )
   END_RUNG wire#w2
   RUNG wire#powerrail
      Contact( #Mx_ET50 )
   END_RUNG wire#w1
   RUNG wire#powerrail
      I_Contact( #Mx_ET02 )
      I_Contact( #Mx_ET50 )
   END_RUNG wire#w3
   // the same network as SCL:
   #CNTSeg_ApHsMx(IN := (#Mx_ET02 OR #Mx_ET50) AND #EstadoVI.Descarga_Act AND #Avance_Tx,   // "FB910_CNT_UHS"
                  R := NOT #Mx_ET02 AND NOT #Mx_ET50,
                  PV := #V_CNTSeg_ApHsMx,
                  BaseUnidades_ms := "CTE_BaseUnidades_1ms");
END_REGION

REGION Network 43: CONTADOR DE LA AUSENCIA - CNT_ApHsMX
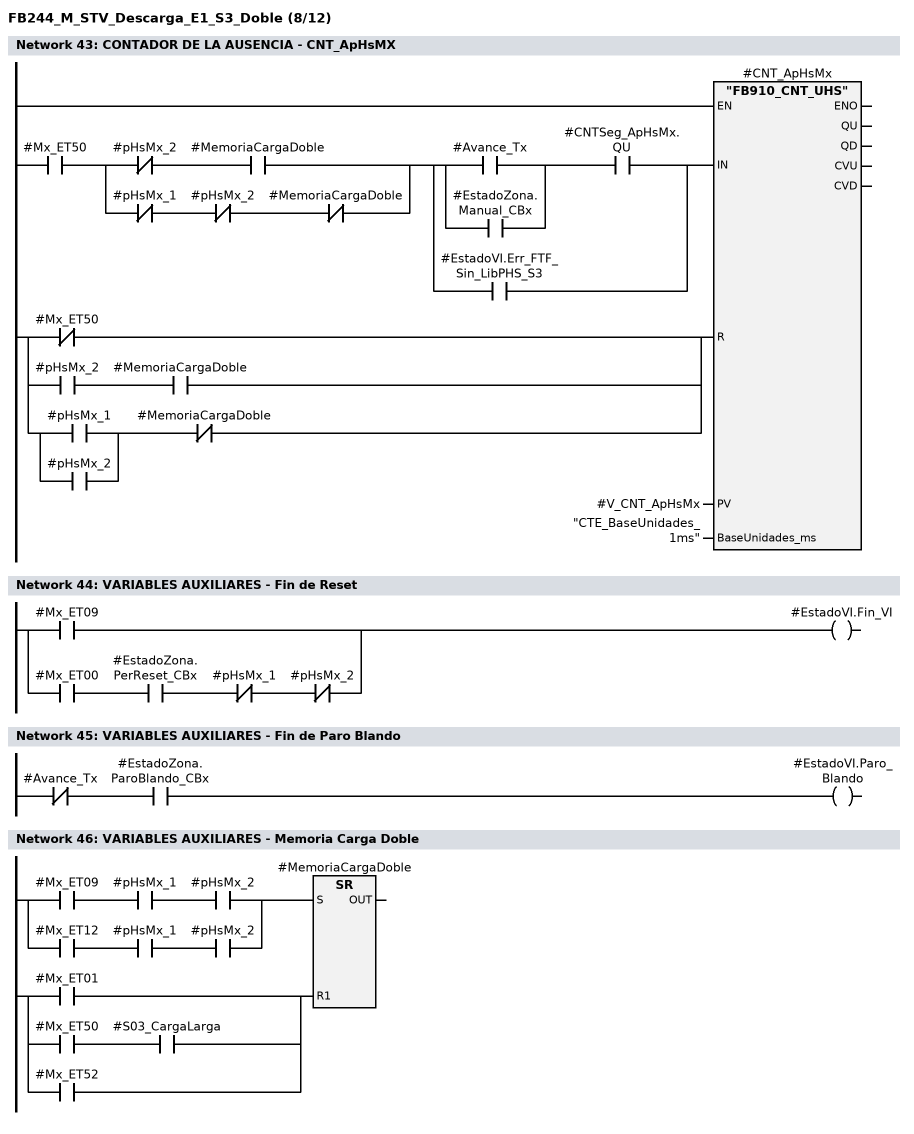
   RUNG wire#powerrail
      #CNT_ApHsMx(IN := wire#w4, R := wire#w6, PV := #V_CNT_ApHsMx, BaseUnidades_ms := "CTE_BaseUnidades_1ms", QU =>, QD =>, CVU =>, CVD =>)
   END_RUNG
   RUNG wire#powerrail
      Contact( #Mx_ET50 )
      wire#w1
      I_Contact( #pHsMx_2 )
      Contact( #MemoriaCargaDoble )
      wire#w2
      Contact( #Avance_Tx )
      wire#w3
      Contact( #CNTSeg_ApHsMx.QU )
   END_RUNG wire#w4
   RUNG wire#w1
      I_Contact( #pHsMx_1 )
      I_Contact( #pHsMx_2 )
      I_Contact( #MemoriaCargaDoble )
   END_RUNG wire#w2
   RUNG wire#w2
      Contact( #EstadoZona.Manual_CBx )
   END_RUNG wire#w3
   RUNG wire#w2
      Contact( #EstadoVI.Err_FTF_Sin_LibPHS_S3 )
   END_RUNG wire#w4
   RUNG wire#powerrail
      I_Contact( #Mx_ET50 )
   END_RUNG wire#w6
   RUNG wire#powerrail
      Contact( #pHsMx_2 )
      Contact( #MemoriaCargaDoble )
   END_RUNG wire#w6
   RUNG wire#powerrail
      Contact( #pHsMx_1 )
      wire#w5
      I_Contact( #MemoriaCargaDoble )
   END_RUNG wire#w6
   RUNG wire#powerrail
      Contact( #pHsMx_2 )
   END_RUNG wire#w5
   // the same network as SCL:
   #CNT_ApHsMx(IN := #Mx_ET50 AND ((NOT #pHsMx_2 AND #MemoriaCargaDoble) OR (NOT #pHsMx_1 AND NOT #pHsMx_2 AND NOT #MemoriaCargaDoble)) AND (((#Avance_Tx OR #EstadoZona.Manual_CBx) AND #CNTSeg_ApHsMx.QU) OR #EstadoVI.Err_FTF_Sin_LibPHS_S3),   // "FB910_CNT_UHS"
               R := NOT #Mx_ET50 OR (#pHsMx_2 AND #MemoriaCargaDoble) OR ((#pHsMx_1 OR #pHsMx_2) AND NOT #MemoriaCargaDoble),
               PV := #V_CNT_ApHsMx,
               BaseUnidades_ms := "CTE_BaseUnidades_1ms");
END_REGION

REGION Network 44: VARIABLES AUXILIARES - Fin de Reset
   RUNG wire#powerrail
      Contact( #Mx_ET09 )
      wire#w1
      Coil( #EstadoVI.Fin_VI )
   END_RUNG
   RUNG wire#powerrail
      Contact( #Mx_ET00 )
      Contact( #EstadoZona.PerReset_CBx )
      I_Contact( #pHsMx_1 )
      I_Contact( #pHsMx_2 )
   END_RUNG wire#w1
   // the same network as SCL:
   #EstadoVI.Fin_VI := #Mx_ET09 OR (#Mx_ET00 AND #EstadoZona.PerReset_CBx AND NOT #pHsMx_1 AND NOT #pHsMx_2);
END_REGION

REGION Network 45: VARIABLES AUXILIARES - Fin de Paro Blando
   RUNG wire#powerrail
      I_Contact( #Avance_Tx )
      Contact( #EstadoZona.ParoBlando_CBx )
      Coil( #EstadoVI.Paro_Blando )
   END_RUNG
   // the same network as SCL:
   #EstadoVI.Paro_Blando := NOT #Avance_Tx AND #EstadoZona.ParoBlando_CBx;
END_REGION

REGION Network 46: VARIABLES AUXILIARES - Memoria Carga Doble
   RUNG wire#powerrail
      Contact( #Mx_ET09 )
      Contact( #pHsMx_1 )
      Contact( #pHsMx_2 )
      wire#w1
      S_SR(operand := #MemoriaCargaDoble, r1 := wire#w2)
   END_RUNG
   RUNG wire#powerrail
      Contact( #Mx_ET12 )
      Contact( #pHsMx_1 )
      Contact( #pHsMx_2 )
   END_RUNG wire#w1
   RUNG wire#powerrail
      Contact( #Mx_ET01 )
   END_RUNG wire#w2
   RUNG wire#powerrail
      Contact( #Mx_ET50 )
      Contact( #S03_CargaLarga )
   END_RUNG wire#w2
   RUNG wire#powerrail
      Contact( #Mx_ET52 )
   END_RUNG wire#w2
   // the same network as SCL:
   IF (#Mx_ET09 AND #pHsMx_1 AND #pHsMx_2) OR (#Mx_ET12 AND #pHsMx_1 AND #pHsMx_2) THEN
       #MemoriaCargaDoble := TRUE;   // SR flip-flop
   END_IF;
   IF #Mx_ET01 OR (#Mx_ET50 AND #S03_CargaLarga) OR #Mx_ET52 THEN #MemoriaCargaDoble := FALSE; END_IF;
END_REGION

REGION Network 47: VARIABLES AUXILIARES - Aviso de Salida - AVTF_Mx_MSig
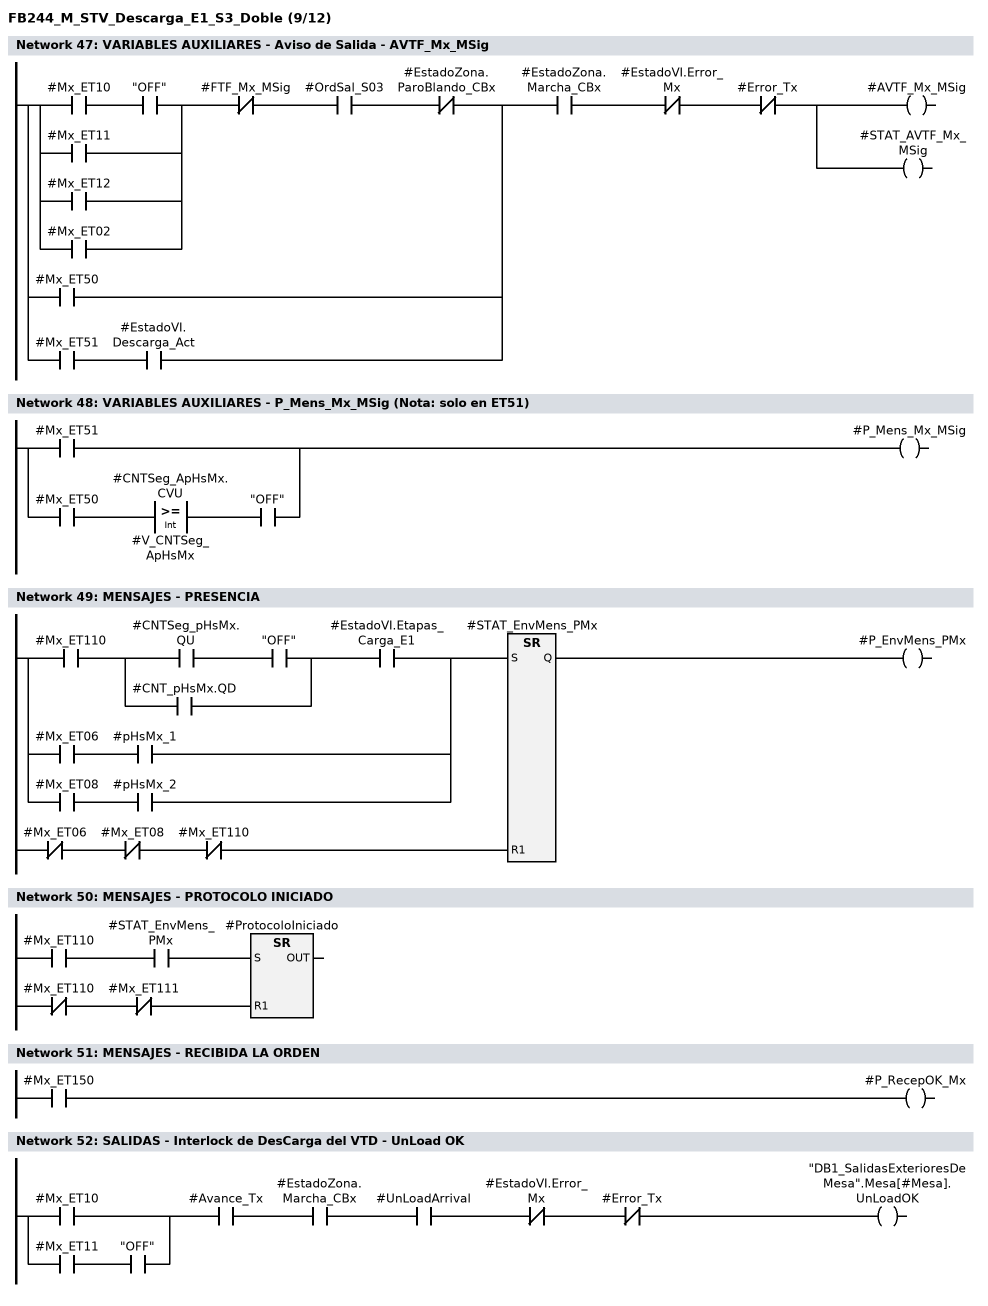
   RUNG wire#powerrail
      Contact( #Mx_ET10 )
      Contact( "OFF" )
      wire#w1
      I_Contact( #FTF_Mx_MSig )
      Contact( #OrdSal_S03 )
      I_Contact( #EstadoZona.ParoBlando_CBx )
      wire#w2
      Contact( #EstadoZona.Marcha_CBx )
      I_Contact( #EstadoVI.Error_Mx )
      I_Contact( #Error_Tx )
      wire#w3
      Coil( #AVTF_Mx_MSig )
   END_RUNG
   RUNG wire#powerrail
      Contact( #Mx_ET11 )
   END_RUNG wire#w1
   RUNG wire#powerrail
      Contact( #Mx_ET12 )
   END_RUNG wire#w1
   RUNG wire#powerrail
      Contact( #Mx_ET02 )
   END_RUNG wire#w1
   RUNG wire#powerrail
      Contact( #Mx_ET50 )
   END_RUNG wire#w2
   RUNG wire#powerrail
      Contact( #Mx_ET51 )
      Contact( #EstadoVI.Descarga_Act )
   END_RUNG wire#w2
   RUNG wire#w3
      Coil( #STAT_AVTF_Mx_MSig )
   END_RUNG
   // the same network as SCL:
   #AVTF_Mx_MSig := ((((#Mx_ET10 AND "OFF") OR #Mx_ET11 OR #Mx_ET12 OR #Mx_ET02) AND NOT #FTF_Mx_MSig AND #OrdSal_S03 AND NOT #EstadoZona.ParoBlando_CBx) OR #Mx_ET50 OR (#Mx_ET51 AND #EstadoVI.Descarga_Act)) AND #EstadoZona.Marcha_CBx AND NOT #EstadoVI.Error_Mx AND NOT #Error_Tx;
   #STAT_AVTF_Mx_MSig := #AVTF_Mx_MSig;
END_REGION

REGION Network 48: VARIABLES AUXILIARES - P_Mens_Mx_MSig (Nota: solo en ET51)
   RUNG wire#powerrail
      Contact( #Mx_ET51 )
      wire#w1
      Coil( #P_Mens_Mx_MSig )
   END_RUNG
   RUNG wire#powerrail
      Contact( #Mx_ET50 )
      { S7_Templates := "SrcType := Int" } GE_Contact(in1 := #CNTSeg_ApHsMx.CVU, in2 := #V_CNTSeg_ApHsMx)
      Contact( "OFF" )
   END_RUNG wire#w1
   // the same network as SCL:
   #P_Mens_Mx_MSig := #Mx_ET51 OR (#Mx_ET50 AND (#CNTSeg_ApHsMx.CVU >= #V_CNTSeg_ApHsMx) AND "OFF");
END_REGION

REGION Network 49: MENSAJES - PRESENCIA
   RUNG wire#powerrail
      Contact( #Mx_ET110 )
      wire#w1
      Contact( #CNTSeg_pHsMx.QU )
      Contact( "OFF" )
      wire#w2
      Contact( #EstadoVI.Etapas_Carga_E1 )
      wire#w3
      S_SR(operand := #STAT_EnvMens_PMx, r1 := wire#w4)
      Coil( #P_EnvMens_PMx )
   END_RUNG
   RUNG wire#w1
      Contact( #CNT_pHsMx.QD )
   END_RUNG wire#w2
   RUNG wire#powerrail
      Contact( #Mx_ET06 )
      Contact( #pHsMx_1 )
   END_RUNG wire#w3
   RUNG wire#powerrail
      Contact( #Mx_ET08 )
      Contact( #pHsMx_2 )
   END_RUNG wire#w3
   RUNG wire#powerrail
      I_Contact( #Mx_ET06 )
      I_Contact( #Mx_ET08 )
      I_Contact( #Mx_ET110 )
   END_RUNG wire#w4
   // the same network as SCL:
   IF (#Mx_ET110 AND ((#CNTSeg_pHsMx.QU AND "OFF") OR #CNT_pHsMx.QD) AND #EstadoVI.Etapas_Carga_E1) OR (#Mx_ET06 AND #pHsMx_1) OR (#Mx_ET08 AND #pHsMx_2) THEN
       #STAT_EnvMens_PMx := TRUE;   // SR flip-flop
   END_IF;
   IF NOT #Mx_ET06 AND NOT #Mx_ET08 AND NOT #Mx_ET110 THEN #STAT_EnvMens_PMx := FALSE; END_IF;
   #P_EnvMens_PMx := #STAT_EnvMens_PMx;
END_REGION

REGION Network 50: MENSAJES - PROTOCOLO INICIADO
   RUNG wire#powerrail
      Contact( #Mx_ET110 )
      Contact( #STAT_EnvMens_PMx )
      S_SR(operand := #ProtocoloIniciado, r1 := wire#w1)
   END_RUNG
   RUNG wire#powerrail
      I_Contact( #Mx_ET110 )
      I_Contact( #Mx_ET111 )
   END_RUNG wire#w1
   // the same network as SCL:
   IF #Mx_ET110 AND #STAT_EnvMens_PMx THEN
       #ProtocoloIniciado := TRUE;   // SR flip-flop
   END_IF;
   IF NOT #Mx_ET110 AND NOT #Mx_ET111 THEN #ProtocoloIniciado := FALSE; END_IF;
END_REGION

REGION Network 51: MENSAJES - RECIBIDA LA ORDEN
   RUNG wire#powerrail
      Contact( #Mx_ET150 )
      Coil( #P_RecepOK_Mx )
   END_RUNG
   // the same network as SCL:
   #P_RecepOK_Mx := #Mx_ET150;
END_REGION

REGION Network 52: SALIDAS - Interlock de DesCarga del VTD - UnLoad OK
   RUNG wire#powerrail
      Contact( #Mx_ET10 )
      wire#w1
      Contact( #Avance_Tx )
      Contact( #EstadoZona.Marcha_CBx )
      Contact( #UnLoadArrival )
      I_Contact( #EstadoVI.Error_Mx )
      I_Contact( #Error_Tx )
      Coil( "DB1_SalidasExterioresDeMesa".Mesa[#Mesa].UnLoadOK )
   END_RUNG
   RUNG wire#powerrail
      Contact( #Mx_ET11 )
      Contact( "OFF" )
   END_RUNG wire#w1
   // the same network as SCL:
   "DB1_SalidasExterioresDeMesa".Mesa[#Mesa].UnLoadOK := (#Mx_ET10 OR (#Mx_ET11 AND "OFF")) AND #Avance_Tx AND #EstadoZona.Marcha_CBx AND #UnLoadArrival AND NOT #EstadoVI.Error_Mx AND NOT #Error_Tx;
END_REGION

REGION Network 53: SALIDAS - Avance E1E3
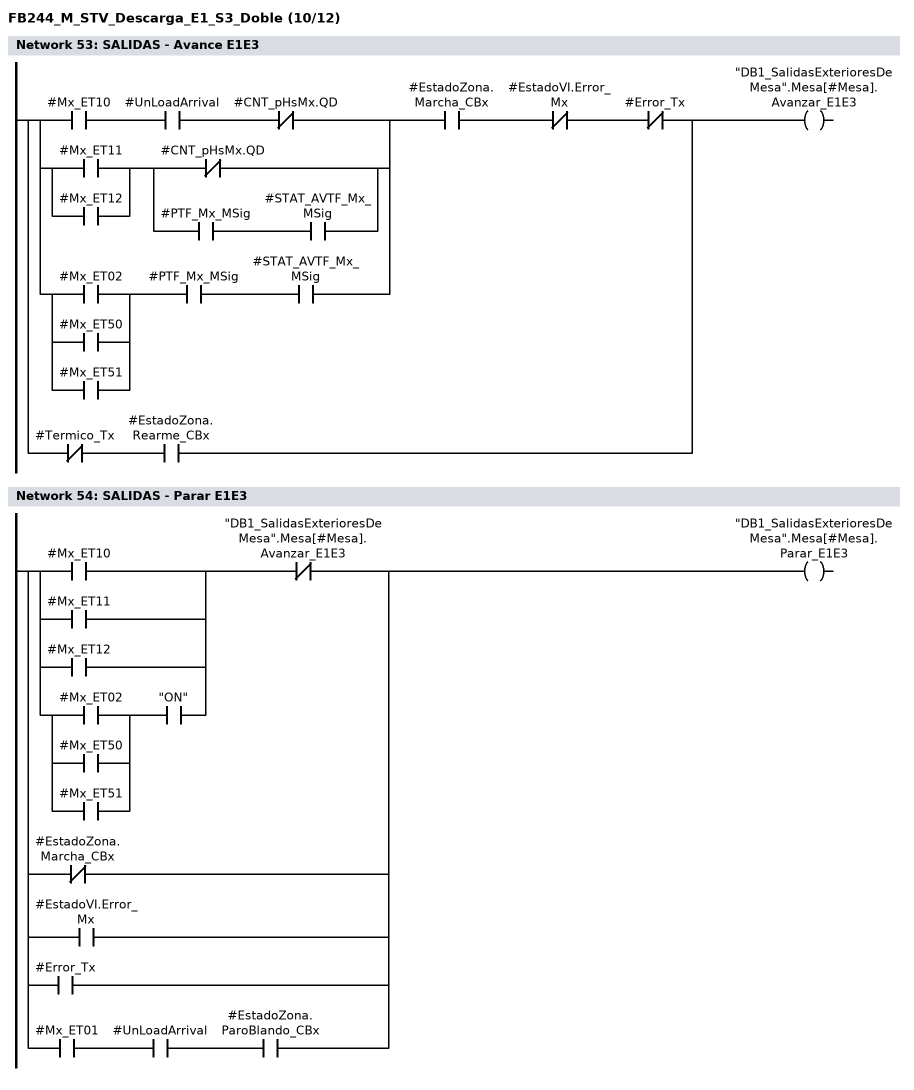
   RUNG wire#powerrail
      Contact( #Mx_ET10 )
      Contact( #UnLoadArrival )
      I_Contact( #CNT_pHsMx.QD )
      wire#w1
      Contact( #EstadoZona.Marcha_CBx )
      I_Contact( #EstadoVI.Error_Mx )
      I_Contact( #Error_Tx )
      wire#w4
      Coil( "DB1_SalidasExterioresDeMesa".Mesa[#Mesa].Avanzar_E1E3 )
   END_RUNG
   RUNG wire#powerrail
      Contact( #Mx_ET11 )
      wire#w2
      I_Contact( #CNT_pHsMx.QD )
   END_RUNG wire#w1
   RUNG wire#powerrail
      Contact( #Mx_ET12 )
   END_RUNG wire#w2
   RUNG wire#w2
      Contact( #PTF_Mx_MSig )
      Contact( #STAT_AVTF_Mx_MSig )
   END_RUNG wire#w1
   RUNG wire#powerrail
      Contact( #Mx_ET02 )
      wire#w3
      Contact( #PTF_Mx_MSig )
      Contact( #STAT_AVTF_Mx_MSig )
   END_RUNG wire#w1
   RUNG wire#powerrail
      Contact( #Mx_ET50 )
   END_RUNG wire#w3
   RUNG wire#powerrail
      Contact( #Mx_ET51 )
   END_RUNG wire#w3
   RUNG wire#powerrail
      I_Contact( #Termico_Tx )
      Contact( #EstadoZona.Rearme_CBx )
   END_RUNG wire#w4
   // the same network as SCL:
   "DB1_SalidasExterioresDeMesa".Mesa[#Mesa].Avanzar_E1E3 := (((#Mx_ET10 AND #UnLoadArrival AND NOT #CNT_pHsMx.QD) OR ((#Mx_ET11 OR #Mx_ET12) AND (NOT #CNT_pHsMx.QD OR (#PTF_Mx_MSig AND #STAT_AVTF_Mx_MSig))) OR ((#Mx_ET02 OR #Mx_ET50 OR #Mx_ET51) AND #PTF_Mx_MSig AND #STAT_AVTF_Mx_MSig)) AND #EstadoZona.Marcha_CBx AND NOT #EstadoVI.Error_Mx AND NOT #Error_Tx) OR (NOT #Termico_Tx AND #EstadoZona.Rearme_CBx);
END_REGION

REGION Network 54: SALIDAS - Parar E1E3
   RUNG wire#powerrail
      Contact( #Mx_ET10 )
      wire#w1
      I_Contact( "DB1_SalidasExterioresDeMesa".Mesa[#Mesa].Avanzar_E1E3 )
      wire#w3
      Coil( "DB1_SalidasExterioresDeMesa".Mesa[#Mesa].Parar_E1E3 )
   END_RUNG
   RUNG wire#powerrail
      Contact( #Mx_ET11 )
   END_RUNG wire#w1
   RUNG wire#powerrail
      Contact( #Mx_ET12 )
   END_RUNG wire#w1
   RUNG wire#powerrail
      Contact( #Mx_ET02 )
      wire#w2
      Contact( "ON" )
   END_RUNG wire#w1
   RUNG wire#powerrail
      Contact( #Mx_ET50 )
   END_RUNG wire#w2
   RUNG wire#powerrail
      Contact( #Mx_ET51 )
   END_RUNG wire#w2
   RUNG wire#powerrail
      I_Contact( #EstadoZona.Marcha_CBx )
   END_RUNG wire#w3
   RUNG wire#powerrail
      Contact( #EstadoVI.Error_Mx )
   END_RUNG wire#w3
   RUNG wire#powerrail
      Contact( #Error_Tx )
   END_RUNG wire#w3
   RUNG wire#powerrail
      Contact( #Mx_ET01 )
      Contact( #UnLoadArrival )
      Contact( #EstadoZona.ParoBlando_CBx )
   END_RUNG wire#w3
   // the same network as SCL:
   "DB1_SalidasExterioresDeMesa".Mesa[#Mesa].Parar_E1E3 := ((#Mx_ET10 OR #Mx_ET11 OR #Mx_ET12 OR ((#Mx_ET02 OR #Mx_ET50 OR #Mx_ET51) AND "ON")) AND NOT "DB1_SalidasExterioresDeMesa".Mesa[#Mesa].Avanzar_E1E3) OR NOT #EstadoZona.Marcha_CBx OR #EstadoVI.Error_Mx OR #Error_Tx OR (#Mx_ET01 AND #UnLoadArrival AND #EstadoZona.ParoBlando_CBx);
END_REGION

REGION Network 55: SALIDAS - Valor Frecuencia Lenta E1E3
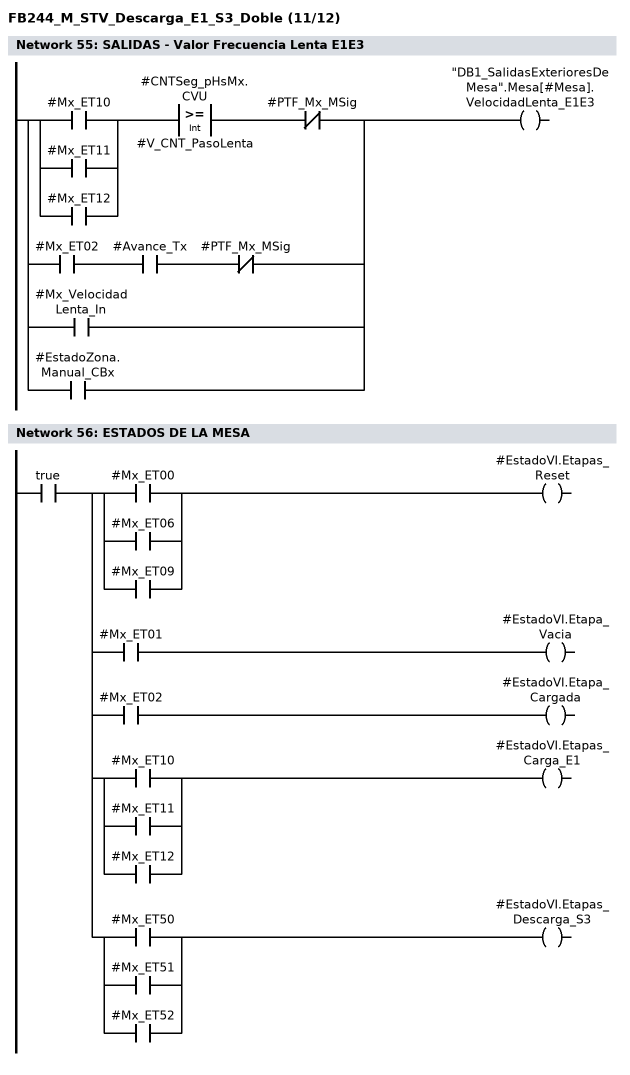
   RUNG wire#powerrail
      Contact( #Mx_ET10 )
      wire#w1
      { S7_Templates := "SrcType := Int" } GE_Contact(in1 := #CNTSeg_pHsMx.CVU, in2 := #V_CNT_PasoLenta)
      I_Contact( #PTF_Mx_MSig )
      wire#w2
      Coil( "DB1_SalidasExterioresDeMesa".Mesa[#Mesa].VelocidadLenta_E1E3 )
   END_RUNG
   RUNG wire#powerrail
      Contact( #Mx_ET11 )
   END_RUNG wire#w1
   RUNG wire#powerrail
      Contact( #Mx_ET12 )
   END_RUNG wire#w1
   RUNG wire#powerrail
      Contact( #Mx_ET02 )
      Contact( #Avance_Tx )
      I_Contact( #PTF_Mx_MSig )
   END_RUNG wire#w2
   RUNG wire#powerrail
      Contact( #Mx_VelocidadLenta_In )
   END_RUNG wire#w2
   RUNG wire#powerrail
      Contact( #EstadoZona.Manual_CBx )
   END_RUNG wire#w2
   // the same network as SCL:
   "DB1_SalidasExterioresDeMesa".Mesa[#Mesa].VelocidadLenta_E1E3 := ((#Mx_ET10 OR #Mx_ET11 OR #Mx_ET12) AND (#CNTSeg_pHsMx.CVU >= #V_CNT_PasoLenta) AND NOT #PTF_Mx_MSig) OR (#Mx_ET02 AND #Avance_Tx AND NOT #PTF_Mx_MSig) OR #Mx_VelocidadLenta_In OR #EstadoZona.Manual_CBx;
END_REGION

REGION Network 56: ESTADOS DE LA MESA
   RUNG wire#powerrail
      Contact( true )
      wire#w1
      Contact( #Mx_ET00 )
      wire#w2
      Coil( #EstadoVI.Etapas_Reset )
   END_RUNG
   RUNG wire#w1
      Contact( #Mx_ET06 )
   END_RUNG wire#w2
   RUNG wire#w1
      Contact( #Mx_ET09 )
   END_RUNG wire#w2
   RUNG wire#w1
      Contact( #Mx_ET01 )
      Coil( #EstadoVI.Etapa_Vacia )
   END_RUNG
   RUNG wire#w1
      Contact( #Mx_ET02 )
      Coil( #EstadoVI.Etapa_Cargada )
   END_RUNG
   RUNG wire#w1
      Contact( #Mx_ET10 )
      wire#w3
      Coil( #EstadoVI.Etapas_Carga_E1 )
   END_RUNG
   RUNG wire#w1
      Contact( #Mx_ET11 )
   END_RUNG wire#w3
   RUNG wire#w1
      Contact( #Mx_ET12 )
   END_RUNG wire#w3
   RUNG wire#w1
      Contact( #Mx_ET50 )
      wire#w4
      Coil( #EstadoVI.Etapas_Descarga_S3 )
   END_RUNG
   RUNG wire#w1
      Contact( #Mx_ET51 )
   END_RUNG wire#w4
   RUNG wire#w1
      Contact( #Mx_ET52 )
   END_RUNG wire#w4
   // the same network as SCL:
   #EstadoVI.Etapas_Reset := true AND (#Mx_ET00 OR #Mx_ET06 OR #Mx_ET09);
   #EstadoVI.Etapa_Vacia := true AND #Mx_ET01;
   #EstadoVI.Etapa_Cargada := true AND #Mx_ET02;
   #EstadoVI.Etapas_Carga_E1 := true AND (#Mx_ET10 OR #Mx_ET11 OR #Mx_ET12);
   #EstadoVI.Etapas_Descarga_S3 := true AND (#Mx_ET50 OR #Mx_ET51 OR #Mx_ET52);
END_REGION

REGION Network 57: ENTRADAS DE LA MESA
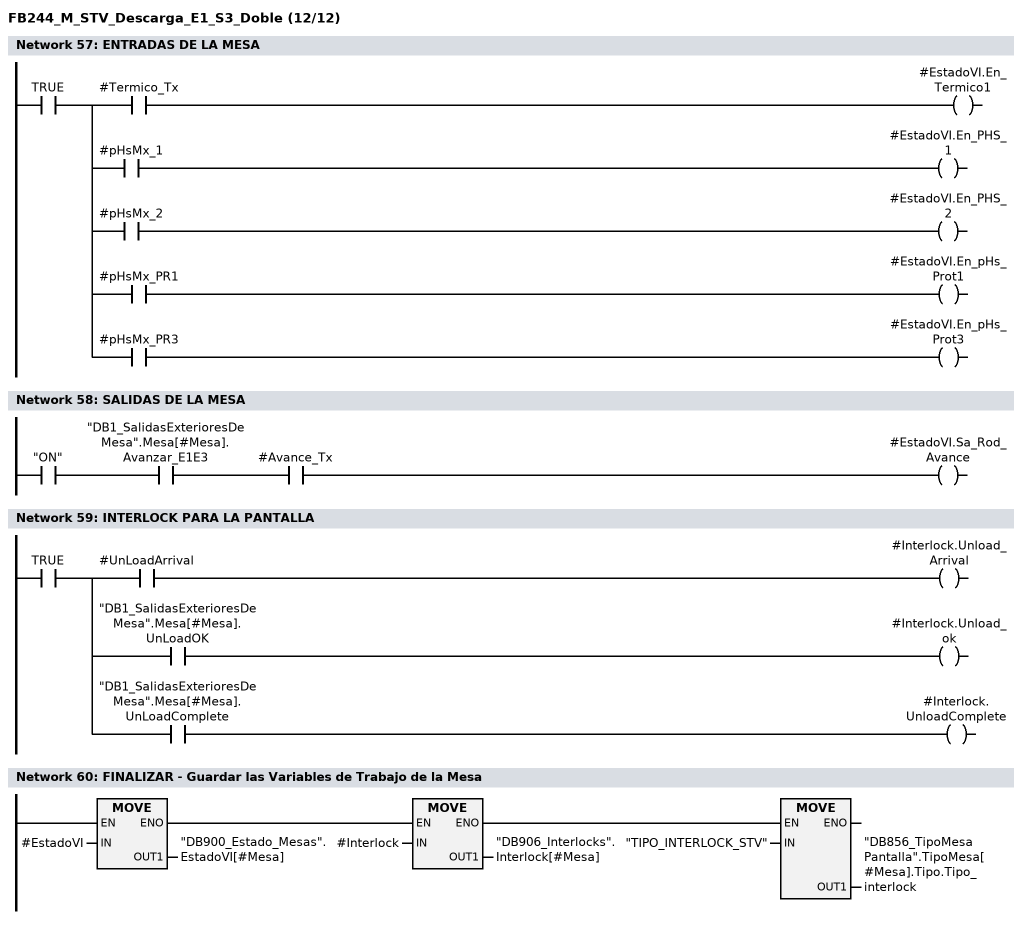
   RUNG wire#powerrail
      Contact( TRUE )
      wire#w1
      Contact( #Termico_Tx )
      Coil( #EstadoVI.En_Termico1 )
   END_RUNG
   RUNG wire#w1
      Contact( #pHsMx_1 )
      Coil( #EstadoVI.En_PHS_1 )
   END_RUNG
   RUNG wire#w1
      Contact( #pHsMx_2 )
      Coil( #EstadoVI.En_PHS_2 )
   END_RUNG
   RUNG wire#w1
      Contact( #pHsMx_PR1 )
      Coil( #EstadoVI.En_pHs_Prot1 )
   END_RUNG
   RUNG wire#w1
      Contact( #pHsMx_PR3 )
      Coil( #EstadoVI.En_pHs_Prot3 )
   END_RUNG
   // the same network as SCL:
   #EstadoVI.En_Termico1 := TRUE AND #Termico_Tx;
   #EstadoVI.En_PHS_1 := TRUE AND #pHsMx_1;
   #EstadoVI.En_PHS_2 := TRUE AND #pHsMx_2;
   #EstadoVI.En_pHs_Prot1 := TRUE AND #pHsMx_PR1;
   #EstadoVI.En_pHs_Prot3 := TRUE AND #pHsMx_PR3;
END_REGION

REGION Network 58: SALIDAS DE LA MESA
   RUNG wire#powerrail
      Contact( "ON" )
      Contact( "DB1_SalidasExterioresDeMesa".Mesa[#Mesa].Avanzar_E1E3 )
      Contact( #Avance_Tx )
      Coil( #EstadoVI.Sa_Rod_Avance )
   END_RUNG
   // the same network as SCL:
   #EstadoVI.Sa_Rod_Avance := "ON" AND "DB1_SalidasExterioresDeMesa".Mesa[#Mesa].Avanzar_E1E3 AND #Avance_Tx;
END_REGION

REGION Network 59: INTERLOCK PARA LA PANTALLA
   RUNG wire#powerrail
      Contact( TRUE )
      wire#w1
      Contact( #UnLoadArrival )
      Coil( #Interlock.Unload_Arrival )
   END_RUNG
   RUNG wire#w1
      Contact( "DB1_SalidasExterioresDeMesa".Mesa[#Mesa].UnLoadOK )
      Coil( #Interlock.Unload_ok )
   END_RUNG
   RUNG wire#w1
      Contact( "DB1_SalidasExterioresDeMesa".Mesa[#Mesa].UnLoadComplete )
      Coil( #Interlock.UnloadComplete )
   END_RUNG
   // the same network as SCL:
   #Interlock.Unload_Arrival := TRUE AND #UnLoadArrival;
   #Interlock.Unload_ok := TRUE AND "DB1_SalidasExterioresDeMesa".Mesa[#Mesa].UnLoadOK;
   #Interlock.UnloadComplete := TRUE AND "DB1_SalidasExterioresDeMesa".Mesa[#Mesa].UnLoadComplete;
END_REGION

REGION Network 60: FINALIZAR - Guardar las Variables de Trabajo de la Mesa
   RUNG wire#powerrail
      Move(in := #EstadoVI, out1 => "DB900_Estado_Mesas".EstadoVI[#Mesa])
      Move(in := #Interlock, out1 => "DB906_Interlocks".Interlock[#Mesa])
      Move(in := "TIPO_INTERLOCK_STV", out1 => "DB856_TipoMesaPantalla".TipoMesa[#Mesa].Tipo.Tipo_interlock)
   END_RUNG
   // the same network as SCL:
   "DB900_Estado_Mesas".EstadoVI[#Mesa] := #EstadoVI;
   "DB906_Interlocks".Interlock[#Mesa] := #Interlock;
   "DB856_TipoMesaPantalla".TipoMesa[#Mesa].Tipo.Tipo_interlock := "TIPO_INTERLOCK_STV";
END_REGION
END_FUNCTION_BLOCK

